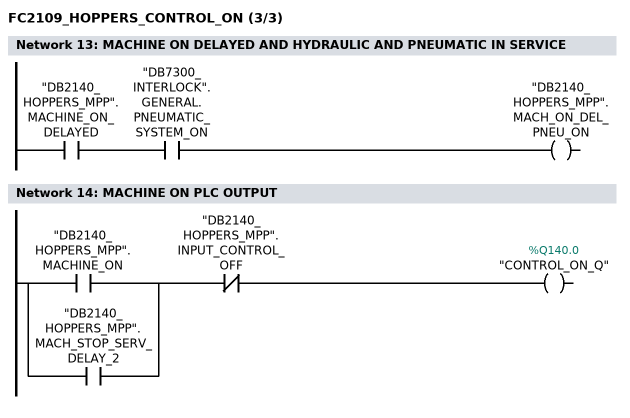
   RUNG wire#powerrail
      Contact( "DB2140_HOPPERS_MPP".MACHINE_ON_DELAYED )
      Contact( "DB7300_INTERLOCK".GENERAL.PNEUMATIC_SYSTEM_ON )
      Coil( "DB2140_HOPPERS_MPP".MACH_ON_DEL_PNEU_ON )
   END_RUNG
   // the same network as SCL:
   "DB2140_HOPPERS_MPP".MACH_ON_DEL_PNEU_ON := "DB2140_HOPPERS_MPP".MACHINE_ON_DELAYED AND "DB7300_INTERLOCK".GENERAL.PNEUMATIC_SYSTEM_ON;
END_REGION

REGION Network 14: MACHINE ON PLC OUTPUT
   RUNG wire#powerrail
      Contact( "DB2140_HOPPERS_MPP".MACHINE_ON )
      wire#w1
      I_Contact( "DB2140_HOPPERS_MPP".INPUT_CONTROL_OFF )
      Coil( "CONTROL_ON_Q" )
   END_RUNG
   RUNG wire#powerrail
      Contact( "DB2140_HOPPERS_MPP".MACH_STOP_SERV_DELAY_2 )
   END_RUNG wire#w1
   // the same network as SCL:
   "CONTROL_ON_Q" := ("DB2140_HOPPERS_MPP".MACHINE_ON OR "DB2140_HOPPERS_MPP".MACH_STOP_SERV_DELAY_2) AND NOT "DB2140_HOPPERS_MPP".INPUT_CONTROL_OFF;
END_REGION
END_FUNCTION

FUNCTION "FC2140_HOPPERS_BUTTONS" : Void   // FC2140, LAD
{ S7_Optimized_Access := 'FALSE' }
AUTHOR : ETXETAR
VERSION : 1.0
// stored: AutoNumber false, IsIECCheckEnabled false, SetENOAutomatically false, UDAEnableTagReadback false
   VAR_TEMP
      O_BYTE_0 : Struct   // OPTIONS BYTE 0
         IPC : Bool;   // IPC OPTION
      END_STRUCT;
      TCU_INDEX_SEL : Int;
   END_VAR
   VAR CONSTANT
      FC_NUMBER : DInt := 2140;   // FC NUMBER
   END_VAR
   VAR_TEMP   // added for the SCL form of the ladder/FBD networks
      _w1 : Bool;
   END_VAR
BEGIN

REGION Network 1: OPTIONS
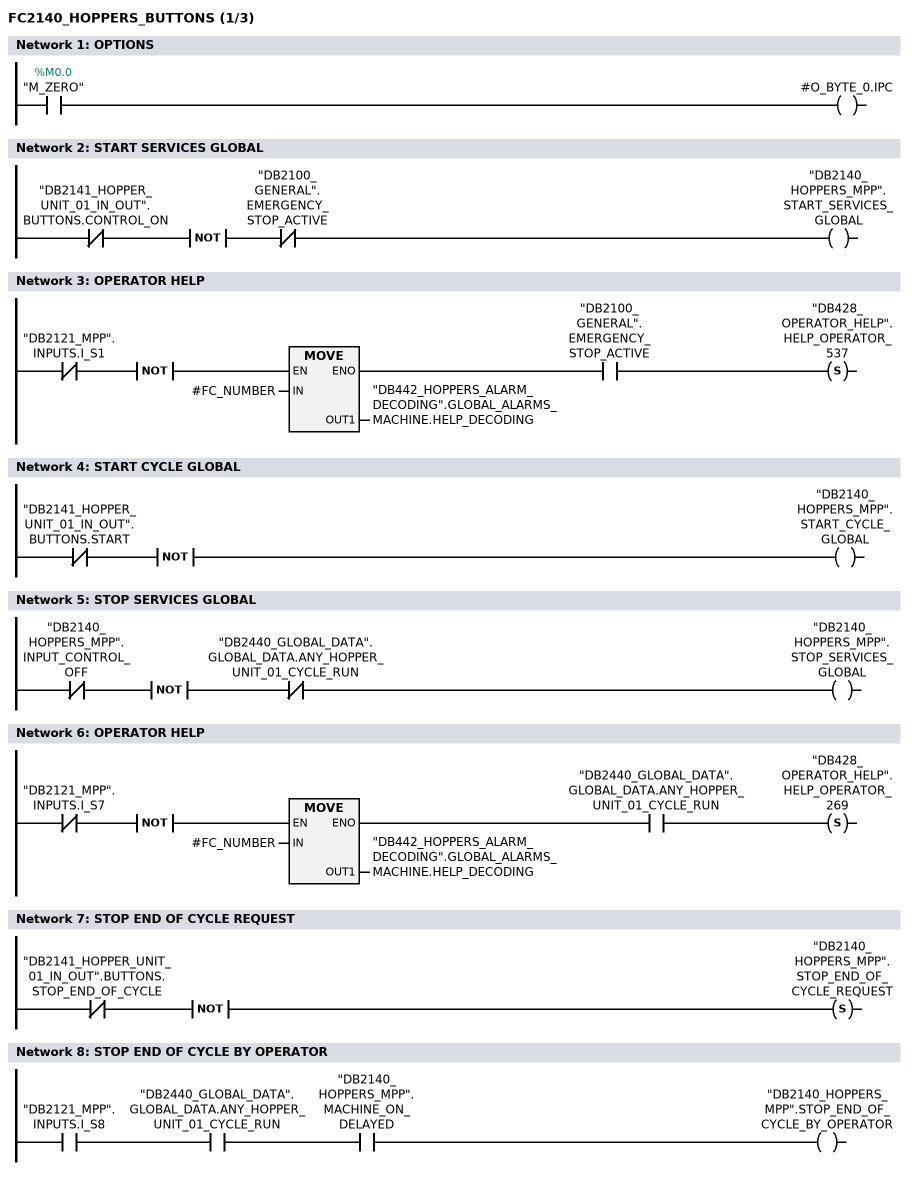
   RUNG wire#powerrail
      Contact( "M_ZERO" )
      Coil( #O_BYTE_0.IPC )
   END_RUNG
   // the same network as SCL:
   #O_BYTE_0.IPC := "M_ZERO";
END_REGION

REGION Network 2: START SERVICES GLOBAL
   RUNG wire#powerrail
      I_Contact( "DB2141_HOPPER_UNIT_01_IN_OUT".BUTTONS.CONTROL_ON )
      Not()
      I_Contact( "DB2100_GENERAL".EMERGENCY_STOP_ACTIVE )
      Coil( "DB2140_HOPPERS_MPP".START_SERVICES_GLOBAL )
   END_RUNG
   // the same network as SCL:
   "DB2140_HOPPERS_MPP".START_SERVICES_GLOBAL := NOT (NOT "DB2141_HOPPER_UNIT_01_IN_OUT".BUTTONS.CONTROL_ON) AND NOT "DB2100_GENERAL".EMERGENCY_STOP_ACTIVE;
END_REGION

REGION Network 3: OPERATOR HELP
   RUNG wire#powerrail
      I_Contact( "DB2121_MPP".INPUTS.I_S1 )
      Not()
      { S7_GenerateENO := "TRUE" } Move(in := #FC_NUMBER, out1 => "DB442_HOPPERS_ALARM_DECODING".GLOBAL_ALARMS_MACHINE.HELP_DECODING)
      Contact( "DB2100_GENERAL".EMERGENCY_STOP_ACTIVE )
      S_Coil( "DB428_OPERATOR_HELP".HELP_OPERATOR_537 )
   END_RUNG
   // the same network as SCL:
   // ENO of a box is taken as its EN; it also drops when the box reports an error
   #_w1 := NOT (NOT "DB2121_MPP".INPUTS.I_S1);
   IF #_w1 THEN "DB442_HOPPERS_ALARM_DECODING".GLOBAL_ALARMS_MACHINE.HELP_DECODING := #FC_NUMBER; END_IF;
   IF #_w1 AND "DB2100_GENERAL".EMERGENCY_STOP_ACTIVE THEN
       "DB428_OPERATOR_HELP".HELP_OPERATOR_537 := TRUE;
   END_IF;
END_REGION

REGION Network 4: START CYCLE GLOBAL
   RUNG wire#powerrail
      I_Contact( "DB2141_HOPPER_UNIT_01_IN_OUT".BUTTONS.START )
      Not()
      Coil( "DB2140_HOPPERS_MPP".START_CYCLE_GLOBAL )
   END_RUNG
   // the same network as SCL:
   "DB2140_HOPPERS_MPP".START_CYCLE_GLOBAL := NOT (NOT "DB2141_HOPPER_UNIT_01_IN_OUT".BUTTONS.START);
END_REGION

REGION Network 5: STOP SERVICES GLOBAL
   RUNG wire#powerrail
      I_Contact( "DB2140_HOPPERS_MPP".INPUT_CONTROL_OFF )
      Not()
      I_Contact( "DB2440_GLOBAL_DATA".GLOBAL_DATA.ANY_HOPPER_UNIT_01_CYCLE_RUN )
      Coil( "DB2140_HOPPERS_MPP".STOP_SERVICES_GLOBAL )
   END_RUNG
   // the same network as SCL:
   "DB2140_HOPPERS_MPP".STOP_SERVICES_GLOBAL := NOT (NOT "DB2140_HOPPERS_MPP".INPUT_CONTROL_OFF) AND NOT "DB2440_GLOBAL_DATA".GLOBAL_DATA.ANY_HOPPER_UNIT_01_CYCLE_RUN;
END_REGION

REGION Network 6: OPERATOR HELP
   RUNG wire#powerrail
      I_Contact( "DB2121_MPP".INPUTS.I_S7 )
      Not()
      { S7_GenerateENO := "TRUE" } Move(in := #FC_NUMBER, out1 => "DB442_HOPPERS_ALARM_DECODING".GLOBAL_ALARMS_MACHINE.HELP_DECODING)
      Contact( "DB2440_GLOBAL_DATA".GLOBAL_DATA.ANY_HOPPER_UNIT_01_CYCLE_RUN )
      S_Coil( "DB428_OPERATOR_HELP".HELP_OPERATOR_269 )
   END_RUNG
   // the same network as SCL:
   // ENO of a box is taken as its EN; it also drops when the box reports an error
   #_w1 := NOT (NOT "DB2121_MPP".INPUTS.I_S7);
   IF #_w1 THEN "DB442_HOPPERS_ALARM_DECODING".GLOBAL_ALARMS_MACHINE.HELP_DECODING := #FC_NUMBER; END_IF;
   IF #_w1 AND "DB2440_GLOBAL_DATA".GLOBAL_DATA.ANY_HOPPER_UNIT_01_CYCLE_RUN THEN
       "DB428_OPERATOR_HELP".HELP_OPERATOR_269 := TRUE;
   END_IF;
END_REGION

REGION Network 7: STOP END OF CYCLE REQUEST
   RUNG wire#powerrail
      I_Contact( "DB2141_HOPPER_UNIT_01_IN_OUT".BUTTONS.STOP_END_OF_CYCLE )
      Not()
      S_Coil( "DB2140_HOPPERS_MPP".STOP_END_OF_CYCLE_REQUEST )
   END_RUNG
   // the same network as SCL:
   IF NOT (NOT "DB2141_HOPPER_UNIT_01_IN_OUT".BUTTONS.STOP_END_OF_CYCLE) THEN
       "DB2140_HOPPERS_MPP".STOP_END_OF_CYCLE_REQUEST := TRUE;
   END_IF;
END_REGION

REGION Network 8: STOP END OF CYCLE BY OPERATOR
   RUNG wire#powerrail
      Contact( "DB2121_MPP".INPUTS.I_S8 )
      Contact( "DB2440_GLOBAL_DATA".GLOBAL_DATA.ANY_HOPPER_UNIT_01_CYCLE_RUN )
      Contact( "DB2140_HOPPERS_MPP".MACHINE_ON_DELAYED )
      Coil( "DB2140_HOPPERS_MPP".STOP_END_OF_CYCLE_BY_OPERATOR )
   END_RUNG
   // the same network as SCL:
   "DB2140_HOPPERS_MPP".STOP_END_OF_CYCLE_BY_OPERATOR := "DB2121_MPP".INPUTS.I_S8 AND "DB2440_GLOBAL_DATA".GLOBAL_DATA.ANY_HOPPER_UNIT_01_CYCLE_RUN AND "DB2140_HOPPERS_MPP".MACHINE_ON_DELAYED;
END_REGION

REGION Network 9: MAIN PANEL OPERATOR REQUEST STOP AT END OF CYCLE
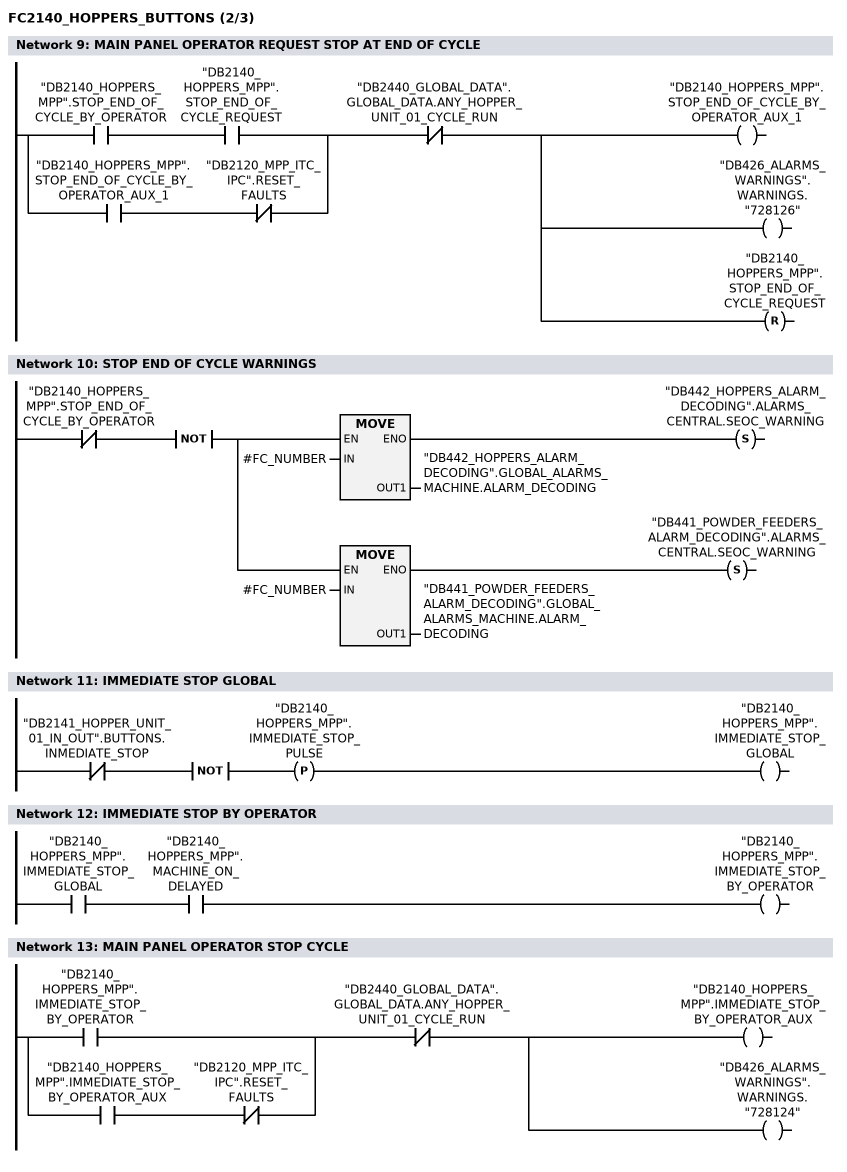
   RUNG wire#powerrail
      Contact( "DB2140_HOPPERS_MPP".STOP_END_OF_CYCLE_BY_OPERATOR )
      Contact( "DB2140_HOPPERS_MPP".STOP_END_OF_CYCLE_REQUEST )
      wire#w1
      I_Contact( "DB2440_GLOBAL_DATA".GLOBAL_DATA.ANY_HOPPER_UNIT_01_CYCLE_RUN )
      wire#w2
      Coil( "DB2140_HOPPERS_MPP".STOP_END_OF_CYCLE_BY_OPERATOR_AUX_1 )
   END_RUNG
   RUNG wire#powerrail
      Contact( "DB2140_HOPPERS_MPP".STOP_END_OF_CYCLE_BY_OPERATOR_AUX_1 )
      I_Contact( "DB2120_MPP_ITC_IPC".RESET_FAULTS )
   END_RUNG wire#w1
   RUNG wire#w2
      Coil( "DB426_ALARMS_WARNINGS".WARNINGS."728126" )
   END_RUNG
   RUNG wire#w2
      R_Coil( "DB2140_HOPPERS_MPP".STOP_END_OF_CYCLE_REQUEST )
   END_RUNG
   // the same network as SCL:
   "DB2140_HOPPERS_MPP".STOP_END_OF_CYCLE_BY_OPERATOR_AUX_1 := (("DB2140_HOPPERS_MPP".STOP_END_OF_CYCLE_BY_OPERATOR AND "DB2140_HOPPERS_MPP".STOP_END_OF_CYCLE_REQUEST) OR ("DB2140_HOPPERS_MPP".STOP_END_OF_CYCLE_BY_OPERATOR_AUX_1 AND NOT "DB2120_MPP_ITC_IPC".RESET_FAULTS)) AND NOT "DB2440_GLOBAL_DATA".GLOBAL_DATA.ANY_HOPPER_UNIT_01_CYCLE_RUN;
   "DB426_ALARMS_WARNINGS".WARNINGS."728126" := "DB2140_HOPPERS_MPP".STOP_END_OF_CYCLE_BY_OPERATOR_AUX_1;
   IF "DB2140_HOPPERS_MPP".STOP_END_OF_CYCLE_BY_OPERATOR_AUX_1 THEN
       "DB2140_HOPPERS_MPP".STOP_END_OF_CYCLE_REQUEST := FALSE;
   END_IF;
END_REGION

REGION Network 10: STOP END OF CYCLE WARNINGS
   RUNG wire#powerrail
      I_Contact( "DB2140_HOPPERS_MPP".STOP_END_OF_CYCLE_BY_OPERATOR )
      Not()
      wire#w1
      { S7_GenerateENO := "TRUE" } Move(in := #FC_NUMBER, out1 => "DB442_HOPPERS_ALARM_DECODING".GLOBAL_ALARMS_MACHINE.ALARM_DECODING)
      S_Coil( "DB442_HOPPERS_ALARM_DECODING".ALARMS_CENTRAL.SEOC_WARNING )
   END_RUNG
   RUNG wire#w1
      { S7_GenerateENO := "TRUE" } Move(in := #FC_NUMBER, out1 => "DB441_POWDER_FEEDERS_ALARM_DECODING".GLOBAL_ALARMS_MACHINE.ALARM_DECODING)
      S_Coil( "DB441_POWDER_FEEDERS_ALARM_DECODING".ALARMS_CENTRAL.SEOC_WARNING )
   END_RUNG
   // the same network as SCL:
   // ENO of a box is taken as its EN; it also drops when the box reports an error
   IF NOT (NOT "DB2140_HOPPERS_MPP".STOP_END_OF_CYCLE_BY_OPERATOR) THEN
       "DB442_HOPPERS_ALARM_DECODING".GLOBAL_ALARMS_MACHINE.ALARM_DECODING := #FC_NUMBER;
       "DB442_HOPPERS_ALARM_DECODING".ALARMS_CENTRAL.SEOC_WARNING := TRUE;
       "DB441_POWDER_FEEDERS_ALARM_DECODING".GLOBAL_ALARMS_MACHINE.ALARM_DECODING := #FC_NUMBER;
       "DB441_POWDER_FEEDERS_ALARM_DECODING".ALARMS_CENTRAL.SEOC_WARNING := TRUE;
   END_IF;
END_REGION

REGION Network 11: IMMEDIATE STOP GLOBAL
   RUNG wire#powerrail
      I_Contact( "DB2141_HOPPER_UNIT_01_IN_OUT".BUTTONS.INMEDIATE_STOP )
      Not()
      P_Trig( "DB2140_HOPPERS_MPP".IMMEDIATE_STOP_PULSE )
      Coil( "DB2140_HOPPERS_MPP".IMMEDIATE_STOP_GLOBAL )
   END_RUNG
   // the same network as SCL:
   #_w1 := NOT (NOT "DB2141_HOPPER_UNIT_01_IN_OUT".BUTTONS.INMEDIATE_STOP) AND NOT "DB2140_HOPPERS_MPP".IMMEDIATE_STOP_PULSE;   // rising edge
   "DB2140_HOPPERS_MPP".IMMEDIATE_STOP_PULSE := NOT (NOT "DB2141_HOPPER_UNIT_01_IN_OUT".BUTTONS.INMEDIATE_STOP);
   "DB2140_HOPPERS_MPP".IMMEDIATE_STOP_GLOBAL := #_w1;
END_REGION

REGION Network 12: IMMEDIATE STOP BY OPERATOR
   RUNG wire#powerrail
      Contact( "DB2140_HOPPERS_MPP".IMMEDIATE_STOP_GLOBAL )
      Contact( "DB2140_HOPPERS_MPP".MACHINE_ON_DELAYED )
      Coil( "DB2140_HOPPERS_MPP".IMMEDIATE_STOP_BY_OPERATOR )
   END_RUNG
   // the same network as SCL:
   "DB2140_HOPPERS_MPP".IMMEDIATE_STOP_BY_OPERATOR := "DB2140_HOPPERS_MPP".IMMEDIATE_STOP_GLOBAL AND "DB2140_HOPPERS_MPP".MACHINE_ON_DELAYED;
END_REGION

REGION Network 13: MAIN PANEL OPERATOR STOP CYCLE
   RUNG wire#powerrail
      Contact( "DB2140_HOPPERS_MPP".IMMEDIATE_STOP_BY_OPERATOR )
      wire#w1
      I_Contact( "DB2440_GLOBAL_DATA".GLOBAL_DATA.ANY_HOPPER_UNIT_01_CYCLE_RUN )
      wire#w2
      Coil( "DB2140_HOPPERS_MPP".IMMEDIATE_STOP_BY_OPERATOR_AUX )
   END_RUNG
   RUNG wire#powerrail
      Contact( "DB2140_HOPPERS_MPP".IMMEDIATE_STOP_BY_OPERATOR_AUX )
      I_Contact( "DB2120_MPP_ITC_IPC".RESET_FAULTS )
   END_RUNG wire#w1
   RUNG wire#w2
      Coil( "DB426_ALARMS_WARNINGS".WARNINGS."728124" )
   END_RUNG
   // the same network as SCL:
   "DB2140_HOPPERS_MPP".IMMEDIATE_STOP_BY_OPERATOR_AUX := ("DB2140_HOPPERS_MPP".IMMEDIATE_STOP_BY_OPERATOR OR ("DB2140_HOPPERS_MPP".IMMEDIATE_STOP_BY_OPERATOR_AUX AND NOT "DB2120_MPP_ITC_IPC".RESET_FAULTS)) AND NOT "DB2440_GLOBAL_DATA".GLOBAL_DATA.ANY_HOPPER_UNIT_01_CYCLE_RUN;
   "DB426_ALARMS_WARNINGS".WARNINGS."728124" := "DB2140_HOPPERS_MPP".IMMEDIATE_STOP_BY_OPERATOR_AUX;
END_REGION

REGION Network 14: IMMEDIATE STOP WARNING
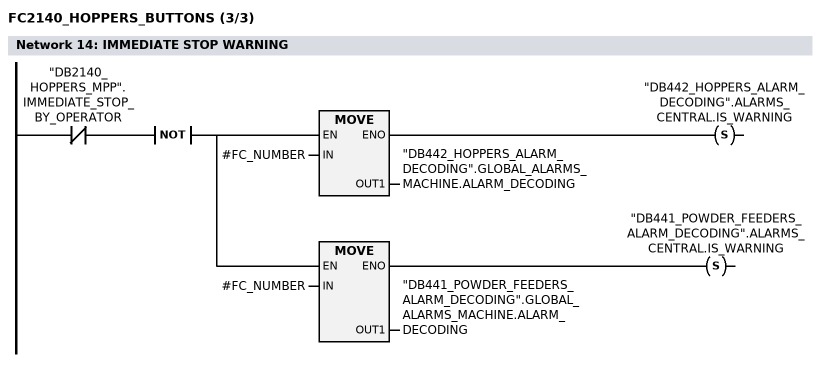
   RUNG wire#powerrail
      I_Contact( "DB2140_HOPPERS_MPP".IMMEDIATE_STOP_BY_OPERATOR )
      Not()
      wire#w1
      { S7_GenerateENO := "TRUE" } Move(in := #FC_NUMBER, out1 => "DB442_HOPPERS_ALARM_DECODING".GLOBAL_ALARMS_MACHINE.ALARM_DECODING)
      S_Coil( "DB442_HOPPERS_ALARM_DECODING".ALARMS_CENTRAL.IS_WARNING )
   END_RUNG
   RUNG wire#w1
      { S7_GenerateENO := "TRUE" } Move(in := #FC_NUMBER, out1 => "DB441_POWDER_FEEDERS_ALARM_DECODING".GLOBAL_ALARMS_MACHINE.ALARM_DECODING)
      S_Coil( "DB441_POWDER_FEEDERS_ALARM_DECODING".ALARMS_CENTRAL.IS_WARNING )
   END_RUNG
   // the same network as SCL:
   // ENO of a box is taken as its EN; it also drops when the box reports an error
   IF NOT (NOT "DB2140_HOPPERS_MPP".IMMEDIATE_STOP_BY_OPERATOR) THEN
       "DB442_HOPPERS_ALARM_DECODING".GLOBAL_ALARMS_MACHINE.ALARM_DECODING := #FC_NUMBER;
       "DB442_HOPPERS_ALARM_DECODING".ALARMS_CENTRAL.IS_WARNING := TRUE;
       "DB441_POWDER_FEEDERS_ALARM_DECODING".GLOBAL_ALARMS_MACHINE.ALARM_DECODING := #FC_NUMBER;
       "DB441_POWDER_FEEDERS_ALARM_DECODING".ALARMS_CENTRAL.IS_WARNING := TRUE;
   END_IF;
END_REGION
END_FUNCTION

FUNCTION "FC2141_HOPPERS_LAMPS" : Void   // FC2141, LAD
{ S7_Optimized_Access := 'FALSE' }
AUTHOR : ETXETAR
VERSION : 1.0
// stored: AutoNumber false, IsIECCheckEnabled false, SetENOAutomatically false, UDAEnableTagReadback false
   VAR_TEMP
      ONE : Int;
      RETVAL1 : Int;
      SIMU_PANEL_HMI_SEL : Bool;   // SIMULATED PANEL IN HMI SELECTED
   END_VAR
   VAR CONSTANT
      FC_NUMBER : DInt := 2141;   // FC NUMBER
   END_VAR
BEGIN

REGION Network 1: LAMP - CONTROL ON
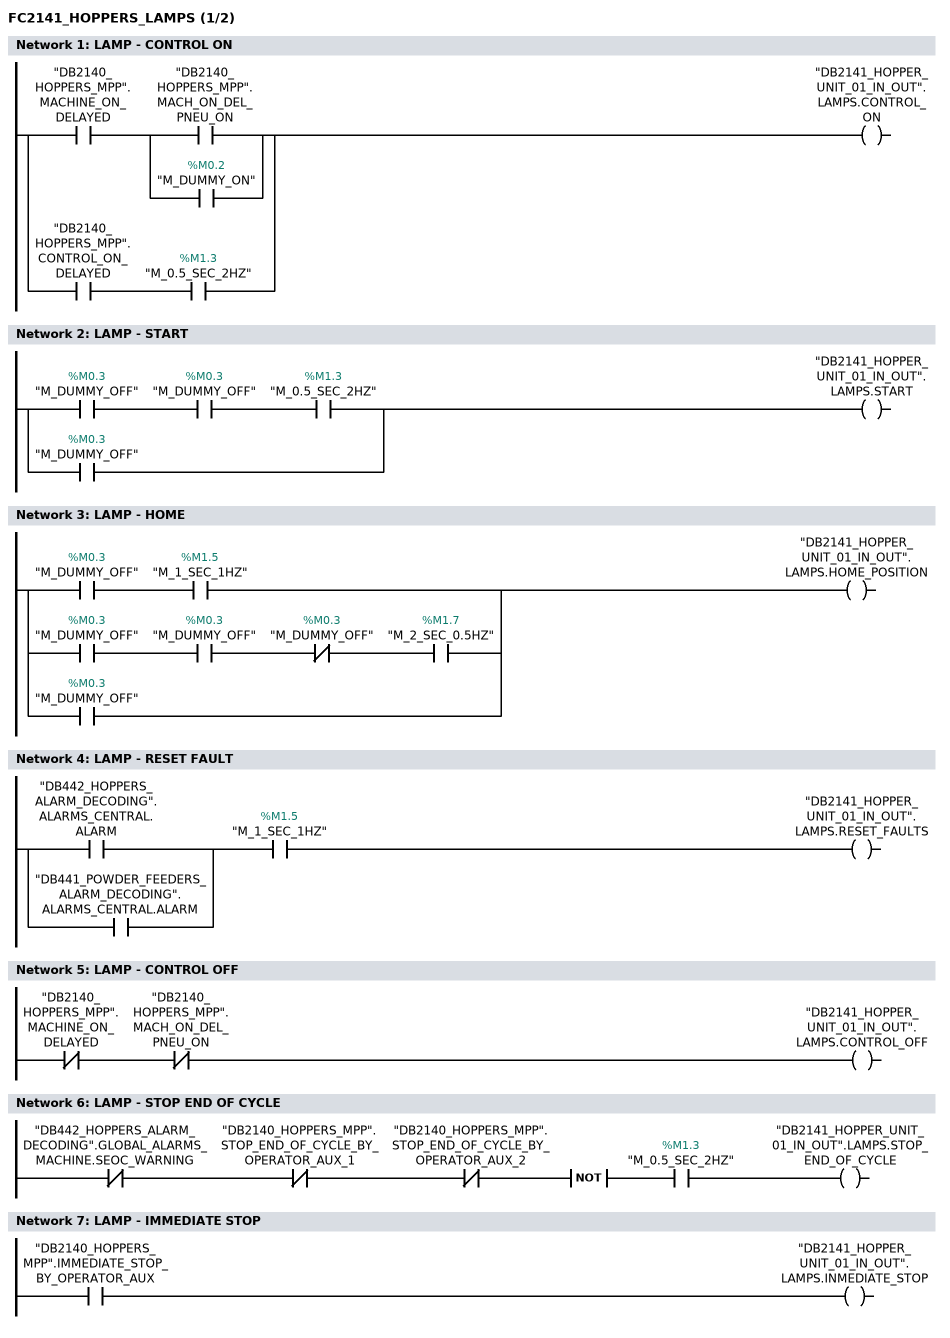
   RUNG wire#powerrail
      Contact( "DB2140_HOPPERS_MPP".MACHINE_ON_DELAYED )
      wire#w1
      Contact( "DB2140_HOPPERS_MPP".MACH_ON_DEL_PNEU_ON )
      wire#w2
      Coil( "DB2141_HOPPER_UNIT_01_IN_OUT".LAMPS.CONTROL_ON )
   END_RUNG
   RUNG wire#w1
      Contact( "M_DUMMY_ON" )
   END_RUNG wire#w2
   RUNG wire#powerrail
      Contact( "DB2140_HOPPERS_MPP".CONTROL_ON_DELAYED )
      Contact( "M_0.5_SEC_2HZ" )
   END_RUNG wire#w2
   // the same network as SCL:
   "DB2141_HOPPER_UNIT_01_IN_OUT".LAMPS.CONTROL_ON := ("DB2140_HOPPERS_MPP".MACHINE_ON_DELAYED AND ("DB2140_HOPPERS_MPP".MACH_ON_DEL_PNEU_ON OR "M_DUMMY_ON")) OR ("DB2140_HOPPERS_MPP".CONTROL_ON_DELAYED AND "M_0.5_SEC_2HZ");
END_REGION

REGION Network 2: LAMP - START
   RUNG wire#powerrail
      Contact( "M_DUMMY_OFF" )
      Contact( "M_DUMMY_OFF" )
      Contact( "M_0.5_SEC_2HZ" )
      wire#w1
      Coil( "DB2141_HOPPER_UNIT_01_IN_OUT".LAMPS.START )
   END_RUNG
   RUNG wire#powerrail
      Contact( "M_DUMMY_OFF" )
   END_RUNG wire#w1
   // the same network as SCL:
   "DB2141_HOPPER_UNIT_01_IN_OUT".LAMPS.START := ("M_DUMMY_OFF" AND "M_DUMMY_OFF" AND "M_0.5_SEC_2HZ") OR "M_DUMMY_OFF";
END_REGION

REGION Network 3: LAMP - HOME
   RUNG wire#powerrail
      Contact( "M_DUMMY_OFF" )
      Contact( "M_1_SEC_1HZ" )
      wire#w1
      Coil( "DB2141_HOPPER_UNIT_01_IN_OUT".LAMPS.HOME_POSITION )
   END_RUNG
   RUNG wire#powerrail
      Contact( "M_DUMMY_OFF" )
      Contact( "M_DUMMY_OFF" )
      I_Contact( "M_DUMMY_OFF" )
      Contact( "M_2_SEC_0.5HZ" )
   END_RUNG wire#w1
   RUNG wire#powerrail
      Contact( "M_DUMMY_OFF" )
   END_RUNG wire#w1
   // the same network as SCL:
   "DB2141_HOPPER_UNIT_01_IN_OUT".LAMPS.HOME_POSITION := ("M_DUMMY_OFF" AND "M_1_SEC_1HZ") OR ("M_DUMMY_OFF" AND "M_DUMMY_OFF" AND NOT "M_DUMMY_OFF" AND "M_2_SEC_0.5HZ") OR "M_DUMMY_OFF";
END_REGION

REGION Network 4: LAMP - RESET FAULT
   RUNG wire#powerrail
      Contact( "DB442_HOPPERS_ALARM_DECODING".ALARMS_CENTRAL.ALARM )
      wire#w1
      Contact( "M_1_SEC_1HZ" )
      Coil( "DB2141_HOPPER_UNIT_01_IN_OUT".LAMPS.RESET_FAULTS )
   END_RUNG
   RUNG wire#powerrail
      Contact( "DB441_POWDER_FEEDERS_ALARM_DECODING".ALARMS_CENTRAL.ALARM )
   END_RUNG wire#w1
   // the same network as SCL:
   "DB2141_HOPPER_UNIT_01_IN_OUT".LAMPS.RESET_FAULTS := ("DB442_HOPPERS_ALARM_DECODING".ALARMS_CENTRAL.ALARM OR "DB441_POWDER_FEEDERS_ALARM_DECODING".ALARMS_CENTRAL.ALARM) AND "M_1_SEC_1HZ";
END_REGION

REGION Network 5: LAMP - CONTROL OFF
   RUNG wire#powerrail
      I_Contact( "DB2140_HOPPERS_MPP".MACHINE_ON_DELAYED )
      I_Contact( "DB2140_HOPPERS_MPP".MACH_ON_DEL_PNEU_ON )
      Coil( "DB2141_HOPPER_UNIT_01_IN_OUT".LAMPS.CONTROL_OFF )
   END_RUNG
   // the same network as SCL:
   "DB2141_HOPPER_UNIT_01_IN_OUT".LAMPS.CONTROL_OFF := NOT "DB2140_HOPPERS_MPP".MACHINE_ON_DELAYED AND NOT "DB2140_HOPPERS_MPP".MACH_ON_DEL_PNEU_ON;
END_REGION

REGION Network 6: LAMP - STOP END OF CYCLE
   RUNG wire#powerrail
      I_Contact( "DB442_HOPPERS_ALARM_DECODING".GLOBAL_ALARMS_MACHINE.SEOC_WARNING )
      I_Contact( "DB2140_HOPPERS_MPP".STOP_END_OF_CYCLE_BY_OPERATOR_AUX_1 )
      I_Contact( "DB2140_HOPPERS_MPP".STOP_END_OF_CYCLE_BY_OPERATOR_AUX_2 )
      Not()
      Contact( "M_0.5_SEC_2HZ" )
      Coil( "DB2141_HOPPER_UNIT_01_IN_OUT".LAMPS.STOP_END_OF_CYCLE )
   END_RUNG
   // the same network as SCL:
   "DB2141_HOPPER_UNIT_01_IN_OUT".LAMPS.STOP_END_OF_CYCLE := NOT (NOT "DB442_HOPPERS_ALARM_DECODING".GLOBAL_ALARMS_MACHINE.SEOC_WARNING AND NOT "DB2140_HOPPERS_MPP".STOP_END_OF_CYCLE_BY_OPERATOR_AUX_1 AND NOT "DB2140_HOPPERS_MPP".STOP_END_OF_CYCLE_BY_OPERATOR_AUX_2) AND "M_0.5_SEC_2HZ";
END_REGION

REGION Network 7: LAMP - IMMEDIATE STOP
   RUNG wire#powerrail
      Contact( "DB2140_HOPPERS_MPP".IMMEDIATE_STOP_BY_OPERATOR_AUX )
      Coil( "DB2141_HOPPER_UNIT_01_IN_OUT".LAMPS.INMEDIATE_STOP )
   END_RUNG
   // the same network as SCL:
   "DB2141_HOPPER_UNIT_01_IN_OUT".LAMPS.INMEDIATE_STOP := "DB2140_HOPPERS_MPP".IMMEDIATE_STOP_BY_OPERATOR_AUX;
END_REGION

REGION Network 8: LAMPS - MODES
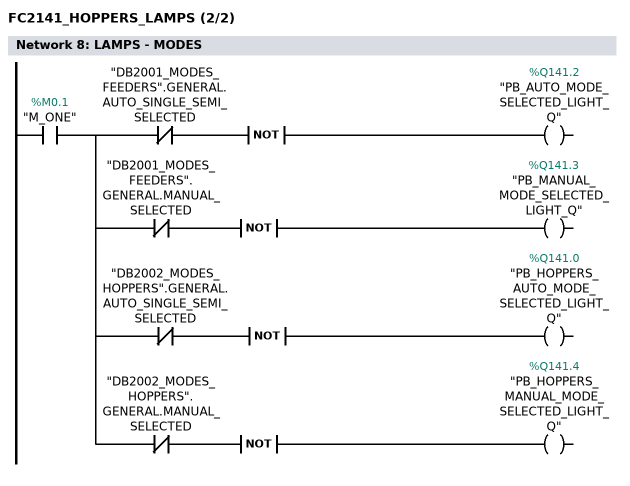
   RUNG wire#powerrail
      Contact( "M_ONE" )
      wire#w1
      I_Contact( "DB2001_MODES_FEEDERS".GENERAL.AUTO_SINGLE_SEMI_SELECTED )
      Not()
      Coil( "PB_AUTO_MODE_SELECTED_LIGHT_Q" )
   END_RUNG
   RUNG wire#w1
      I_Contact( "DB2001_MODES_FEEDERS".GENERAL.MANUAL_SELECTED )
      Not()
      Coil( "PB_MANUAL_MODE_SELECTED_LIGHT_Q" )
   END_RUNG
   RUNG wire#w1
      I_Contact( "DB2002_MODES_HOPPERS".GENERAL.AUTO_SINGLE_SEMI_SELECTED )
      Not()
      Coil( "PB_HOPPERS_AUTO_MODE_SELECTED_LIGHT_Q" )
   END_RUNG
   RUNG wire#w1
      I_Contact( "DB2002_MODES_HOPPERS".GENERAL.MANUAL_SELECTED )
      Not()
      Coil( "PB_HOPPERS_MANUAL_MODE_SELECTED_LIGHT_Q" )
   END_RUNG
   // the same network as SCL:
   "PB_AUTO_MODE_SELECTED_LIGHT_Q" := NOT ("M_ONE" AND NOT "DB2001_MODES_FEEDERS".GENERAL.AUTO_SINGLE_SEMI_SELECTED);
   "PB_MANUAL_MODE_SELECTED_LIGHT_Q" := NOT ("M_ONE" AND NOT "DB2001_MODES_FEEDERS".GENERAL.MANUAL_SELECTED);
   "PB_HOPPERS_AUTO_MODE_SELECTED_LIGHT_Q" := NOT ("M_ONE" AND NOT "DB2002_MODES_HOPPERS".GENERAL.AUTO_SINGLE_SEMI_SELECTED);
   "PB_HOPPERS_MANUAL_MODE_SELECTED_LIGHT_Q" := NOT ("M_ONE" AND NOT "DB2002_MODES_HOPPERS".GENERAL.MANUAL_SELECTED);
END_REGION
END_FUNCTION

FUNCTION "FC21000_POWDER_FEEDER_MAIN" : Void   // FC21000, LAD
TITLE = FC21000 POWDER FEEDER MAIN
{ S7_Optimized_Access := 'TRUE' }
VERSION : 0.1
// stored: AutoNumber false, IsIECCheckEnabled false, SetENOAutomatically false, UDAEnableTagReadback false
   VAR_TEMP
      ret_val_1 : Int;
      OPTIONS_OFF : Bool;
      OPTIONS_ON : Bool;
      POWDER_SWITCH_OPTION : Bool;
      MEDICOAT_OPTION : Bool;
   END_VAR
BEGIN

REGION Network 1: OPTIONS OFF
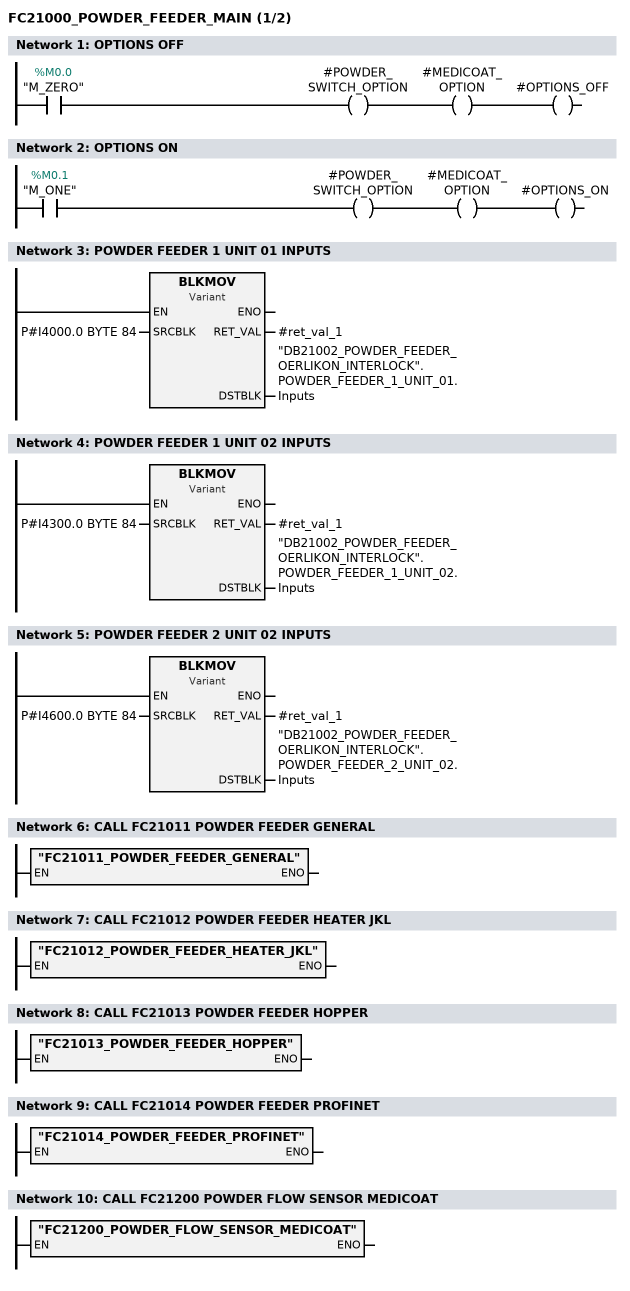
   RUNG wire#powerrail
      Contact( "M_ZERO" )
      Coil( #POWDER_SWITCH_OPTION )
      Coil( #MEDICOAT_OPTION )
      Coil( #OPTIONS_OFF )
   END_RUNG
   // the same network as SCL:
   #POWDER_SWITCH_OPTION := "M_ZERO";
   #MEDICOAT_OPTION := "M_ZERO";
   #OPTIONS_OFF := "M_ZERO";
END_REGION

REGION Network 2: OPTIONS ON
   RUNG wire#powerrail
      Contact( "M_ONE" )
      Coil( #POWDER_SWITCH_OPTION )
      Coil( #MEDICOAT_OPTION )
      Coil( #OPTIONS_ON )
   END_RUNG
   // the same network as SCL:
   #POWDER_SWITCH_OPTION := "M_ONE";
   #MEDICOAT_OPTION := "M_ONE";
   #OPTIONS_ON := "M_ONE";
END_REGION

REGION Network 3: POWDER FEEDER 1 UNIT 01 INPUTS
   RUNG wire#powerrail
      { S7_Templates := "blk_type := Variant" } BLKMOV(SRCBLK := P#I4000.0 BYTE 84, RET_VAL => #ret_val_1, DSTBLK => "DB21002_POWDER_FEEDER_OERLIKON_INTERLOCK".POWDER_FEEDER_1_UNIT_01.Inputs)
   END_RUNG
   // the same network as SCL:
   #ret_val_1 := BLKMOV(SRCBLK := P#I4000.0 BYTE 84,
                        DSTBLK => "DB21002_POWDER_FEEDER_OERLIKON_INTERLOCK".POWDER_FEEDER_1_UNIT_01.Inputs);
END_REGION

REGION Network 4: POWDER FEEDER 1 UNIT 02 INPUTS
   RUNG wire#powerrail
      { S7_Templates := "blk_type := Variant" } BLKMOV(SRCBLK := P#I4300.0 BYTE 84, RET_VAL => #ret_val_1, DSTBLK => "DB21002_POWDER_FEEDER_OERLIKON_INTERLOCK".POWDER_FEEDER_1_UNIT_02.Inputs)
   END_RUNG
   // the same network as SCL:
   #ret_val_1 := BLKMOV(SRCBLK := P#I4300.0 BYTE 84,
                        DSTBLK => "DB21002_POWDER_FEEDER_OERLIKON_INTERLOCK".POWDER_FEEDER_1_UNIT_02.Inputs);
END_REGION

REGION Network 5: POWDER FEEDER 2 UNIT 02 INPUTS
   RUNG wire#powerrail
      { S7_Templates := "blk_type := Variant" } BLKMOV(SRCBLK := P#I4600.0 BYTE 84, RET_VAL => #ret_val_1, DSTBLK => "DB21002_POWDER_FEEDER_OERLIKON_INTERLOCK".POWDER_FEEDER_2_UNIT_02.Inputs)
   END_RUNG
   // the same network as SCL:
   #ret_val_1 := BLKMOV(SRCBLK := P#I4600.0 BYTE 84,
                        DSTBLK => "DB21002_POWDER_FEEDER_OERLIKON_INTERLOCK".POWDER_FEEDER_2_UNIT_02.Inputs);
END_REGION

REGION Network 6: CALL FC21011 POWDER FEEDER GENERAL
   RUNG wire#powerrail
      "FC21011_POWDER_FEEDER_GENERAL"()
   END_RUNG
   // the same network as SCL:
   "FC21011_POWDER_FEEDER_GENERAL"();
END_REGION

REGION Network 7: CALL FC21012 POWDER FEEDER HEATER JKL
   RUNG wire#powerrail
      "FC21012_POWDER_FEEDER_HEATER_JKL"()
   END_RUNG
   // the same network as SCL:
   "FC21012_POWDER_FEEDER_HEATER_JKL"();
END_REGION

REGION Network 8: CALL FC21013 POWDER FEEDER HOPPER
   RUNG wire#powerrail
      "FC21013_POWDER_FEEDER_HOPPER"()
   END_RUNG
   // the same network as SCL:
   "FC21013_POWDER_FEEDER_HOPPER"();
END_REGION

REGION Network 9: CALL FC21014 POWDER FEEDER PROFINET
   RUNG wire#powerrail
      "FC21014_POWDER_FEEDER_PROFINET"()
   END_RUNG
   // the same network as SCL:
   "FC21014_POWDER_FEEDER_PROFINET"();
END_REGION

REGION Network 10: CALL FC21200 POWDER FLOW SENSOR MEDICOAT
   RUNG wire#powerrail
      "FC21200_POWDER_FLOW_SENSOR_MEDICOAT"()
   END_RUNG
   // the same network as SCL:
   "FC21200_POWDER_FLOW_SENSOR_MEDICOAT"();
END_REGION

REGION Network 11: POWDER FEEDER 1 UNIT 01 OUTPUTS
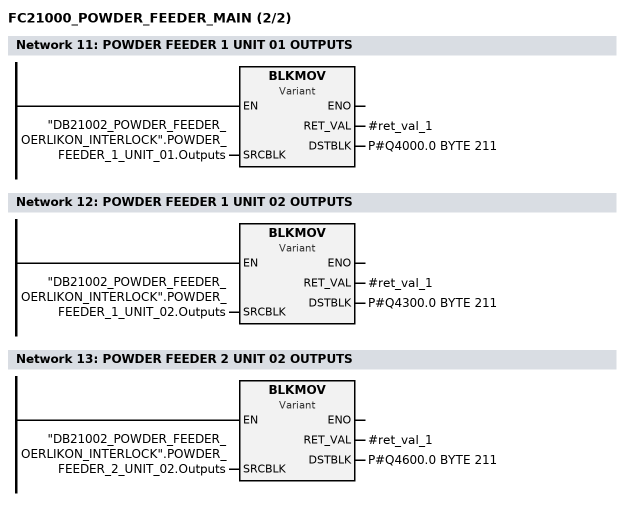
   RUNG wire#powerrail
      { S7_Templates := "blk_type := Variant" } BLKMOV(SRCBLK := "DB21002_POWDER_FEEDER_OERLIKON_INTERLOCK".POWDER_FEEDER_1_UNIT_01.Outputs, RET_VAL => #ret_val_1, DSTBLK => P#Q4000.0 BYTE 211)
   END_RUNG
   // the same network as SCL:
   #ret_val_1 := BLKMOV(SRCBLK := "DB21002_POWDER_FEEDER_OERLIKON_INTERLOCK".POWDER_FEEDER_1_UNIT_01.Outputs,
                        DSTBLK => P#Q4000.0 BYTE 211);
END_REGION

REGION Network 12: POWDER FEEDER 1 UNIT 02 OUTPUTS
   RUNG wire#powerrail
      { S7_Templates := "blk_type := Variant" } BLKMOV(SRCBLK := "DB21002_POWDER_FEEDER_OERLIKON_INTERLOCK".POWDER_FEEDER_1_UNIT_02.Outputs, RET_VAL => #ret_val_1, DSTBLK => P#Q4300.0 BYTE 211)
   END_RUNG
   // the same network as SCL:
   #ret_val_1 := BLKMOV(SRCBLK := "DB21002_POWDER_FEEDER_OERLIKON_INTERLOCK".POWDER_FEEDER_1_UNIT_02.Outputs,
                        DSTBLK => P#Q4300.0 BYTE 211);
END_REGION

REGION Network 13: POWDER FEEDER 2 UNIT 02 OUTPUTS
   RUNG wire#powerrail
      { S7_Templates := "blk_type := Variant" } BLKMOV(SRCBLK := "DB21002_POWDER_FEEDER_OERLIKON_INTERLOCK".POWDER_FEEDER_2_UNIT_02.Outputs, RET_VAL => #ret_val_1, DSTBLK => P#Q4600.0 BYTE 211)
   END_RUNG
   // the same network as SCL:
   #ret_val_1 := BLKMOV(SRCBLK := "DB21002_POWDER_FEEDER_OERLIKON_INTERLOCK".POWDER_FEEDER_2_UNIT_02.Outputs,
                        DSTBLK => P#Q4600.0 BYTE 211);
END_REGION
END_FUNCTION

FUNCTION "FC21011_POWDER_FEEDER_GENERAL" : Void   // FC21011, LAD
TITLE = FC21011 POWDER FEEDER GENERAL
{ S7_Optimized_Access := 'TRUE' }
VERSION : 0.1
// stored: AutoNumber false, IsIECCheckEnabled false, SetENOAutomatically false, UDAEnableTagReadback false
BEGIN

REGION Network 1: /////_UNIT_01_/////
END_REGION

REGION Network 2: CALL FB21011 POWDER FEEDER 1 GENERAL UNIT 01
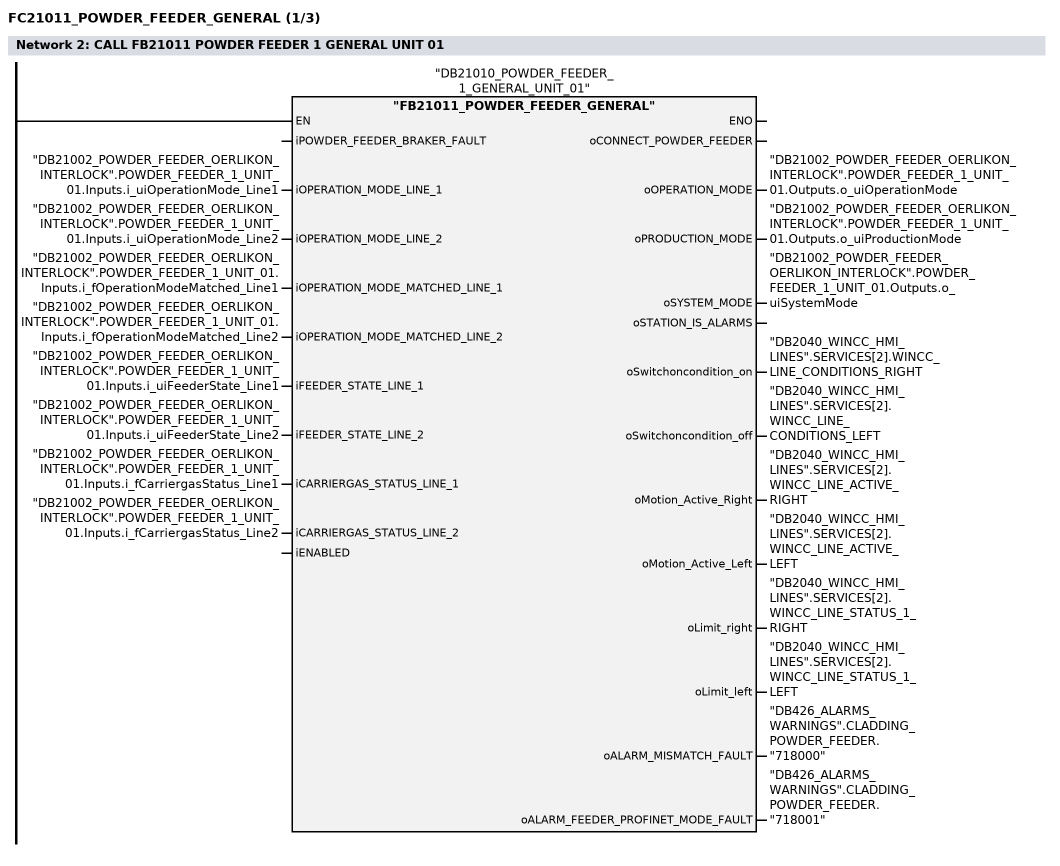
   RUNG wire#powerrail
      "DB21010_POWDER_FEEDER_1_GENERAL_UNIT_01"(iPOWDER_FEEDER_BRAKER_FAULT :=, iOPERATION_MODE_LINE_1 := "DB21002_POWDER_FEEDER_OERLIKON_INTERLOCK".POWDER_FEEDER_1_UNIT_01.Inputs.i_uiOperationMode_Line1, iOPERATION_MODE_LINE_2 := "DB21002_POWDER_FEEDER_OERLIKON_INTERLOCK".POWDER_FEEDER_1_UNIT_01.Inputs.i_uiOperationMode_Line2, iOPERATION_MODE_MATCHED_LINE_1 := "DB21002_POWDER_FEEDER_OERLIKON_INTERLOCK".POWDER_FEEDER_1_UNIT_01.Inputs.i_fOperationModeMatched_Line1, iOPERATION_MODE_MATCHED_LINE_2 := "DB21002_POWDER_FEEDER_OERLIKON_INTERLOCK".POWDER_FEEDER_1_UNIT_01.Inputs.i_fOperationModeMatched_Line2, iFEEDER_STATE_LINE_1 := "DB21002_POWDER_FEEDER_OERLIKON_INTERLOCK".POWDER_FEEDER_1_UNIT_01.Inputs.i_uiFeederState_Line1, iFEEDER_STATE_LINE_2 := "DB21002_POWDER_FEEDER_OERLIKON_INTERLOCK".POWDER_FEEDER_1_UNIT_01.Inputs.i_uiFeederState_Line2, iCARRIERGAS_STATUS_LINE_1 := "DB21002_POWDER_FEEDER_OERLIKON_INTERLOCK".POWDER_FEEDER_1_UNIT_01.Inputs.i_fCarriergasStatus_Line1, iCARRIERGAS_STATUS_LINE_2 := "DB21002_POWDER_FEEDER_OERLIKON_INTERLOCK".POWDER_FEEDER_1_UNIT_01.Inputs.i_fCarriergasStatus_Line2, iENABLED :=, oCONNECT_POWDER_FEEDER =>, oOPERATION_MODE => "DB21002_POWDER_FEEDER_OERLIKON_INTERLOCK".POWDER_FEEDER_1_UNIT_01.Outputs.o_uiOperationMode, oPRODUCTION_MODE => "DB21002_POWDER_FEEDER_OERLIKON_INTERLOCK".POWDER_FEEDER_1_UNIT_01.Outputs.o_uiProductionMode, oSYSTEM_MODE => "DB21002_POWDER_FEEDER_OERLIKON_INTERLOCK".POWDER_FEEDER_1_UNIT_01.Outputs.o_uiSystemMode, oSTATION_IS_ALARMS =>, oSwitchoncondition_on => "DB2040_WINCC_HMI_LINES".SERVICES[2].WINCC_LINE_CONDITIONS_RIGHT, oSwitchoncondition_off => "DB2040_WINCC_HMI_LINES".SERVICES[2].WINCC_LINE_CONDITIONS_LEFT, oMotion_Active_Right => "DB2040_WINCC_HMI_LINES".SERVICES[2].WINCC_LINE_ACTIVE_RIGHT, oMotion_Active_Left => "DB2040_WINCC_HMI_LINES".SERVICES[2].WINCC_LINE_ACTIVE_LEFT, oLimit_right => "DB2040_WINCC_HMI_LINES".SERVICES[2].WINCC_LINE_STATUS_1_RIGHT, oLimit_left => "DB2040_WINCC_HMI_LINES".SERVICES[2].WINCC_LINE_STATUS_1_LEFT, oALARM_MISMATCH_FAULT => "DB426_ALARMS_WARNINGS".CLADDING_POWDER_FEEDER."718000", oALARM_FEEDER_PROFINET_MODE_FAULT => "DB426_ALARMS_WARNINGS".CLADDING_POWDER_FEEDER."718001")
   END_RUNG
   // the same network as SCL:
   "DB21010_POWDER_FEEDER_1_GENERAL_UNIT_01"(iOPERATION_MODE_LINE_1 := "DB21002_POWDER_FEEDER_OERLIKON_INTERLOCK".POWDER_FEEDER_1_UNIT_01.Inputs.i_uiOperationMode_Line1,   // "FB21011_POWDER_FEEDER_GENERAL"
                           iOPERATION_MODE_LINE_2 := "DB21002_POWDER_FEEDER_OERLIKON_INTERLOCK".POWDER_FEEDER_1_UNIT_01.Inputs.i_uiOperationMode_Line2,
                           iOPERATION_MODE_MATCHED_LINE_1 := "DB21002_POWDER_FEEDER_OERLIKON_INTERLOCK".POWDER_FEEDER_1_UNIT_01.Inputs.i_fOperationModeMatched_Line1,
                           iOPERATION_MODE_MATCHED_LINE_2 := "DB21002_POWDER_FEEDER_OERLIKON_INTERLOCK".POWDER_FEEDER_1_UNIT_01.Inputs.i_fOperationModeMatched_Line2,
                           iFEEDER_STATE_LINE_1 := "DB21002_POWDER_FEEDER_OERLIKON_INTERLOCK".POWDER_FEEDER_1_UNIT_01.Inputs.i_uiFeederState_Line1,
                           iFEEDER_STATE_LINE_2 := "DB21002_POWDER_FEEDER_OERLIKON_INTERLOCK".POWDER_FEEDER_1_UNIT_01.Inputs.i_uiFeederState_Line2,
                           iCARRIERGAS_STATUS_LINE_1 := "DB21002_POWDER_FEEDER_OERLIKON_INTERLOCK".POWDER_FEEDER_1_UNIT_01.Inputs.i_fCarriergasStatus_Line1,
                           iCARRIERGAS_STATUS_LINE_2 := "DB21002_POWDER_FEEDER_OERLIKON_INTERLOCK".POWDER_FEEDER_1_UNIT_01.Inputs.i_fCarriergasStatus_Line2,
                           oOPERATION_MODE => "DB21002_POWDER_FEEDER_OERLIKON_INTERLOCK".POWDER_FEEDER_1_UNIT_01.Outputs.o_uiOperationMode,
                           oPRODUCTION_MODE => "DB21002_POWDER_FEEDER_OERLIKON_INTERLOCK".POWDER_FEEDER_1_UNIT_01.Outputs.o_uiProductionMode,
                           oSYSTEM_MODE => "DB21002_POWDER_FEEDER_OERLIKON_INTERLOCK".POWDER_FEEDER_1_UNIT_01.Outputs.o_uiSystemMode,
                           oSwitchoncondition_on => "DB2040_WINCC_HMI_LINES".SERVICES[2].WINCC_LINE_CONDITIONS_RIGHT,
                           oSwitchoncondition_off => "DB2040_WINCC_HMI_LINES".SERVICES[2].WINCC_LINE_CONDITIONS_LEFT,
                           oMotion_Active_Right => "DB2040_WINCC_HMI_LINES".SERVICES[2].WINCC_LINE_ACTIVE_RIGHT,
                           oMotion_Active_Left => "DB2040_WINCC_HMI_LINES".SERVICES[2].WINCC_LINE_ACTIVE_LEFT,
                           oLimit_right => "DB2040_WINCC_HMI_LINES".SERVICES[2].WINCC_LINE_STATUS_1_RIGHT,
                           oLimit_left => "DB2040_WINCC_HMI_LINES".SERVICES[2].WINCC_LINE_STATUS_1_LEFT,
                           oALARM_MISMATCH_FAULT => "DB426_ALARMS_WARNINGS".CLADDING_POWDER_FEEDER."718000",
                           oALARM_FEEDER_PROFINET_MODE_FAULT => "DB426_ALARMS_WARNINGS".CLADDING_POWDER_FEEDER."718001");
END_REGION

REGION Network 3: /////_UNIT_02_/////
END_REGION

REGION Network 4: CALL FB21011 POWDER FEEDER 1 GENERAL UNIT 02
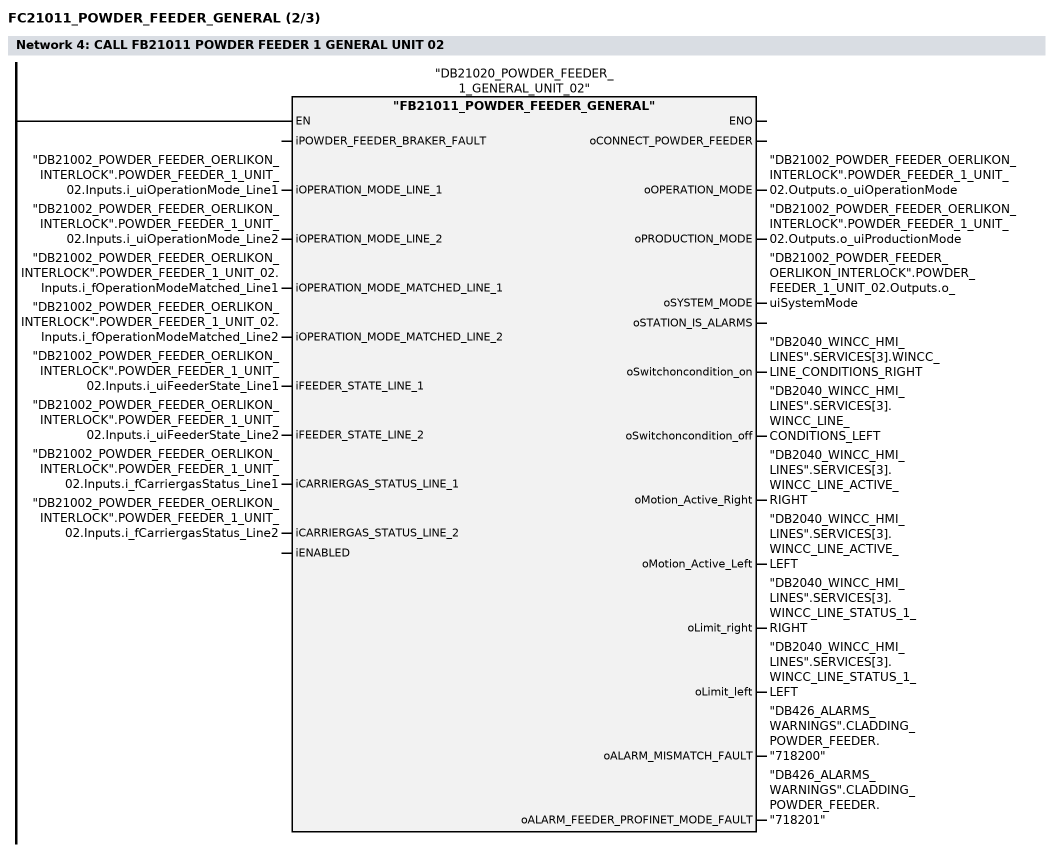
   RUNG wire#powerrail
      "DB21020_POWDER_FEEDER_1_GENERAL_UNIT_02"(iPOWDER_FEEDER_BRAKER_FAULT :=, iOPERATION_MODE_LINE_1 := "DB21002_POWDER_FEEDER_OERLIKON_INTERLOCK".POWDER_FEEDER_1_UNIT_02.Inputs.i_uiOperationMode_Line1, iOPERATION_MODE_LINE_2 := "DB21002_POWDER_FEEDER_OERLIKON_INTERLOCK".POWDER_FEEDER_1_UNIT_02.Inputs.i_uiOperationMode_Line2, iOPERATION_MODE_MATCHED_LINE_1 := "DB21002_POWDER_FEEDER_OERLIKON_INTERLOCK".POWDER_FEEDER_1_UNIT_02.Inputs.i_fOperationModeMatched_Line1, iOPERATION_MODE_MATCHED_LINE_2 := "DB21002_POWDER_FEEDER_OERLIKON_INTERLOCK".POWDER_FEEDER_1_UNIT_02.Inputs.i_fOperationModeMatched_Line2, iFEEDER_STATE_LINE_1 := "DB21002_POWDER_FEEDER_OERLIKON_INTERLOCK".POWDER_FEEDER_1_UNIT_02.Inputs.i_uiFeederState_Line1, iFEEDER_STATE_LINE_2 := "DB21002_POWDER_FEEDER_OERLIKON_INTERLOCK".POWDER_FEEDER_1_UNIT_02.Inputs.i_uiFeederState_Line2, iCARRIERGAS_STATUS_LINE_1 := "DB21002_POWDER_FEEDER_OERLIKON_INTERLOCK".POWDER_FEEDER_1_UNIT_02.Inputs.i_fCarriergasStatus_Line1, iCARRIERGAS_STATUS_LINE_2 := "DB21002_POWDER_FEEDER_OERLIKON_INTERLOCK".POWDER_FEEDER_1_UNIT_02.Inputs.i_fCarriergasStatus_Line2, iENABLED :=, oCONNECT_POWDER_FEEDER =>, oOPERATION_MODE => "DB21002_POWDER_FEEDER_OERLIKON_INTERLOCK".POWDER_FEEDER_1_UNIT_02.Outputs.o_uiOperationMode, oPRODUCTION_MODE => "DB21002_POWDER_FEEDER_OERLIKON_INTERLOCK".POWDER_FEEDER_1_UNIT_02.Outputs.o_uiProductionMode, oSYSTEM_MODE => "DB21002_POWDER_FEEDER_OERLIKON_INTERLOCK".POWDER_FEEDER_1_UNIT_02.Outputs.o_uiSystemMode, oSTATION_IS_ALARMS =>, oSwitchoncondition_on => "DB2040_WINCC_HMI_LINES".SERVICES[3].WINCC_LINE_CONDITIONS_RIGHT, oSwitchoncondition_off => "DB2040_WINCC_HMI_LINES".SERVICES[3].WINCC_LINE_CONDITIONS_LEFT, oMotion_Active_Right => "DB2040_WINCC_HMI_LINES".SERVICES[3].WINCC_LINE_ACTIVE_RIGHT, oMotion_Active_Left => "DB2040_WINCC_HMI_LINES".SERVICES[3].WINCC_LINE_ACTIVE_LEFT, oLimit_right => "DB2040_WINCC_HMI_LINES".SERVICES[3].WINCC_LINE_STATUS_1_RIGHT, oLimit_left => "DB2040_WINCC_HMI_LINES".SERVICES[3].WINCC_LINE_STATUS_1_LEFT, oALARM_MISMATCH_FAULT => "DB426_ALARMS_WARNINGS".CLADDING_POWDER_FEEDER."718200", oALARM_FEEDER_PROFINET_MODE_FAULT => "DB426_ALARMS_WARNINGS".CLADDING_POWDER_FEEDER."718201")
   END_RUNG
   // the same network as SCL:
   "DB21020_POWDER_FEEDER_1_GENERAL_UNIT_02"(iOPERATION_MODE_LINE_1 := "DB21002_POWDER_FEEDER_OERLIKON_INTERLOCK".POWDER_FEEDER_1_UNIT_02.Inputs.i_uiOperationMode_Line1,   // "FB21011_POWDER_FEEDER_GENERAL"
                           iOPERATION_MODE_LINE_2 := "DB21002_POWDER_FEEDER_OERLIKON_INTERLOCK".POWDER_FEEDER_1_UNIT_02.Inputs.i_uiOperationMode_Line2,
                           iOPERATION_MODE_MATCHED_LINE_1 := "DB21002_POWDER_FEEDER_OERLIKON_INTERLOCK".POWDER_FEEDER_1_UNIT_02.Inputs.i_fOperationModeMatched_Line1,
                           iOPERATION_MODE_MATCHED_LINE_2 := "DB21002_POWDER_FEEDER_OERLIKON_INTERLOCK".POWDER_FEEDER_1_UNIT_02.Inputs.i_fOperationModeMatched_Line2,
                           iFEEDER_STATE_LINE_1 := "DB21002_POWDER_FEEDER_OERLIKON_INTERLOCK".POWDER_FEEDER_1_UNIT_02.Inputs.i_uiFeederState_Line1,
                           iFEEDER_STATE_LINE_2 := "DB21002_POWDER_FEEDER_OERLIKON_INTERLOCK".POWDER_FEEDER_1_UNIT_02.Inputs.i_uiFeederState_Line2,
                           iCARRIERGAS_STATUS_LINE_1 := "DB21002_POWDER_FEEDER_OERLIKON_INTERLOCK".POWDER_FEEDER_1_UNIT_02.Inputs.i_fCarriergasStatus_Line1,
                           iCARRIERGAS_STATUS_LINE_2 := "DB21002_POWDER_FEEDER_OERLIKON_INTERLOCK".POWDER_FEEDER_1_UNIT_02.Inputs.i_fCarriergasStatus_Line2,
                           oOPERATION_MODE => "DB21002_POWDER_FEEDER_OERLIKON_INTERLOCK".POWDER_FEEDER_1_UNIT_02.Outputs.o_uiOperationMode,
                           oPRODUCTION_MODE => "DB21002_POWDER_FEEDER_OERLIKON_INTERLOCK".POWDER_FEEDER_1_UNIT_02.Outputs.o_uiProductionMode,
                           oSYSTEM_MODE => "DB21002_POWDER_FEEDER_OERLIKON_INTERLOCK".POWDER_FEEDER_1_UNIT_02.Outputs.o_uiSystemMode,
                           oSwitchoncondition_on => "DB2040_WINCC_HMI_LINES".SERVICES[3].WINCC_LINE_CONDITIONS_RIGHT,
                           oSwitchoncondition_off => "DB2040_WINCC_HMI_LINES".SERVICES[3].WINCC_LINE_CONDITIONS_LEFT,
                           oMotion_Active_Right => "DB2040_WINCC_HMI_LINES".SERVICES[3].WINCC_LINE_ACTIVE_RIGHT,
                           oMotion_Active_Left => "DB2040_WINCC_HMI_LINES".SERVICES[3].WINCC_LINE_ACTIVE_LEFT,
                           oLimit_right => "DB2040_WINCC_HMI_LINES".SERVICES[3].WINCC_LINE_STATUS_1_RIGHT,
                           oLimit_left => "DB2040_WINCC_HMI_LINES".SERVICES[3].WINCC_LINE_STATUS_1_LEFT,
                           oALARM_MISMATCH_FAULT => "DB426_ALARMS_WARNINGS".CLADDING_POWDER_FEEDER."718200",
                           oALARM_FEEDER_PROFINET_MODE_FAULT => "DB426_ALARMS_WARNINGS".CLADDING_POWDER_FEEDER."718201");
END_REGION

REGION Network 5: CALL FB21011 POWDER FEEDER 2 GENERAL UNIT 02
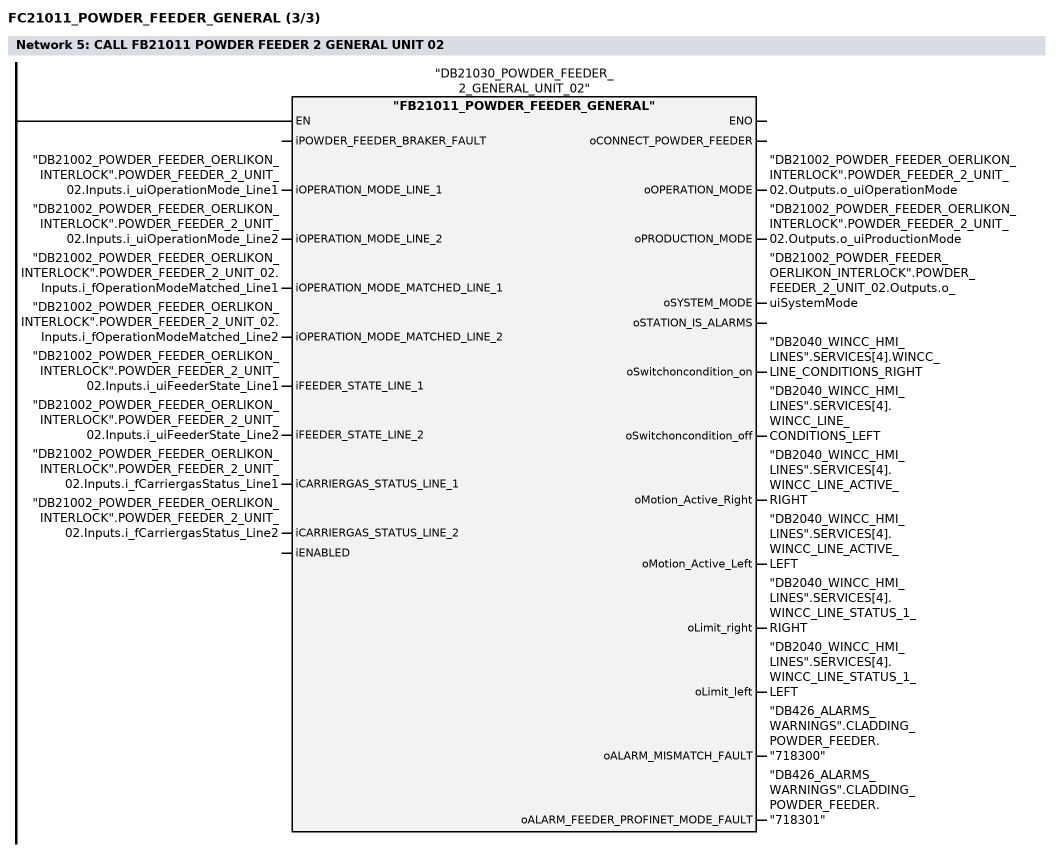
   RUNG wire#powerrail
      "DB21030_POWDER_FEEDER_2_GENERAL_UNIT_02"(iPOWDER_FEEDER_BRAKER_FAULT :=, iOPERATION_MODE_LINE_1 := "DB21002_POWDER_FEEDER_OERLIKON_INTERLOCK".POWDER_FEEDER_2_UNIT_02.Inputs.i_uiOperationMode_Line1, iOPERATION_MODE_LINE_2 := "DB21002_POWDER_FEEDER_OERLIKON_INTERLOCK".POWDER_FEEDER_2_UNIT_02.Inputs.i_uiOperationMode_Line2, iOPERATION_MODE_MATCHED_LINE_1 := "DB21002_POWDER_FEEDER_OERLIKON_INTERLOCK".POWDER_FEEDER_2_UNIT_02.Inputs.i_fOperationModeMatched_Line1, iOPERATION_MODE_MATCHED_LINE_2 := "DB21002_POWDER_FEEDER_OERLIKON_INTERLOCK".POWDER_FEEDER_2_UNIT_02.Inputs.i_fOperationModeMatched_Line2, iFEEDER_STATE_LINE_1 := "DB21002_POWDER_FEEDER_OERLIKON_INTERLOCK".POWDER_FEEDER_2_UNIT_02.Inputs.i_uiFeederState_Line1, iFEEDER_STATE_LINE_2 := "DB21002_POWDER_FEEDER_OERLIKON_INTERLOCK".POWDER_FEEDER_2_UNIT_02.Inputs.i_uiFeederState_Line2, iCARRIERGAS_STATUS_LINE_1 := "DB21002_POWDER_FEEDER_OERLIKON_INTERLOCK".POWDER_FEEDER_2_UNIT_02.Inputs.i_fCarriergasStatus_Line1, iCARRIERGAS_STATUS_LINE_2 := "DB21002_POWDER_FEEDER_OERLIKON_INTERLOCK".POWDER_FEEDER_2_UNIT_02.Inputs.i_fCarriergasStatus_Line2, iENABLED :=, oCONNECT_POWDER_FEEDER =>, oOPERATION_MODE => "DB21002_POWDER_FEEDER_OERLIKON_INTERLOCK".POWDER_FEEDER_2_UNIT_02.Outputs.o_uiOperationMode, oPRODUCTION_MODE => "DB21002_POWDER_FEEDER_OERLIKON_INTERLOCK".POWDER_FEEDER_2_UNIT_02.Outputs.o_uiProductionMode, oSYSTEM_MODE => "DB21002_POWDER_FEEDER_OERLIKON_INTERLOCK".POWDER_FEEDER_2_UNIT_02.Outputs.o_uiSystemMode, oSTATION_IS_ALARMS =>, oSwitchoncondition_on => "DB2040_WINCC_HMI_LINES".SERVICES[4].WINCC_LINE_CONDITIONS_RIGHT, oSwitchoncondition_off => "DB2040_WINCC_HMI_LINES".SERVICES[4].WINCC_LINE_CONDITIONS_LEFT, oMotion_Active_Right => "DB2040_WINCC_HMI_LINES".SERVICES[4].WINCC_LINE_ACTIVE_RIGHT, oMotion_Active_Left => "DB2040_WINCC_HMI_LINES".SERVICES[4].WINCC_LINE_ACTIVE_LEFT, oLimit_right => "DB2040_WINCC_HMI_LINES".SERVICES[4].WINCC_LINE_STATUS_1_RIGHT, oLimit_left => "DB2040_WINCC_HMI_LINES".SERVICES[4].WINCC_LINE_STATUS_1_LEFT, oALARM_MISMATCH_FAULT => "DB426_ALARMS_WARNINGS".CLADDING_POWDER_FEEDER."718300", oALARM_FEEDER_PROFINET_MODE_FAULT => "DB426_ALARMS_WARNINGS".CLADDING_POWDER_FEEDER."718301")
   END_RUNG
   // the same network as SCL:
   "DB21030_POWDER_FEEDER_2_GENERAL_UNIT_02"(iOPERATION_MODE_LINE_1 := "DB21002_POWDER_FEEDER_OERLIKON_INTERLOCK".POWDER_FEEDER_2_UNIT_02.Inputs.i_uiOperationMode_Line1,   // "FB21011_POWDER_FEEDER_GENERAL"
                           iOPERATION_MODE_LINE_2 := "DB21002_POWDER_FEEDER_OERLIKON_INTERLOCK".POWDER_FEEDER_2_UNIT_02.Inputs.i_uiOperationMode_Line2,
                           iOPERATION_MODE_MATCHED_LINE_1 := "DB21002_POWDER_FEEDER_OERLIKON_INTERLOCK".POWDER_FEEDER_2_UNIT_02.Inputs.i_fOperationModeMatched_Line1,
                           iOPERATION_MODE_MATCHED_LINE_2 := "DB21002_POWDER_FEEDER_OERLIKON_INTERLOCK".POWDER_FEEDER_2_UNIT_02.Inputs.i_fOperationModeMatched_Line2,
                           iFEEDER_STATE_LINE_1 := "DB21002_POWDER_FEEDER_OERLIKON_INTERLOCK".POWDER_FEEDER_2_UNIT_02.Inputs.i_uiFeederState_Line1,
                           iFEEDER_STATE_LINE_2 := "DB21002_POWDER_FEEDER_OERLIKON_INTERLOCK".POWDER_FEEDER_2_UNIT_02.Inputs.i_uiFeederState_Line2,
                           iCARRIERGAS_STATUS_LINE_1 := "DB21002_POWDER_FEEDER_OERLIKON_INTERLOCK".POWDER_FEEDER_2_UNIT_02.Inputs.i_fCarriergasStatus_Line1,
                           iCARRIERGAS_STATUS_LINE_2 := "DB21002_POWDER_FEEDER_OERLIKON_INTERLOCK".POWDER_FEEDER_2_UNIT_02.Inputs.i_fCarriergasStatus_Line2,
                           oOPERATION_MODE => "DB21002_POWDER_FEEDER_OERLIKON_INTERLOCK".POWDER_FEEDER_2_UNIT_02.Outputs.o_uiOperationMode,
                           oPRODUCTION_MODE => "DB21002_POWDER_FEEDER_OERLIKON_INTERLOCK".POWDER_FEEDER_2_UNIT_02.Outputs.o_uiProductionMode,
                           oSYSTEM_MODE => "DB21002_POWDER_FEEDER_OERLIKON_INTERLOCK".POWDER_FEEDER_2_UNIT_02.Outputs.o_uiSystemMode,
                           oSwitchoncondition_on => "DB2040_WINCC_HMI_LINES".SERVICES[4].WINCC_LINE_CONDITIONS_RIGHT,
                           oSwitchoncondition_off => "DB2040_WINCC_HMI_LINES".SERVICES[4].WINCC_LINE_CONDITIONS_LEFT,
                           oMotion_Active_Right => "DB2040_WINCC_HMI_LINES".SERVICES[4].WINCC_LINE_ACTIVE_RIGHT,
                           oMotion_Active_Left => "DB2040_WINCC_HMI_LINES".SERVICES[4].WINCC_LINE_ACTIVE_LEFT,
                           oLimit_right => "DB2040_WINCC_HMI_LINES".SERVICES[4].WINCC_LINE_STATUS_1_RIGHT,
                           oLimit_left => "DB2040_WINCC_HMI_LINES".SERVICES[4].WINCC_LINE_STATUS_1_LEFT,
                           oALARM_MISMATCH_FAULT => "DB426_ALARMS_WARNINGS".CLADDING_POWDER_FEEDER."718300",
                           oALARM_FEEDER_PROFINET_MODE_FAULT => "DB426_ALARMS_WARNINGS".CLADDING_POWDER_FEEDER."718301");
END_REGION
END_FUNCTION

FUNCTION_BLOCK "FB21011_POWDER_FEEDER_GENERAL"   // FB21011, LAD
TITLE = FB21011 POWDER FEEDER GENERAL
{ S7_Optimized_Access := 'TRUE' }
VERSION : 0.1
// stored: AutoNumber false, IsIECCheckEnabled false, IsRetainMemResEnabled false, MemoryReserve 100, SetENOAutomatically false, UDAEnableTagReadback false
   VAR_INPUT
      iPOWDER_FEEDER_BRAKER_FAULT : Bool;
      iOPERATION_MODE_LINE_1 : Word;
      iOPERATION_MODE_LINE_2 : Word;
      iOPERATION_MODE_MATCHED_LINE_1 : Bool;
      iOPERATION_MODE_MATCHED_LINE_2 : Bool;
      iFEEDER_STATE_LINE_1 : Word;
      iFEEDER_STATE_LINE_2 : Word;
      iCARRIERGAS_STATUS_LINE_1 : Bool;
      iCARRIERGAS_STATUS_LINE_2 : Bool;
      iENABLED : Bool;
   END_VAR
   VAR_OUTPUT
      oCONNECT_POWDER_FEEDER : Bool;
      oOPERATION_MODE : Word;
      oPRODUCTION_MODE : Word;
      oSYSTEM_MODE : Word;
      oSTATION_IS_ALARMS : Bool;
      oSwitchoncondition_on : Bool;
      oSwitchoncondition_off : Bool;
      oMotion_Active_Right : Bool;
      oMotion_Active_Left : Bool;
      oLimit_right : Bool;
      oLimit_left : Bool;
      oALARM_MISMATCH_FAULT : Bool;
      oALARM_FEEDER_PROFINET_MODE_FAULT : Bool;
   END_VAR
   VAR
      DATA : "POWDER FEEDER GENERAL";
      INPUT_SETTINGS : Struct
         UNIT_NUMBER : Int;
         FEEDER_NUMBER : Int;
      END_STRUCT;
   END_VAR
   VAR_TEMP
      OPTIONS_OFF : Bool;
      OPTIONS_ON : Bool;
      HOPPER_1 : Bool;
      HOPPER_2 : Bool;
      DB_NUMBER : DInt;
   END_VAR
   VAR_TEMP   // added for the SCL form of the ladder/FBD networks
      _w1 : Bool;
   END_VAR
BEGIN

NETWORK
TITLE = READ INSTANCE DB NUMBER
      L     DINO;
      +     10#800000;
      T     #DB_NUMBER;

REGION Network 2: OPTIONS OFF / Options Off
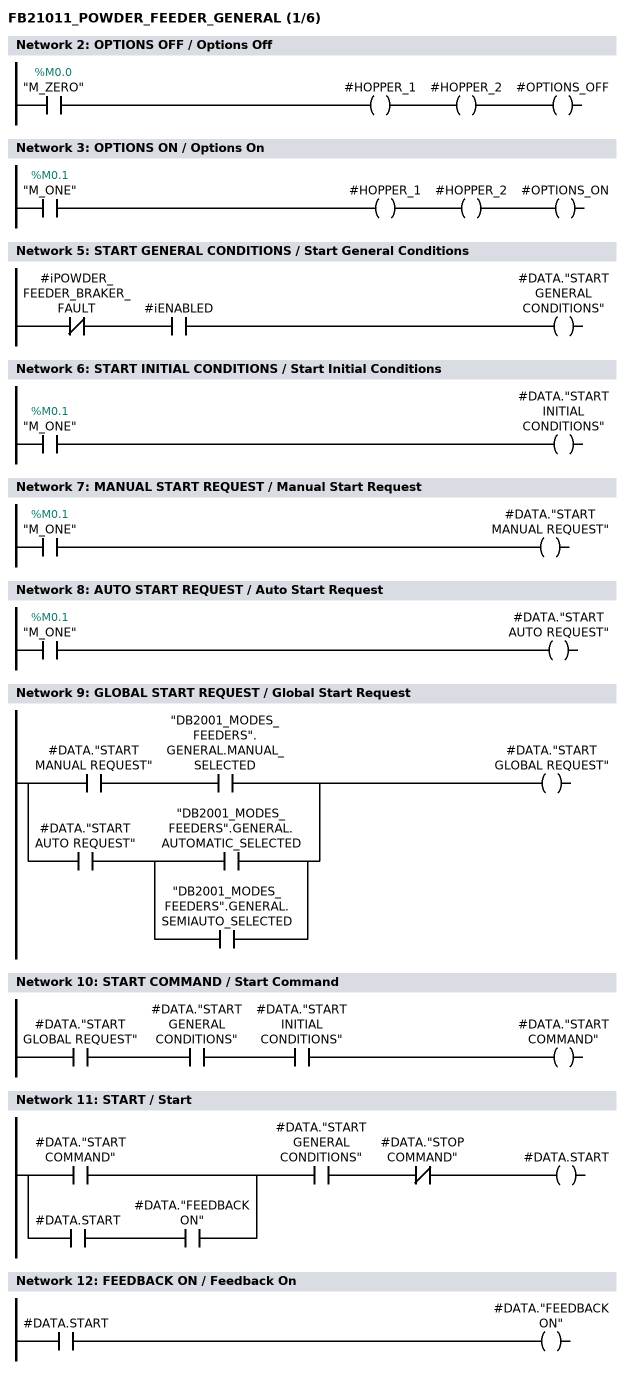
   RUNG wire#powerrail
      Contact( "M_ZERO" )
      Coil( #HOPPER_1 )
      Coil( #HOPPER_2 )
      Coil( #OPTIONS_OFF )
   END_RUNG
   // the same network as SCL:
   #HOPPER_1 := "M_ZERO";
   #HOPPER_2 := "M_ZERO";
   #OPTIONS_OFF := "M_ZERO";
END_REGION

REGION Network 3: OPTIONS ON / Options On
   RUNG wire#powerrail
      Contact( "M_ONE" )
      Coil( #HOPPER_1 )
      Coil( #HOPPER_2 )
      Coil( #OPTIONS_ON )
   END_RUNG
   // the same network as SCL:
   #HOPPER_1 := "M_ONE";
   #HOPPER_2 := "M_ONE";
   #OPTIONS_ON := "M_ONE";
END_REGION

REGION Network 4: INPUT / Input
END_REGION

REGION Network 5: START GENERAL CONDITIONS / Start General Conditions
   RUNG wire#powerrail
      I_Contact( #iPOWDER_FEEDER_BRAKER_FAULT )
      Contact( #iENABLED )
      Coil( #DATA."START GENERAL CONDITIONS" )
   END_RUNG
   // the same network as SCL:
   #DATA."START GENERAL CONDITIONS" := NOT #iPOWDER_FEEDER_BRAKER_FAULT AND #iENABLED;
END_REGION

REGION Network 6: START INITIAL CONDITIONS / Start Initial Conditions
   RUNG wire#powerrail
      Contact( "M_ONE" )
      Coil( #DATA."START INITIAL CONDITIONS" )
   END_RUNG
   // the same network as SCL:
   #DATA."START INITIAL CONDITIONS" := "M_ONE";
END_REGION

REGION Network 7: MANUAL START REQUEST / Manual Start Request
   RUNG wire#powerrail
      Contact( "M_ONE" )
      Coil( #DATA."START MANUAL REQUEST" )
   END_RUNG
   // the same network as SCL:
   #DATA."START MANUAL REQUEST" := "M_ONE";
END_REGION

REGION Network 8: AUTO START REQUEST / Auto Start Request
   RUNG wire#powerrail
      Contact( "M_ONE" )
      Coil( #DATA."START AUTO REQUEST" )
   END_RUNG
   // the same network as SCL:
   #DATA."START AUTO REQUEST" := "M_ONE";
END_REGION

REGION Network 9: GLOBAL START REQUEST / Global Start Request
   RUNG wire#powerrail
      Contact( #DATA."START MANUAL REQUEST" )
      Contact( "DB2001_MODES_FEEDERS".GENERAL.MANUAL_SELECTED )
      wire#w1
      Coil( #DATA."START GLOBAL REQUEST" )
   END_RUNG
   RUNG wire#powerrail
      Contact( #DATA."START AUTO REQUEST" )
      wire#w2
      Contact( "DB2001_MODES_FEEDERS".GENERAL.AUTOMATIC_SELECTED )
   END_RUNG wire#w1
   RUNG wire#w2
      Contact( "DB2001_MODES_FEEDERS".GENERAL.SEMIAUTO_SELECTED )
   END_RUNG wire#w1
   // the same network as SCL:
   #DATA."START GLOBAL REQUEST" := (#DATA."START MANUAL REQUEST" AND "DB2001_MODES_FEEDERS".GENERAL.MANUAL_SELECTED) OR (#DATA."START AUTO REQUEST" AND ("DB2001_MODES_FEEDERS".GENERAL.AUTOMATIC_SELECTED OR "DB2001_MODES_FEEDERS".GENERAL.SEMIAUTO_SELECTED));
END_REGION

REGION Network 10: START COMMAND / Start Command
   RUNG wire#powerrail
      Contact( #DATA."START GLOBAL REQUEST" )
      Contact( #DATA."START GENERAL CONDITIONS" )
      Contact( #DATA."START INITIAL CONDITIONS" )
      Coil( #DATA."START COMMAND" )
   END_RUNG
   // the same network as SCL:
   #DATA."START COMMAND" := #DATA."START GLOBAL REQUEST" AND #DATA."START GENERAL CONDITIONS" AND #DATA."START INITIAL CONDITIONS";
END_REGION

REGION Network 11: START / Start
   RUNG wire#powerrail
      Contact( #DATA."START COMMAND" )
      wire#w1
      Contact( #DATA."START GENERAL CONDITIONS" )
      I_Contact( #DATA."STOP COMMAND" )
      Coil( #DATA.START )
   END_RUNG
   RUNG wire#powerrail
      Contact( #DATA.START )
      Contact( #DATA."FEEDBACK ON" )
   END_RUNG wire#w1
   // the same network as SCL:
   #DATA.START := (#DATA."START COMMAND" OR (#DATA.START AND #DATA."FEEDBACK ON")) AND #DATA."START GENERAL CONDITIONS" AND NOT #DATA."STOP COMMAND";
END_REGION

REGION Network 12: FEEDBACK ON / Feedback On
   RUNG wire#powerrail
      Contact( #DATA.START )
      Coil( #DATA."FEEDBACK ON" )
   END_RUNG
   // the same network as SCL:
   #DATA."FEEDBACK ON" := #DATA.START;
END_REGION

REGION Network 13: STOP GENERAL CONDITIONS / Stop General Conditions
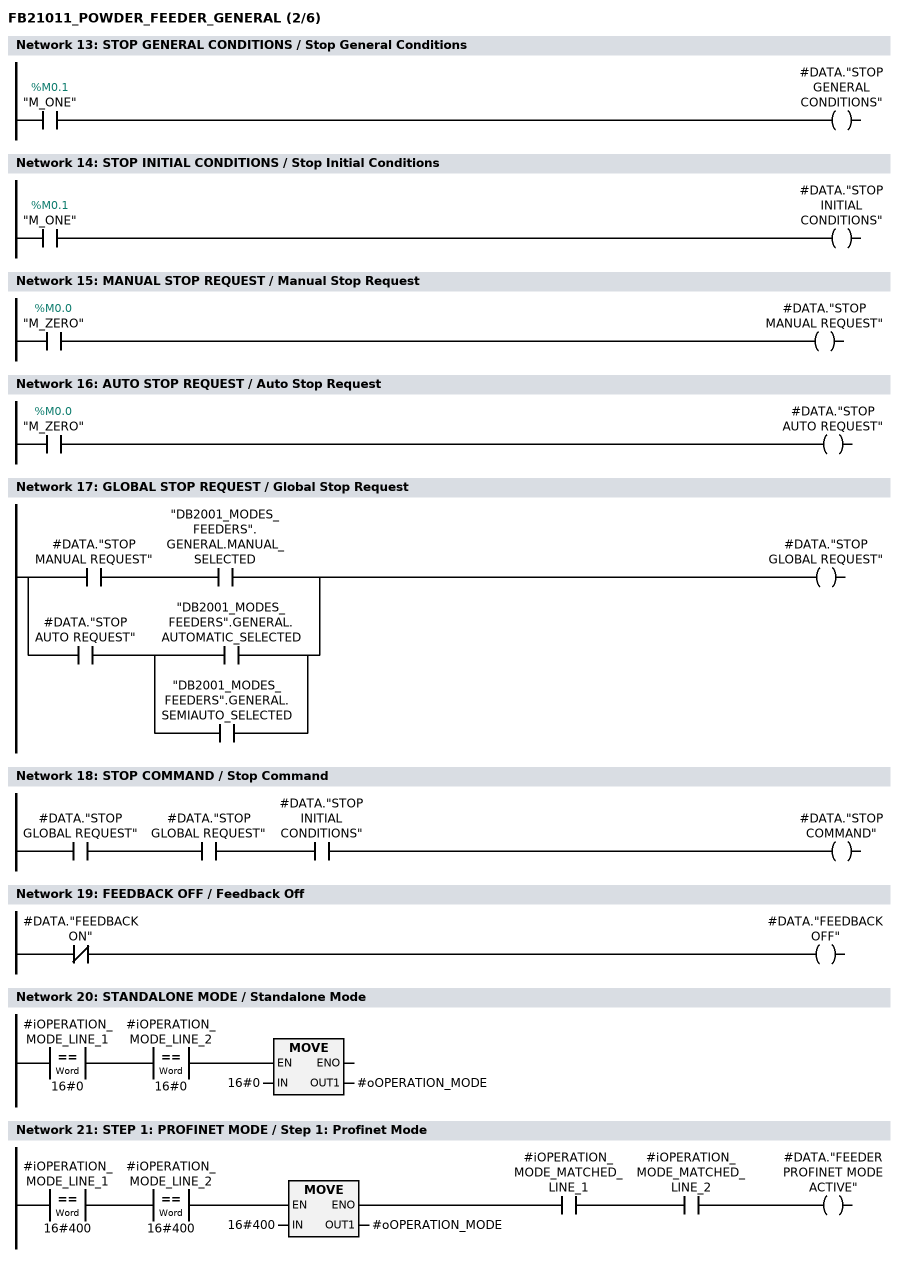
   RUNG wire#powerrail
      Contact( "M_ONE" )
      Coil( #DATA."STOP GENERAL CONDITIONS" )
   END_RUNG
   // the same network as SCL:
   #DATA."STOP GENERAL CONDITIONS" := "M_ONE";
END_REGION

REGION Network 14: STOP INITIAL CONDITIONS / Stop Initial Conditions
   RUNG wire#powerrail
      Contact( "M_ONE" )
      Coil( #DATA."STOP INITIAL CONDITIONS" )
   END_RUNG
   // the same network as SCL:
   #DATA."STOP INITIAL CONDITIONS" := "M_ONE";
END_REGION

REGION Network 15: MANUAL STOP REQUEST / Manual Stop Request
   RUNG wire#powerrail
      Contact( "M_ZERO" )
      Coil( #DATA."STOP MANUAL REQUEST" )
   END_RUNG
   // the same network as SCL:
   #DATA."STOP MANUAL REQUEST" := "M_ZERO";
END_REGION

REGION Network 16: AUTO STOP REQUEST / Auto Stop Request
   RUNG wire#powerrail
      Contact( "M_ZERO" )
      Coil( #DATA."STOP AUTO REQUEST" )
   END_RUNG
   // the same network as SCL:
   #DATA."STOP AUTO REQUEST" := "M_ZERO";
END_REGION

REGION Network 17: GLOBAL STOP REQUEST / Global Stop Request
   RUNG wire#powerrail
      Contact( #DATA."STOP MANUAL REQUEST" )
      Contact( "DB2001_MODES_FEEDERS".GENERAL.MANUAL_SELECTED )
      wire#w1
      Coil( #DATA."STOP GLOBAL REQUEST" )
   END_RUNG
   RUNG wire#powerrail
      Contact( #DATA."STOP AUTO REQUEST" )
      wire#w2
      Contact( "DB2001_MODES_FEEDERS".GENERAL.AUTOMATIC_SELECTED )
   END_RUNG wire#w1
   RUNG wire#w2
      Contact( "DB2001_MODES_FEEDERS".GENERAL.SEMIAUTO_SELECTED )
   END_RUNG wire#w1
   // the same network as SCL:
   #DATA."STOP GLOBAL REQUEST" := (#DATA."STOP MANUAL REQUEST" AND "DB2001_MODES_FEEDERS".GENERAL.MANUAL_SELECTED) OR (#DATA."STOP AUTO REQUEST" AND ("DB2001_MODES_FEEDERS".GENERAL.AUTOMATIC_SELECTED OR "DB2001_MODES_FEEDERS".GENERAL.SEMIAUTO_SELECTED));
END_REGION

REGION Network 18: STOP COMMAND / Stop Command
   RUNG wire#powerrail
      Contact( #DATA."STOP GLOBAL REQUEST" )
      Contact( #DATA."STOP GLOBAL REQUEST" )
      Contact( #DATA."STOP INITIAL CONDITIONS" )
      Coil( #DATA."STOP COMMAND" )
   END_RUNG
   // the same network as SCL:
   #DATA."STOP COMMAND" := #DATA."STOP GLOBAL REQUEST" AND #DATA."STOP GLOBAL REQUEST" AND #DATA."STOP INITIAL CONDITIONS";
END_REGION

REGION Network 19: FEEDBACK OFF / Feedback Off
   RUNG wire#powerrail
      I_Contact( #DATA."FEEDBACK ON" )
      Coil( #DATA."FEEDBACK OFF" )
   END_RUNG
   // the same network as SCL:
   #DATA."FEEDBACK OFF" := NOT #DATA."FEEDBACK ON";
END_REGION

REGION Network 20: STANDALONE MODE / Standalone Mode
   RUNG wire#powerrail
      { S7_Templates := "SrcType := Word" } EQ_Contact(in1 := #iOPERATION_MODE_LINE_1, in2 := 16#0)
      { S7_Templates := "SrcType := Word" } EQ_Contact(in1 := #iOPERATION_MODE_LINE_2, in2 := 16#0)
      Move(in := 16#0, out1 => #oOPERATION_MODE)
   END_RUNG
   // the same network as SCL:
   IF (#iOPERATION_MODE_LINE_1 = 16#0) AND (#iOPERATION_MODE_LINE_2 = 16#0) THEN
       #oOPERATION_MODE := 16#0;
   END_IF;
END_REGION

REGION Network 21: STEP 1: PROFINET MODE / Step 1: Profinet Mode
   RUNG wire#powerrail
      { S7_Templates := "SrcType := Word" } EQ_Contact(in1 := #iOPERATION_MODE_LINE_1, in2 := 16#400)
      { S7_Templates := "SrcType := Word" } EQ_Contact(in1 := #iOPERATION_MODE_LINE_2, in2 := 16#400)
      Move(in := 16#400, out1 => #oOPERATION_MODE)
      Contact( #iOPERATION_MODE_MATCHED_LINE_1 )
      Contact( #iOPERATION_MODE_MATCHED_LINE_2 )
      Coil( #DATA."FEEDER PROFINET MODE ACTIVE" )
   END_RUNG
   // the same network as SCL:
   #_w1 := (#iOPERATION_MODE_LINE_1 = 16#400) AND (#iOPERATION_MODE_LINE_2 = 16#400);
   IF #_w1 THEN #oOPERATION_MODE := 16#400; END_IF;
   #DATA."FEEDER PROFINET MODE ACTIVE" := #_w1 AND #iOPERATION_MODE_MATCHED_LINE_1 AND #iOPERATION_MODE_MATCHED_LINE_2;
END_REGION

REGION Network 22: STEP 2: PRODUCTION MODE / Step 2: Production Mode
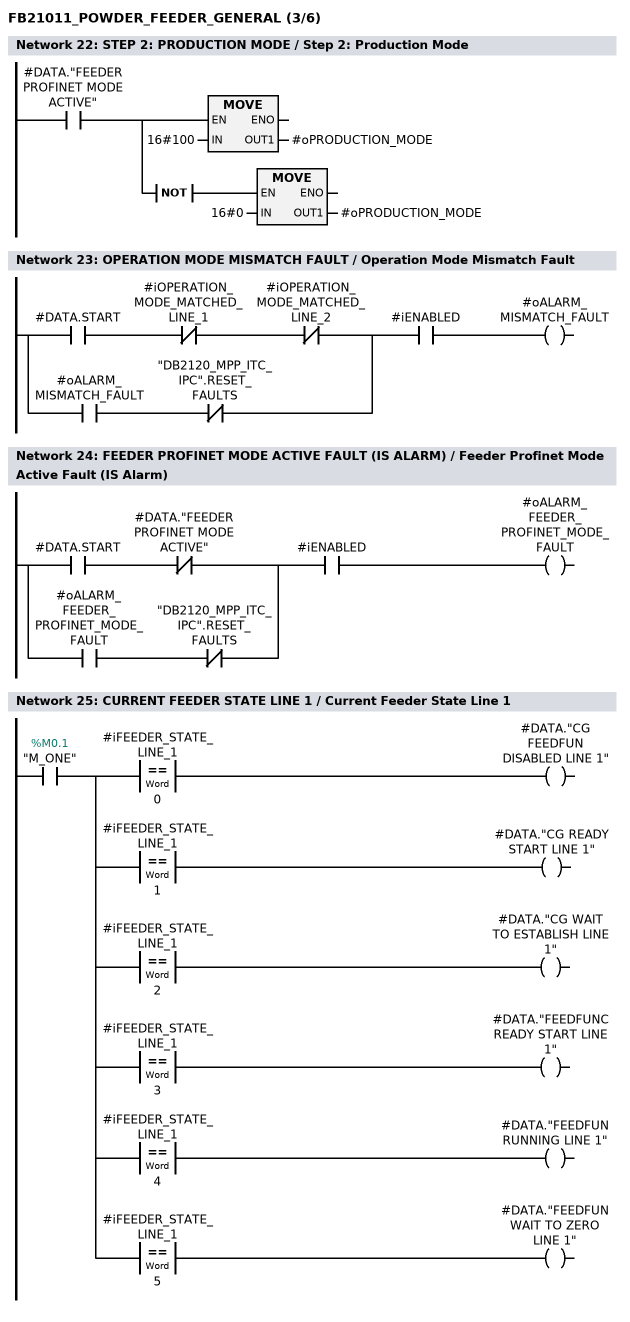
   RUNG wire#powerrail
      Contact( #DATA."FEEDER PROFINET MODE ACTIVE" )
      wire#w1
      Move(in := 16#100, out1 => #oPRODUCTION_MODE)
   END_RUNG
   RUNG wire#w1
      Not()
      Move(in := 16#0, out1 => #oPRODUCTION_MODE)
   END_RUNG
   // the same network as SCL:
   IF #DATA."FEEDER PROFINET MODE ACTIVE" THEN #oPRODUCTION_MODE := 16#100; END_IF;
   IF NOT #DATA."FEEDER PROFINET MODE ACTIVE" THEN #oPRODUCTION_MODE := 16#0; END_IF;
END_REGION

REGION Network 23: OPERATION MODE MISMATCH FAULT / Operation Mode Mismatch Fault
   RUNG wire#powerrail
      Contact( #DATA.START )
      I_Contact( #iOPERATION_MODE_MATCHED_LINE_1 )
      I_Contact( #iOPERATION_MODE_MATCHED_LINE_2 )
      wire#w1
      Contact( #iENABLED )
      Coil( #oALARM_MISMATCH_FAULT )
   END_RUNG
   RUNG wire#powerrail
      Contact( #oALARM_MISMATCH_FAULT )
      I_Contact( "DB2120_MPP_ITC_IPC".RESET_FAULTS )
   END_RUNG wire#w1
   // the same network as SCL:
   #oALARM_MISMATCH_FAULT := ((#DATA.START AND NOT #iOPERATION_MODE_MATCHED_LINE_1 AND NOT #iOPERATION_MODE_MATCHED_LINE_2) OR (#oALARM_MISMATCH_FAULT AND NOT "DB2120_MPP_ITC_IPC".RESET_FAULTS)) AND #iENABLED;
END_REGION

REGION Network 24: FEEDER PROFINET MODE ACTIVE FAULT (IS ALARM) / Feeder Profinet Mode Active Fault (IS Alarm)
   RUNG wire#powerrail
      Contact( #DATA.START )
      I_Contact( #DATA."FEEDER PROFINET MODE ACTIVE" )
      wire#w1
      Contact( #iENABLED )
      Coil( #oALARM_FEEDER_PROFINET_MODE_FAULT )
   END_RUNG
   RUNG wire#powerrail
      Contact( #oALARM_FEEDER_PROFINET_MODE_FAULT )
      I_Contact( "DB2120_MPP_ITC_IPC".RESET_FAULTS )
   END_RUNG wire#w1
   // the same network as SCL:
   #oALARM_FEEDER_PROFINET_MODE_FAULT := ((#DATA.START AND NOT #DATA."FEEDER PROFINET MODE ACTIVE") OR (#oALARM_FEEDER_PROFINET_MODE_FAULT AND NOT "DB2120_MPP_ITC_IPC".RESET_FAULTS)) AND #iENABLED;
END_REGION

REGION Network 25: CURRENT FEEDER STATE LINE 1 / Current Feeder State Line 1
   RUNG wire#powerrail
      Contact( "M_ONE" )
      wire#w1
      { S7_Templates := "SrcType := Word" } EQ_Contact(in1 := #iFEEDER_STATE_LINE_1, in2 := 0)
      Coil( #DATA."CG FEEDFUN DISABLED LINE 1" )
   END_RUNG
   RUNG wire#w1
      { S7_Templates := "SrcType := Word" } EQ_Contact(in1 := #iFEEDER_STATE_LINE_1, in2 := 1)
      Coil( #DATA."CG READY START LINE 1" )
   END_RUNG
   RUNG wire#w1
      { S7_Templates := "SrcType := Word" } EQ_Contact(in1 := #iFEEDER_STATE_LINE_1, in2 := 2)
      Coil( #DATA."CG WAIT TO ESTABLISH LINE 1" )
   END_RUNG
   RUNG wire#w1
      { S7_Templates := "SrcType := Word" } EQ_Contact(in1 := #iFEEDER_STATE_LINE_1, in2 := 3)
      Coil( #DATA."FEEDFUNC READY START LINE 1" )
   END_RUNG
   RUNG wire#w1
      { S7_Templates := "SrcType := Word" } EQ_Contact(in1 := #iFEEDER_STATE_LINE_1, in2 := 4)
      Coil( #DATA."FEEDFUN RUNNING LINE 1" )
   END_RUNG
   RUNG wire#w1
      { S7_Templates := "SrcType := Word" } EQ_Contact(in1 := #iFEEDER_STATE_LINE_1, in2 := 5)
      Coil( #DATA."FEEDFUN WAIT TO ZERO LINE 1" )
   END_RUNG
   // the same network as SCL:
   #DATA."CG FEEDFUN DISABLED LINE 1" := "M_ONE" AND (#iFEEDER_STATE_LINE_1 = 0);
   #DATA."CG READY START LINE 1" := "M_ONE" AND (#iFEEDER_STATE_LINE_1 = 1);
   #DATA."CG WAIT TO ESTABLISH LINE 1" := "M_ONE" AND (#iFEEDER_STATE_LINE_1 = 2);
   #DATA."FEEDFUNC READY START LINE 1" := "M_ONE" AND (#iFEEDER_STATE_LINE_1 = 3);
   #DATA."FEEDFUN RUNNING LINE 1" := "M_ONE" AND (#iFEEDER_STATE_LINE_1 = 4);
   #DATA."FEEDFUN WAIT TO ZERO LINE 1" := "M_ONE" AND (#iFEEDER_STATE_LINE_1 = 5);
END_REGION

REGION Network 26: CURRENT FEEDER STATE LINE 2 / Current Feeder State Line 2
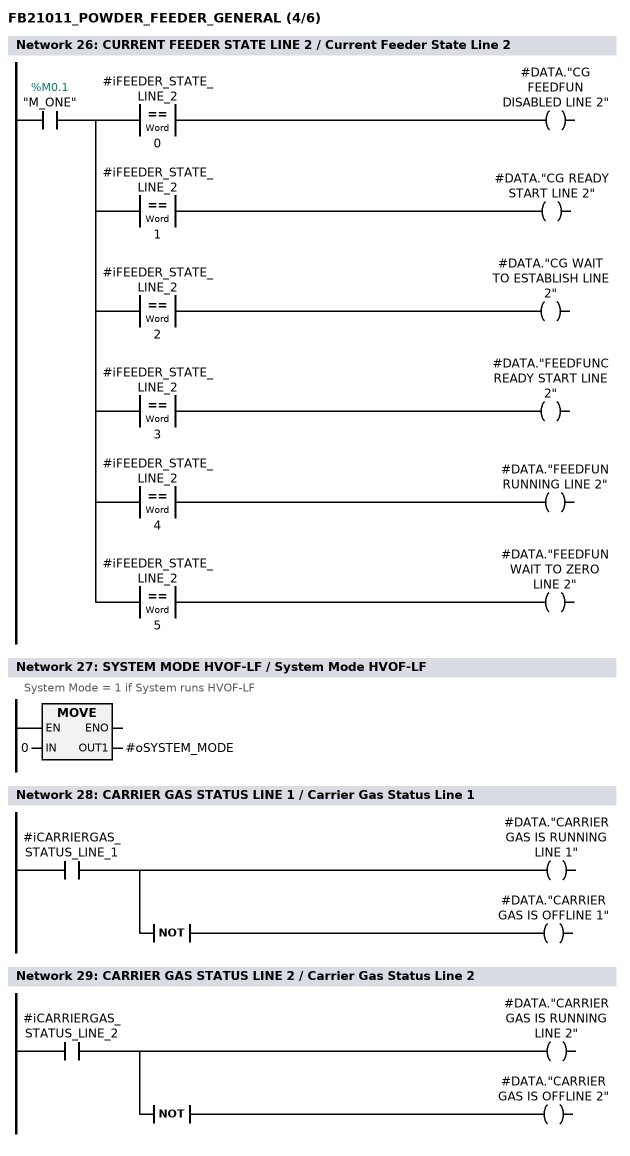
   RUNG wire#powerrail
      Contact( "M_ONE" )
      wire#w1
      { S7_Templates := "SrcType := Word" } EQ_Contact(in1 := #iFEEDER_STATE_LINE_2, in2 := 0)
      Coil( #DATA."CG FEEDFUN DISABLED LINE 2" )
   END_RUNG
   RUNG wire#w1
      { S7_Templates := "SrcType := Word" } EQ_Contact(in1 := #iFEEDER_STATE_LINE_2, in2 := 1)
      Coil( #DATA."CG READY START LINE 2" )
   END_RUNG
   RUNG wire#w1
      { S7_Templates := "SrcType := Word" } EQ_Contact(in1 := #iFEEDER_STATE_LINE_2, in2 := 2)
      Coil( #DATA."CG WAIT TO ESTABLISH LINE 2" )
   END_RUNG
   RUNG wire#w1
      { S7_Templates := "SrcType := Word" } EQ_Contact(in1 := #iFEEDER_STATE_LINE_2, in2 := 3)
      Coil( #DATA."FEEDFUNC READY START LINE 2" )
   END_RUNG
   RUNG wire#w1
      { S7_Templates := "SrcType := Word" } EQ_Contact(in1 := #iFEEDER_STATE_LINE_2, in2 := 4)
      Coil( #DATA."FEEDFUN RUNNING LINE 2" )
   END_RUNG
   RUNG wire#w1
      { S7_Templates := "SrcType := Word" } EQ_Contact(in1 := #iFEEDER_STATE_LINE_2, in2 := 5)
      Coil( #DATA."FEEDFUN WAIT TO ZERO LINE 2" )
   END_RUNG
   // the same network as SCL:
   #DATA."CG FEEDFUN DISABLED LINE 2" := "M_ONE" AND (#iFEEDER_STATE_LINE_2 = 0);
   #DATA."CG READY START LINE 2" := "M_ONE" AND (#iFEEDER_STATE_LINE_2 = 1);
   #DATA."CG WAIT TO ESTABLISH LINE 2" := "M_ONE" AND (#iFEEDER_STATE_LINE_2 = 2);
   #DATA."FEEDFUNC READY START LINE 2" := "M_ONE" AND (#iFEEDER_STATE_LINE_2 = 3);
   #DATA."FEEDFUN RUNNING LINE 2" := "M_ONE" AND (#iFEEDER_STATE_LINE_2 = 4);
   #DATA."FEEDFUN WAIT TO ZERO LINE 2" := "M_ONE" AND (#iFEEDER_STATE_LINE_2 = 5);
END_REGION

REGION Network 27: SYSTEM MODE HVOF-LF / System Mode HVOF-LF
   // System Mode = 1 if System runs HVOF-LF
   RUNG wire#powerrail
      Move(in := 0, out1 => #oSYSTEM_MODE)
   END_RUNG
   // the same network as SCL:
   #oSYSTEM_MODE := 0;
END_REGION

REGION Network 28: CARRIER GAS STATUS LINE 1 / Carrier Gas Status Line 1
   RUNG wire#powerrail
      Contact( #iCARRIERGAS_STATUS_LINE_1 )
      wire#w1
      Coil( #DATA."CARRIER GAS IS RUNNING LINE 1" )
   END_RUNG
   RUNG wire#w1
      Not()
      Coil( #DATA."CARRIER GAS IS OFFLINE 1" )
   END_RUNG
   // the same network as SCL:
   #DATA."CARRIER GAS IS RUNNING LINE 1" := #iCARRIERGAS_STATUS_LINE_1;
   #DATA."CARRIER GAS IS OFFLINE 1" := NOT #iCARRIERGAS_STATUS_LINE_1;
END_REGION

REGION Network 29: CARRIER GAS STATUS LINE 2 / Carrier Gas Status Line 2
   RUNG wire#powerrail
      Contact( #iCARRIERGAS_STATUS_LINE_2 )
      wire#w1
      Coil( #DATA."CARRIER GAS IS RUNNING LINE 2" )
   END_RUNG
   RUNG wire#w1
      Not()
      Coil( #DATA."CARRIER GAS IS OFFLINE 2" )
   END_RUNG
   // the same network as SCL:
   #DATA."CARRIER GAS IS RUNNING LINE 2" := #iCARRIERGAS_STATUS_LINE_2;
   #DATA."CARRIER GAS IS OFFLINE 2" := NOT #iCARRIERGAS_STATUS_LINE_2;
END_REGION

REGION Network 30: INMEDIATE STOP ALARMS / Inmediate Stop Alarms
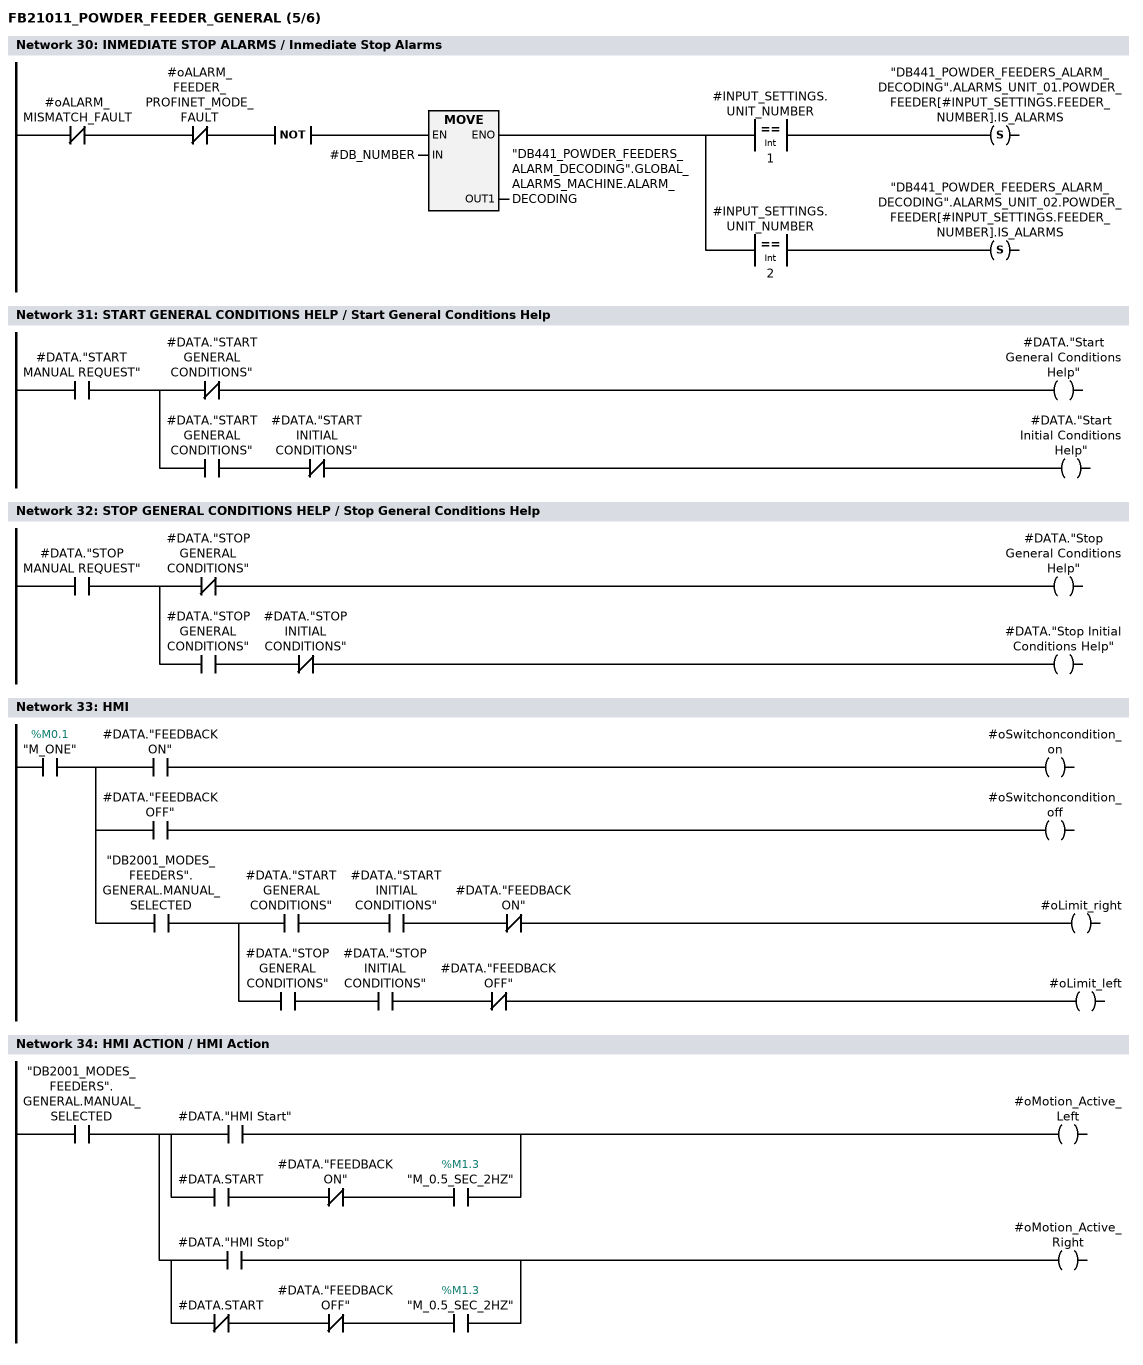
   RUNG wire#powerrail
      I_Contact( #oALARM_MISMATCH_FAULT )
      I_Contact( #oALARM_FEEDER_PROFINET_MODE_FAULT )
      Not()
      Move(in := #DB_NUMBER, out1 => "DB441_POWDER_FEEDERS_ALARM_DECODING".GLOBAL_ALARMS_MACHINE.ALARM_DECODING)
      wire#w1
      { S7_Templates := "SrcType := Int" } EQ_Contact(in1 := #INPUT_SETTINGS.UNIT_NUMBER, in2 := 1)
      S_Coil( "DB441_POWDER_FEEDERS_ALARM_DECODING".ALARMS_UNIT_01.POWDER_FEEDER[#INPUT_SETTINGS.FEEDER_NUMBER].IS_ALARMS )
   END_RUNG
   RUNG wire#w1
      { S7_Templates := "SrcType := Int" } EQ_Contact(in1 := #INPUT_SETTINGS.UNIT_NUMBER, in2 := 2)
      S_Coil( "DB441_POWDER_FEEDERS_ALARM_DECODING".ALARMS_UNIT_02.POWDER_FEEDER[#INPUT_SETTINGS.FEEDER_NUMBER].IS_ALARMS )
   END_RUNG
   // the same network as SCL:
   #_w1 := NOT (NOT #oALARM_MISMATCH_FAULT AND NOT #oALARM_FEEDER_PROFINET_MODE_FAULT);
   IF #_w1 THEN
       "DB441_POWDER_FEEDERS_ALARM_DECODING".GLOBAL_ALARMS_MACHINE.ALARM_DECODING := #DB_NUMBER;
   END_IF;
   IF #_w1 AND (#INPUT_SETTINGS.UNIT_NUMBER = 1) THEN
       "DB441_POWDER_FEEDERS_ALARM_DECODING".ALARMS_UNIT_01.POWDER_FEEDER[#INPUT_SETTINGS.FEEDER_NUMBER].IS_ALARMS := TRUE;
   END_IF;
   IF #_w1 AND (#INPUT_SETTINGS.UNIT_NUMBER = 2) THEN
       "DB441_POWDER_FEEDERS_ALARM_DECODING".ALARMS_UNIT_02.POWDER_FEEDER[#INPUT_SETTINGS.FEEDER_NUMBER].IS_ALARMS := TRUE;
   END_IF;
END_REGION

REGION Network 31: START GENERAL CONDITIONS HELP / Start General Conditions Help
   RUNG wire#powerrail
      Contact( #DATA."START MANUAL REQUEST" )
      wire#w1
      I_Contact( #DATA."START GENERAL CONDITIONS" )
      Coil( #DATA."Start General Conditions Help" )
   END_RUNG
   RUNG wire#w1
      Contact( #DATA."START GENERAL CONDITIONS" )
      I_Contact( #DATA."START INITIAL CONDITIONS" )
      Coil( #DATA."Start Initial Conditions Help" )
   END_RUNG
   // the same network as SCL:
   #DATA."Start General Conditions Help" := #DATA."START MANUAL REQUEST" AND NOT #DATA."START GENERAL CONDITIONS";
   #DATA."Start Initial Conditions Help" := #DATA."START MANUAL REQUEST" AND #DATA."START GENERAL CONDITIONS" AND NOT #DATA."START INITIAL CONDITIONS";
END_REGION

REGION Network 32: STOP GENERAL CONDITIONS HELP / Stop General Conditions Help
   RUNG wire#powerrail
      Contact( #DATA."STOP MANUAL REQUEST" )
      wire#w1
      I_Contact( #DATA."STOP GENERAL CONDITIONS" )
      Coil( #DATA."Stop General Conditions Help" )
   END_RUNG
   RUNG wire#w1
      Contact( #DATA."STOP GENERAL CONDITIONS" )
      I_Contact( #DATA."STOP INITIAL CONDITIONS" )
      Coil( #DATA."Stop Initial Conditions Help" )
   END_RUNG
   // the same network as SCL:
   #DATA."Stop General Conditions Help" := #DATA."STOP MANUAL REQUEST" AND NOT #DATA."STOP GENERAL CONDITIONS";
   #DATA."Stop Initial Conditions Help" := #DATA."STOP MANUAL REQUEST" AND #DATA."STOP GENERAL CONDITIONS" AND NOT #DATA."STOP INITIAL CONDITIONS";
END_REGION

REGION Network 33: HMI
   RUNG wire#powerrail
      Contact( "M_ONE" )
      wire#w1
      Contact( #DATA."FEEDBACK ON" )
      Coil( #oSwitchoncondition_on )
   END_RUNG
   RUNG wire#w1
      Contact( #DATA."FEEDBACK OFF" )
      Coil( #oSwitchoncondition_off )
   END_RUNG
   RUNG wire#w1
      Contact( "DB2001_MODES_FEEDERS".GENERAL.MANUAL_SELECTED )
      wire#w2
      Contact( #DATA."START GENERAL CONDITIONS" )
      Contact( #DATA."START INITIAL CONDITIONS" )
      I_Contact( #DATA."FEEDBACK ON" )
      Coil( #oLimit_right )
   END_RUNG
   RUNG wire#w2
      Contact( #DATA."STOP GENERAL CONDITIONS" )
      Contact( #DATA."STOP INITIAL CONDITIONS" )
      I_Contact( #DATA."FEEDBACK OFF" )
      Coil( #oLimit_left )
   END_RUNG
   // the same network as SCL:
   #oSwitchoncondition_on := "M_ONE" AND #DATA."FEEDBACK ON";
   #oSwitchoncondition_off := "M_ONE" AND #DATA."FEEDBACK OFF";
   #_w1 := "M_ONE" AND "DB2001_MODES_FEEDERS".GENERAL.MANUAL_SELECTED;
   #oLimit_right := #_w1 AND #DATA."START GENERAL CONDITIONS" AND #DATA."START INITIAL CONDITIONS" AND NOT #DATA."FEEDBACK ON";
   #oLimit_left := #_w1 AND #DATA."STOP GENERAL CONDITIONS" AND #DATA."STOP INITIAL CONDITIONS" AND NOT #DATA."FEEDBACK OFF";
END_REGION

REGION Network 34: HMI ACTION / HMI Action
   RUNG wire#powerrail
      Contact( "DB2001_MODES_FEEDERS".GENERAL.MANUAL_SELECTED )
      wire#w1
      Contact( #DATA."HMI Start" )
      wire#w2
      Coil( #oMotion_Active_Left )
   END_RUNG
   RUNG wire#w1
      Contact( #DATA.START )
      I_Contact( #DATA."FEEDBACK ON" )
      Contact( "M_0.5_SEC_2HZ" )
   END_RUNG wire#w2
   RUNG wire#w1
      Contact( #DATA."HMI Stop" )
      wire#w3
      Coil( #oMotion_Active_Right )
   END_RUNG
   RUNG wire#w1
      I_Contact( #DATA.START )
      I_Contact( #DATA."FEEDBACK OFF" )
      Contact( "M_0.5_SEC_2HZ" )
   END_RUNG wire#w3
   // the same network as SCL:
   #oMotion_Active_Left := "DB2001_MODES_FEEDERS".GENERAL.MANUAL_SELECTED AND (#DATA."HMI Start" OR (#DATA.START AND NOT #DATA."FEEDBACK ON" AND "M_0.5_SEC_2HZ"));
   #oMotion_Active_Right := "DB2001_MODES_FEEDERS".GENERAL.MANUAL_SELECTED AND (#DATA."HMI Stop" OR (NOT #DATA.START AND NOT #DATA."FEEDBACK OFF" AND "M_0.5_SEC_2HZ"));
END_REGION

REGION Network 35: FEEDBACK ON AUX FOR HMI / Feedback On Aux for HMI
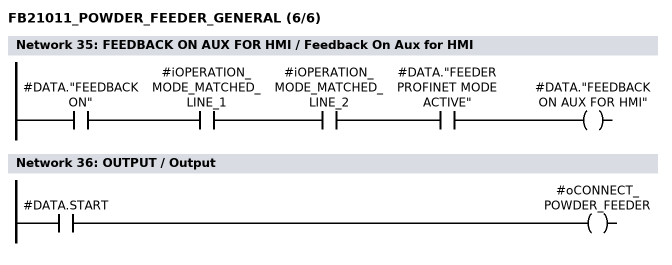
   RUNG wire#powerrail
      Contact( #DATA."FEEDBACK ON" )
      Contact( #iOPERATION_MODE_MATCHED_LINE_1 )
      Contact( #iOPERATION_MODE_MATCHED_LINE_2 )
      Contact( #DATA."FEEDER PROFINET MODE ACTIVE" )
      Coil( #DATA."FEEDBACK ON AUX FOR HMI" )
   END_RUNG
   // the same network as SCL:
   #DATA."FEEDBACK ON AUX FOR HMI" := #DATA."FEEDBACK ON" AND #iOPERATION_MODE_MATCHED_LINE_1 AND #iOPERATION_MODE_MATCHED_LINE_2 AND #DATA."FEEDER PROFINET MODE ACTIVE";
END_REGION

REGION Network 36: OUTPUT / Output
   RUNG wire#powerrail
      Contact( #DATA.START )
      Coil( #oCONNECT_POWDER_FEEDER )
   END_RUNG
   // the same network as SCL:
   #oCONNECT_POWDER_FEEDER := #DATA.START;
END_REGION
END_FUNCTION_BLOCK

FUNCTION "FC21012_POWDER_FEEDER_HEATER_JKL" : Void   // FC21012, LAD
TITLE = FC21012 POWDER FEEDER HEATER JKL
{ S7_Optimized_Access := 'TRUE' }
VERSION : 0.1
// stored: AutoNumber false, IsIECCheckEnabled false, SetENOAutomatically false, UDAEnableTagReadback false
BEGIN

REGION Network 1: /////_UNIT_01_/////
END_REGION

REGION Network 2: CALL FB21012 POWDER FEEDER 1 HEATER JKL UNIT 01
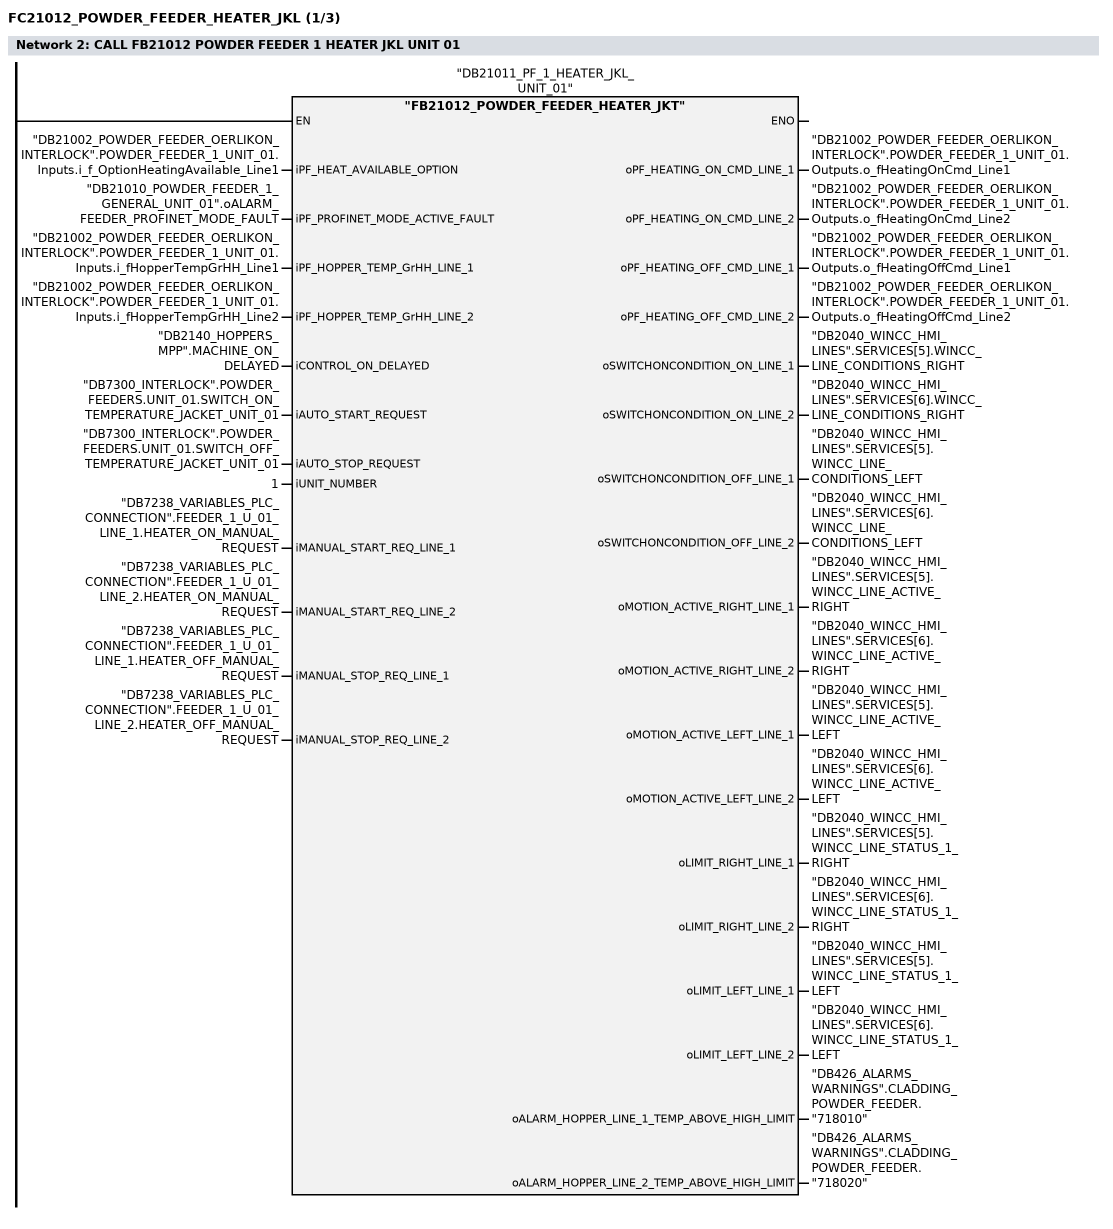
   RUNG wire#powerrail
      "DB21011_PF_1_HEATER_JKL_UNIT_01"(iPF_HEAT_AVAILABLE_OPTION := "DB21002_POWDER_FEEDER_OERLIKON_INTERLOCK".POWDER_FEEDER_1_UNIT_01.Inputs.i_f_OptionHeatingAvailable_Line1, iPF_PROFINET_MODE_ACTIVE_FAULT := "DB21010_POWDER_FEEDER_1_GENERAL_UNIT_01".oALARM_FEEDER_PROFINET_MODE_FAULT, iPF_HOPPER_TEMP_GrHH_LINE_1 := "DB21002_POWDER_FEEDER_OERLIKON_INTERLOCK".POWDER_FEEDER_1_UNIT_01.Inputs.i_fHopperTempGrHH_Line1, iPF_HOPPER_TEMP_GrHH_LINE_2 := "DB21002_POWDER_FEEDER_OERLIKON_INTERLOCK".POWDER_FEEDER_1_UNIT_01.Inputs.i_fHopperTempGrHH_Line2, iCONTROL_ON_DELAYED := "DB2140_HOPPERS_MPP".MACHINE_ON_DELAYED, iAUTO_START_REQUEST := "DB7300_INTERLOCK".POWDER_FEEDERS.UNIT_01.SWITCH_ON_TEMPERATURE_JACKET_UNIT_01, iAUTO_STOP_REQUEST := "DB7300_INTERLOCK".POWDER_FEEDERS.UNIT_01.SWITCH_OFF_TEMPERATURE_JACKET_UNIT_01, iUNIT_NUMBER := 1, iMANUAL_START_REQ_LINE_1 := "DB7238_VARIABLES_PLC_CONNECTION".FEEDER_1_U_01_LINE_1.HEATER_ON_MANUAL_REQUEST, iMANUAL_START_REQ_LINE_2 := "DB7238_VARIABLES_PLC_CONNECTION".FEEDER_1_U_01_LINE_2.HEATER_ON_MANUAL_REQUEST, iMANUAL_STOP_REQ_LINE_1 := "DB7238_VARIABLES_PLC_CONNECTION".FEEDER_1_U_01_LINE_1.HEATER_OFF_MANUAL_REQUEST, iMANUAL_STOP_REQ_LINE_2 := "DB7238_VARIABLES_PLC_CONNECTION".FEEDER_1_U_01_LINE_2.HEATER_OFF_MANUAL_REQUEST, oPF_HEATING_ON_CMD_LINE_1 => "DB21002_POWDER_FEEDER_OERLIKON_INTERLOCK".POWDER_FEEDER_1_UNIT_01.Outputs.o_fHeatingOnCmd_Line1, oPF_HEATING_ON_CMD_LINE_2 => "DB21002_POWDER_FEEDER_OERLIKON_INTERLOCK".POWDER_FEEDER_1_UNIT_01.Outputs.o_fHeatingOnCmd_Line2, oPF_HEATING_OFF_CMD_LINE_1 => "DB21002_POWDER_FEEDER_OERLIKON_INTERLOCK".POWDER_FEEDER_1_UNIT_01.Outputs.o_fHeatingOffCmd_Line1, oPF_HEATING_OFF_CMD_LINE_2 => "DB21002_POWDER_FEEDER_OERLIKON_INTERLOCK".POWDER_FEEDER_1_UNIT_01.Outputs.o_fHeatingOffCmd_Line2, oSWITCHONCONDITION_ON_LINE_1 => "DB2040_WINCC_HMI_LINES".SERVICES[5].WINCC_LINE_CONDITIONS_RIGHT, oSWITCHONCONDITION_ON_LINE_2 => "DB2040_WINCC_HMI_LINES".SERVICES[6].WINCC_LINE_CONDITIONS_RIGHT, oSWITCHONCONDITION_OFF_LINE_1 => "DB2040_WINCC_HMI_LINES".SERVICES[5].WINCC_LINE_CONDITIONS_LEFT, oSWITCHONCONDITION_OFF_LINE_2 => "DB2040_WINCC_HMI_LINES".SERVICES[6].WINCC_LINE_CONDITIONS_LEFT, oMOTION_ACTIVE_RIGHT_LINE_1 => "DB2040_WINCC_HMI_LINES".SERVICES[5].WINCC_LINE_ACTIVE_RIGHT, oMOTION_ACTIVE_RIGHT_LINE_2 => "DB2040_WINCC_HMI_LINES".SERVICES[6].WINCC_LINE_ACTIVE_RIGHT, oMOTION_ACTIVE_LEFT_LINE_1 => "DB2040_WINCC_HMI_LINES".SERVICES[5].WINCC_LINE_ACTIVE_LEFT, oMOTION_ACTIVE_LEFT_LINE_2 => "DB2040_WINCC_HMI_LINES".SERVICES[6].WINCC_LINE_ACTIVE_LEFT, oLIMIT_RIGHT_LINE_1 => "DB2040_WINCC_HMI_LINES".SERVICES[5].WINCC_LINE_STATUS_1_RIGHT, oLIMIT_RIGHT_LINE_2 => "DB2040_WINCC_HMI_LINES".SERVICES[6].WINCC_LINE_STATUS_1_RIGHT, oLIMIT_LEFT_LINE_1 => "DB2040_WINCC_HMI_LINES".SERVICES[5].WINCC_LINE_STATUS_1_LEFT, oLIMIT_LEFT_LINE_2 => "DB2040_WINCC_HMI_LINES".SERVICES[6].WINCC_LINE_STATUS_1_LEFT, oALARM_HOPPER_LINE_1_TEMP_ABOVE_HIGH_LIMIT => "DB426_ALARMS_WARNINGS".CLADDING_POWDER_FEEDER."718010", oALARM_HOPPER_LINE_2_TEMP_ABOVE_HIGH_LIMIT => "DB426_ALARMS_WARNINGS".CLADDING_POWDER_FEEDER."718020")
   END_RUNG
   // the same network as SCL:
   "DB21011_PF_1_HEATER_JKL_UNIT_01"(iPF_HEAT_AVAILABLE_OPTION := "DB21002_POWDER_FEEDER_OERLIKON_INTERLOCK".POWDER_FEEDER_1_UNIT_01.Inputs.i_f_OptionHeatingAvailable_Line1,   // "FB21012_POWDER_FEEDER_HEATER_JKT"
                           iPF_PROFINET_MODE_ACTIVE_FAULT := "DB21010_POWDER_FEEDER_1_GENERAL_UNIT_01".oALARM_FEEDER_PROFINET_MODE_FAULT,
                           iPF_HOPPER_TEMP_GrHH_LINE_1 := "DB21002_POWDER_FEEDER_OERLIKON_INTERLOCK".POWDER_FEEDER_1_UNIT_01.Inputs.i_fHopperTempGrHH_Line1,
                           iPF_HOPPER_TEMP_GrHH_LINE_2 := "DB21002_POWDER_FEEDER_OERLIKON_INTERLOCK".POWDER_FEEDER_1_UNIT_01.Inputs.i_fHopperTempGrHH_Line2,
                           iCONTROL_ON_DELAYED := "DB2140_HOPPERS_MPP".MACHINE_ON_DELAYED,
                           iAUTO_START_REQUEST := "DB7300_INTERLOCK".POWDER_FEEDERS.UNIT_01.SWITCH_ON_TEMPERATURE_JACKET_UNIT_01,
                           iAUTO_STOP_REQUEST := "DB7300_INTERLOCK".POWDER_FEEDERS.UNIT_01.SWITCH_OFF_TEMPERATURE_JACKET_UNIT_01,
                           iUNIT_NUMBER := 1,
                           iMANUAL_START_REQ_LINE_1 := "DB7238_VARIABLES_PLC_CONNECTION".FEEDER_1_U_01_LINE_1.HEATER_ON_MANUAL_REQUEST,
                           iMANUAL_START_REQ_LINE_2 := "DB7238_VARIABLES_PLC_CONNECTION".FEEDER_1_U_01_LINE_2.HEATER_ON_MANUAL_REQUEST,
                           iMANUAL_STOP_REQ_LINE_1 := "DB7238_VARIABLES_PLC_CONNECTION".FEEDER_1_U_01_LINE_1.HEATER_OFF_MANUAL_REQUEST,
                           iMANUAL_STOP_REQ_LINE_2 := "DB7238_VARIABLES_PLC_CONNECTION".FEEDER_1_U_01_LINE_2.HEATER_OFF_MANUAL_REQUEST,
                           oPF_HEATING_ON_CMD_LINE_1 => "DB21002_POWDER_FEEDER_OERLIKON_INTERLOCK".POWDER_FEEDER_1_UNIT_01.Outputs.o_fHeatingOnCmd_Line1,
                           oPF_HEATING_ON_CMD_LINE_2 => "DB21002_POWDER_FEEDER_OERLIKON_INTERLOCK".POWDER_FEEDER_1_UNIT_01.Outputs.o_fHeatingOnCmd_Line2,
                           oPF_HEATING_OFF_CMD_LINE_1 => "DB21002_POWDER_FEEDER_OERLIKON_INTERLOCK".POWDER_FEEDER_1_UNIT_01.Outputs.o_fHeatingOffCmd_Line1,
                           oPF_HEATING_OFF_CMD_LINE_2 => "DB21002_POWDER_FEEDER_OERLIKON_INTERLOCK".POWDER_FEEDER_1_UNIT_01.Outputs.o_fHeatingOffCmd_Line2,
                           oSWITCHONCONDITION_ON_LINE_1 => "DB2040_WINCC_HMI_LINES".SERVICES[5].WINCC_LINE_CONDITIONS_RIGHT,
                           oSWITCHONCONDITION_ON_LINE_2 => "DB2040_WINCC_HMI_LINES".SERVICES[6].WINCC_LINE_CONDITIONS_RIGHT,
                           oSWITCHONCONDITION_OFF_LINE_1 => "DB2040_WINCC_HMI_LINES".SERVICES[5].WINCC_LINE_CONDITIONS_LEFT,
                           oSWITCHONCONDITION_OFF_LINE_2 => "DB2040_WINCC_HMI_LINES".SERVICES[6].WINCC_LINE_CONDITIONS_LEFT,
                           oMOTION_ACTIVE_RIGHT_LINE_1 => "DB2040_WINCC_HMI_LINES".SERVICES[5].WINCC_LINE_ACTIVE_RIGHT,
                           oMOTION_ACTIVE_RIGHT_LINE_2 => "DB2040_WINCC_HMI_LINES".SERVICES[6].WINCC_LINE_ACTIVE_RIGHT,
                           oMOTION_ACTIVE_LEFT_LINE_1 => "DB2040_WINCC_HMI_LINES".SERVICES[5].WINCC_LINE_ACTIVE_LEFT,
                           oMOTION_ACTIVE_LEFT_LINE_2 => "DB2040_WINCC_HMI_LINES".SERVICES[6].WINCC_LINE_ACTIVE_LEFT,
                           oLIMIT_RIGHT_LINE_1 => "DB2040_WINCC_HMI_LINES".SERVICES[5].WINCC_LINE_STATUS_1_RIGHT,
                           oLIMIT_RIGHT_LINE_2 => "DB2040_WINCC_HMI_LINES".SERVICES[6].WINCC_LINE_STATUS_1_RIGHT,
                           oLIMIT_LEFT_LINE_1 => "DB2040_WINCC_HMI_LINES".SERVICES[5].WINCC_LINE_STATUS_1_LEFT,
                           oLIMIT_LEFT_LINE_2 => "DB2040_WINCC_HMI_LINES".SERVICES[6].WINCC_LINE_STATUS_1_LEFT,
                           oALARM_HOPPER_LINE_1_TEMP_ABOVE_HIGH_LIMIT => "DB426_ALARMS_WARNINGS".CLADDING_POWDER_FEEDER."718010",
                           oALARM_HOPPER_LINE_2_TEMP_ABOVE_HIGH_LIMIT => "DB426_ALARMS_WARNINGS".CLADDING_POWDER_FEEDER."718020");
END_REGION

REGION Network 3: /////_UNIT_02_/////
END_REGION

REGION Network 4: CALL FB21012 POWDER FEEDER 1 HEATER JKL UNIT 02
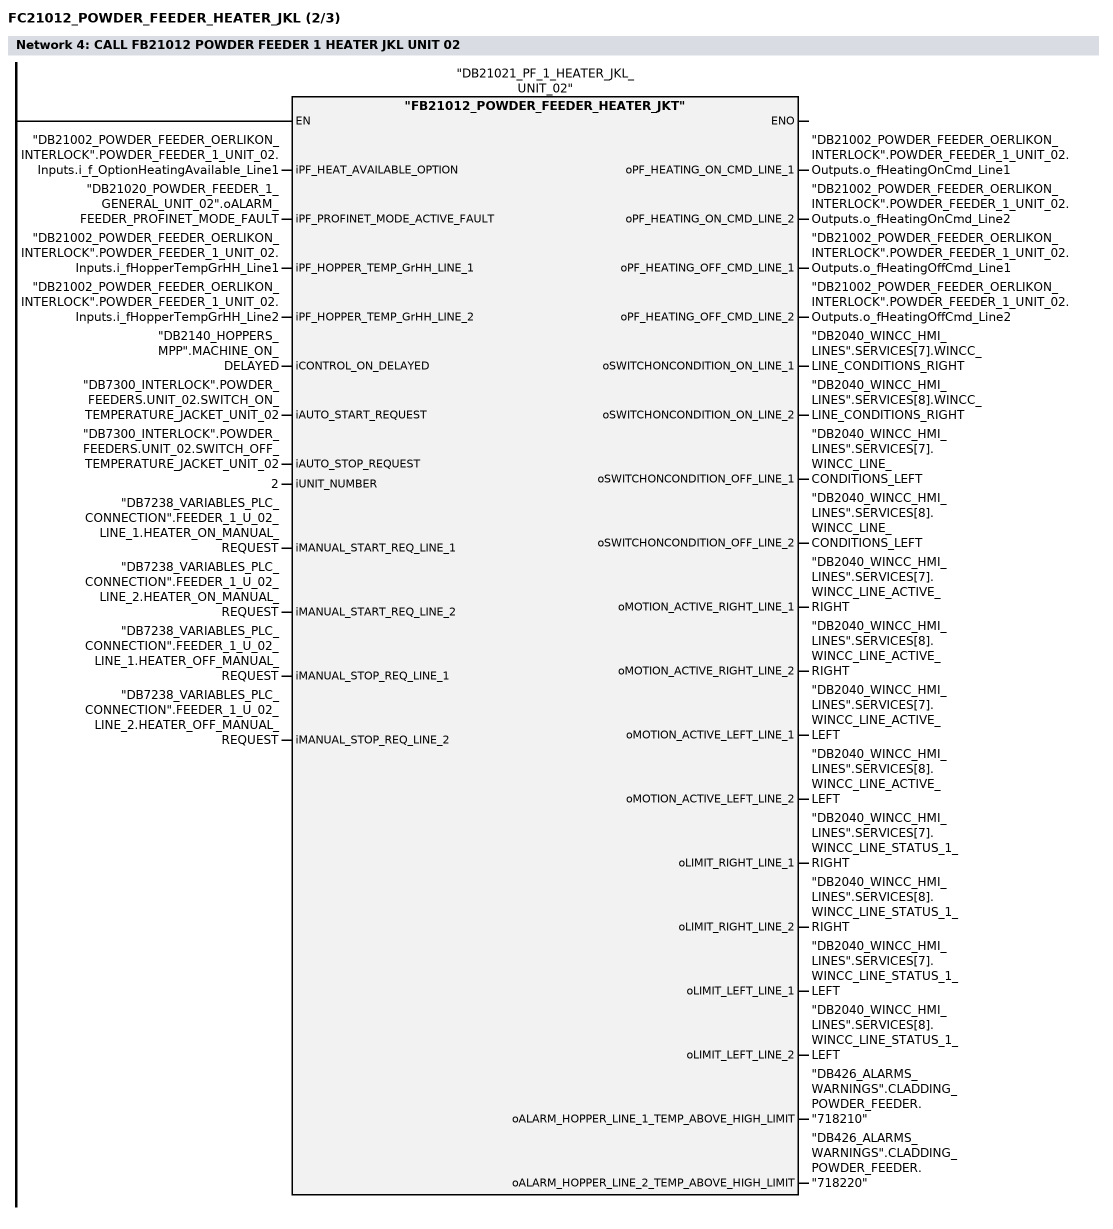
   RUNG wire#powerrail
      "DB21021_PF_1_HEATER_JKL_UNIT_02"(iPF_HEAT_AVAILABLE_OPTION := "DB21002_POWDER_FEEDER_OERLIKON_INTERLOCK".POWDER_FEEDER_1_UNIT_02.Inputs.i_f_OptionHeatingAvailable_Line1, iPF_PROFINET_MODE_ACTIVE_FAULT := "DB21020_POWDER_FEEDER_1_GENERAL_UNIT_02".oALARM_FEEDER_PROFINET_MODE_FAULT, iPF_HOPPER_TEMP_GrHH_LINE_1 := "DB21002_POWDER_FEEDER_OERLIKON_INTERLOCK".POWDER_FEEDER_1_UNIT_02.Inputs.i_fHopperTempGrHH_Line1, iPF_HOPPER_TEMP_GrHH_LINE_2 := "DB21002_POWDER_FEEDER_OERLIKON_INTERLOCK".POWDER_FEEDER_1_UNIT_02.Inputs.i_fHopperTempGrHH_Line2, iCONTROL_ON_DELAYED := "DB2140_HOPPERS_MPP".MACHINE_ON_DELAYED, iAUTO_START_REQUEST := "DB7300_INTERLOCK".POWDER_FEEDERS.UNIT_02.SWITCH_ON_TEMPERATURE_JACKET_UNIT_02, iAUTO_STOP_REQUEST := "DB7300_INTERLOCK".POWDER_FEEDERS.UNIT_02.SWITCH_OFF_TEMPERATURE_JACKET_UNIT_02, iUNIT_NUMBER := 2, iMANUAL_START_REQ_LINE_1 := "DB7238_VARIABLES_PLC_CONNECTION".FEEDER_1_U_02_LINE_1.HEATER_ON_MANUAL_REQUEST, iMANUAL_START_REQ_LINE_2 := "DB7238_VARIABLES_PLC_CONNECTION".FEEDER_1_U_02_LINE_2.HEATER_ON_MANUAL_REQUEST, iMANUAL_STOP_REQ_LINE_1 := "DB7238_VARIABLES_PLC_CONNECTION".FEEDER_1_U_02_LINE_1.HEATER_OFF_MANUAL_REQUEST, iMANUAL_STOP_REQ_LINE_2 := "DB7238_VARIABLES_PLC_CONNECTION".FEEDER_1_U_02_LINE_2.HEATER_OFF_MANUAL_REQUEST, oPF_HEATING_ON_CMD_LINE_1 => "DB21002_POWDER_FEEDER_OERLIKON_INTERLOCK".POWDER_FEEDER_1_UNIT_02.Outputs.o_fHeatingOnCmd_Line1, oPF_HEATING_ON_CMD_LINE_2 => "DB21002_POWDER_FEEDER_OERLIKON_INTERLOCK".POWDER_FEEDER_1_UNIT_02.Outputs.o_fHeatingOnCmd_Line2, oPF_HEATING_OFF_CMD_LINE_1 => "DB21002_POWDER_FEEDER_OERLIKON_INTERLOCK".POWDER_FEEDER_1_UNIT_02.Outputs.o_fHeatingOffCmd_Line1, oPF_HEATING_OFF_CMD_LINE_2 => "DB21002_POWDER_FEEDER_OERLIKON_INTERLOCK".POWDER_FEEDER_1_UNIT_02.Outputs.o_fHeatingOffCmd_Line2, oSWITCHONCONDITION_ON_LINE_1 => "DB2040_WINCC_HMI_LINES".SERVICES[7].WINCC_LINE_CONDITIONS_RIGHT, oSWITCHONCONDITION_ON_LINE_2 => "DB2040_WINCC_HMI_LINES".SERVICES[8].WINCC_LINE_CONDITIONS_RIGHT, oSWITCHONCONDITION_OFF_LINE_1 => "DB2040_WINCC_HMI_LINES".SERVICES[7].WINCC_LINE_CONDITIONS_LEFT, oSWITCHONCONDITION_OFF_LINE_2 => "DB2040_WINCC_HMI_LINES".SERVICES[8].WINCC_LINE_CONDITIONS_LEFT, oMOTION_ACTIVE_RIGHT_LINE_1 => "DB2040_WINCC_HMI_LINES".SERVICES[7].WINCC_LINE_ACTIVE_RIGHT, oMOTION_ACTIVE_RIGHT_LINE_2 => "DB2040_WINCC_HMI_LINES".SERVICES[8].WINCC_LINE_ACTIVE_RIGHT, oMOTION_ACTIVE_LEFT_LINE_1 => "DB2040_WINCC_HMI_LINES".SERVICES[7].WINCC_LINE_ACTIVE_LEFT, oMOTION_ACTIVE_LEFT_LINE_2 => "DB2040_WINCC_HMI_LINES".SERVICES[8].WINCC_LINE_ACTIVE_LEFT, oLIMIT_RIGHT_LINE_1 => "DB2040_WINCC_HMI_LINES".SERVICES[7].WINCC_LINE_STATUS_1_RIGHT, oLIMIT_RIGHT_LINE_2 => "DB2040_WINCC_HMI_LINES".SERVICES[8].WINCC_LINE_STATUS_1_RIGHT, oLIMIT_LEFT_LINE_1 => "DB2040_WINCC_HMI_LINES".SERVICES[7].WINCC_LINE_STATUS_1_LEFT, oLIMIT_LEFT_LINE_2 => "DB2040_WINCC_HMI_LINES".SERVICES[8].WINCC_LINE_STATUS_1_LEFT, oALARM_HOPPER_LINE_1_TEMP_ABOVE_HIGH_LIMIT => "DB426_ALARMS_WARNINGS".CLADDING_POWDER_FEEDER."718210", oALARM_HOPPER_LINE_2_TEMP_ABOVE_HIGH_LIMIT => "DB426_ALARMS_WARNINGS".CLADDING_POWDER_FEEDER."718220")
   END_RUNG
   // the same network as SCL:
   "DB21021_PF_1_HEATER_JKL_UNIT_02"(iPF_HEAT_AVAILABLE_OPTION := "DB21002_POWDER_FEEDER_OERLIKON_INTERLOCK".POWDER_FEEDER_1_UNIT_02.Inputs.i_f_OptionHeatingAvailable_Line1,   // "FB21012_POWDER_FEEDER_HEATER_JKT"
                           iPF_PROFINET_MODE_ACTIVE_FAULT := "DB21020_POWDER_FEEDER_1_GENERAL_UNIT_02".oALARM_FEEDER_PROFINET_MODE_FAULT,
                           iPF_HOPPER_TEMP_GrHH_LINE_1 := "DB21002_POWDER_FEEDER_OERLIKON_INTERLOCK".POWDER_FEEDER_1_UNIT_02.Inputs.i_fHopperTempGrHH_Line1,
                           iPF_HOPPER_TEMP_GrHH_LINE_2 := "DB21002_POWDER_FEEDER_OERLIKON_INTERLOCK".POWDER_FEEDER_1_UNIT_02.Inputs.i_fHopperTempGrHH_Line2,
                           iCONTROL_ON_DELAYED := "DB2140_HOPPERS_MPP".MACHINE_ON_DELAYED,
                           iAUTO_START_REQUEST := "DB7300_INTERLOCK".POWDER_FEEDERS.UNIT_02.SWITCH_ON_TEMPERATURE_JACKET_UNIT_02,
                           iAUTO_STOP_REQUEST := "DB7300_INTERLOCK".POWDER_FEEDERS.UNIT_02.SWITCH_OFF_TEMPERATURE_JACKET_UNIT_02,
                           iUNIT_NUMBER := 2,
                           iMANUAL_START_REQ_LINE_1 := "DB7238_VARIABLES_PLC_CONNECTION".FEEDER_1_U_02_LINE_1.HEATER_ON_MANUAL_REQUEST,
                           iMANUAL_START_REQ_LINE_2 := "DB7238_VARIABLES_PLC_CONNECTION".FEEDER_1_U_02_LINE_2.HEATER_ON_MANUAL_REQUEST,
                           iMANUAL_STOP_REQ_LINE_1 := "DB7238_VARIABLES_PLC_CONNECTION".FEEDER_1_U_02_LINE_1.HEATER_OFF_MANUAL_REQUEST,
                           iMANUAL_STOP_REQ_LINE_2 := "DB7238_VARIABLES_PLC_CONNECTION".FEEDER_1_U_02_LINE_2.HEATER_OFF_MANUAL_REQUEST,
                           oPF_HEATING_ON_CMD_LINE_1 => "DB21002_POWDER_FEEDER_OERLIKON_INTERLOCK".POWDER_FEEDER_1_UNIT_02.Outputs.o_fHeatingOnCmd_Line1,
                           oPF_HEATING_ON_CMD_LINE_2 => "DB21002_POWDER_FEEDER_OERLIKON_INTERLOCK".POWDER_FEEDER_1_UNIT_02.Outputs.o_fHeatingOnCmd_Line2,
                           oPF_HEATING_OFF_CMD_LINE_1 => "DB21002_POWDER_FEEDER_OERLIKON_INTERLOCK".POWDER_FEEDER_1_UNIT_02.Outputs.o_fHeatingOffCmd_Line1,
                           oPF_HEATING_OFF_CMD_LINE_2 => "DB21002_POWDER_FEEDER_OERLIKON_INTERLOCK".POWDER_FEEDER_1_UNIT_02.Outputs.o_fHeatingOffCmd_Line2,
                           oSWITCHONCONDITION_ON_LINE_1 => "DB2040_WINCC_HMI_LINES".SERVICES[7].WINCC_LINE_CONDITIONS_RIGHT,
                           oSWITCHONCONDITION_ON_LINE_2 => "DB2040_WINCC_HMI_LINES".SERVICES[8].WINCC_LINE_CONDITIONS_RIGHT,
                           oSWITCHONCONDITION_OFF_LINE_1 => "DB2040_WINCC_HMI_LINES".SERVICES[7].WINCC_LINE_CONDITIONS_LEFT,
                           oSWITCHONCONDITION_OFF_LINE_2 => "DB2040_WINCC_HMI_LINES".SERVICES[8].WINCC_LINE_CONDITIONS_LEFT,
                           oMOTION_ACTIVE_RIGHT_LINE_1 => "DB2040_WINCC_HMI_LINES".SERVICES[7].WINCC_LINE_ACTIVE_RIGHT,
                           oMOTION_ACTIVE_RIGHT_LINE_2 => "DB2040_WINCC_HMI_LINES".SERVICES[8].WINCC_LINE_ACTIVE_RIGHT,
                           oMOTION_ACTIVE_LEFT_LINE_1 => "DB2040_WINCC_HMI_LINES".SERVICES[7].WINCC_LINE_ACTIVE_LEFT,
                           oMOTION_ACTIVE_LEFT_LINE_2 => "DB2040_WINCC_HMI_LINES".SERVICES[8].WINCC_LINE_ACTIVE_LEFT,
                           oLIMIT_RIGHT_LINE_1 => "DB2040_WINCC_HMI_LINES".SERVICES[7].WINCC_LINE_STATUS_1_RIGHT,
                           oLIMIT_RIGHT_LINE_2 => "DB2040_WINCC_HMI_LINES".SERVICES[8].WINCC_LINE_STATUS_1_RIGHT,
                           oLIMIT_LEFT_LINE_1 => "DB2040_WINCC_HMI_LINES".SERVICES[7].WINCC_LINE_STATUS_1_LEFT,
                           oLIMIT_LEFT_LINE_2 => "DB2040_WINCC_HMI_LINES".SERVICES[8].WINCC_LINE_STATUS_1_LEFT,
                           oALARM_HOPPER_LINE_1_TEMP_ABOVE_HIGH_LIMIT => "DB426_ALARMS_WARNINGS".CLADDING_POWDER_FEEDER."718210",
                           oALARM_HOPPER_LINE_2_TEMP_ABOVE_HIGH_LIMIT => "DB426_ALARMS_WARNINGS".CLADDING_POWDER_FEEDER."718220");
END_REGION

REGION Network 5: CALL FB21012 POWDER FEEDER 2 HEATER JKL UNIT 02
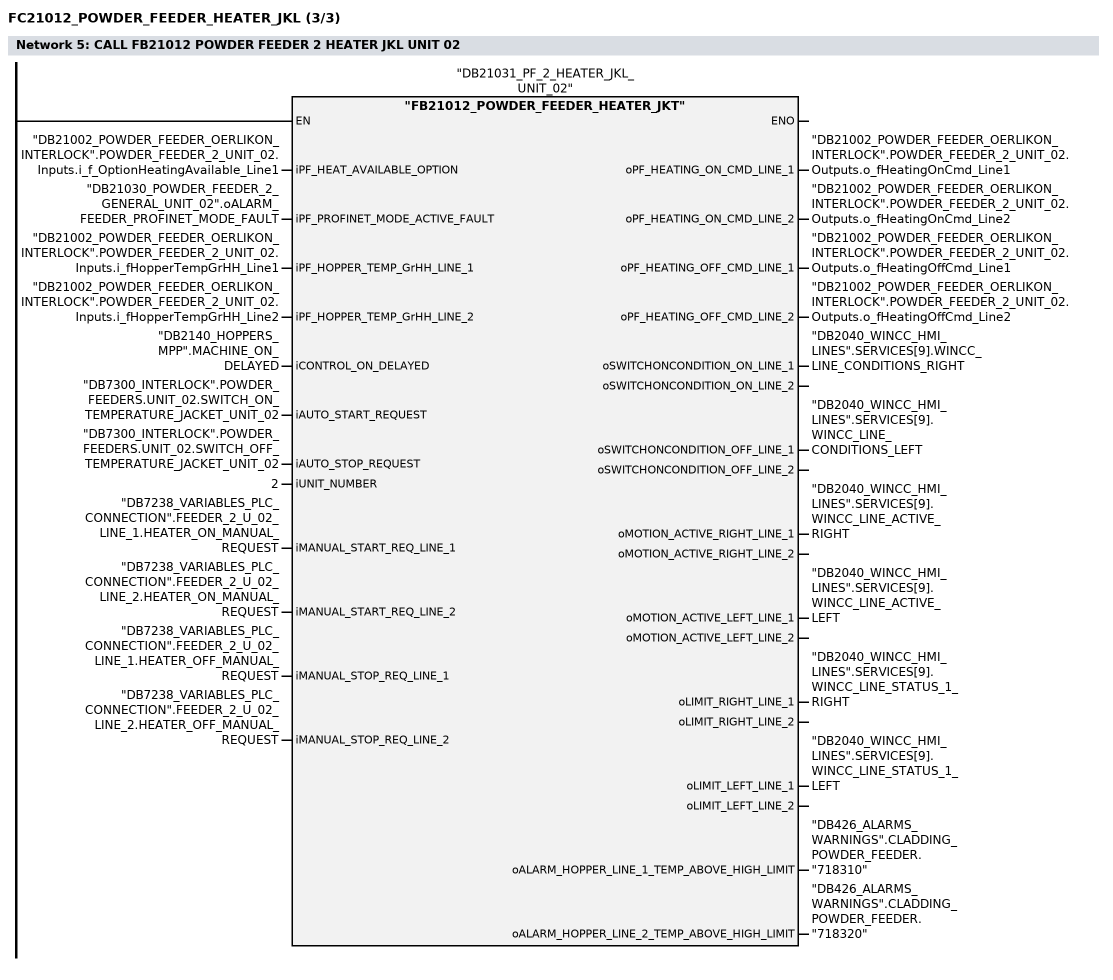
   RUNG wire#powerrail
      "DB21031_PF_2_HEATER_JKL_UNIT_02"(iPF_HEAT_AVAILABLE_OPTION := "DB21002_POWDER_FEEDER_OERLIKON_INTERLOCK".POWDER_FEEDER_2_UNIT_02.Inputs.i_f_OptionHeatingAvailable_Line1, iPF_PROFINET_MODE_ACTIVE_FAULT := "DB21030_POWDER_FEEDER_2_GENERAL_UNIT_02".oALARM_FEEDER_PROFINET_MODE_FAULT, iPF_HOPPER_TEMP_GrHH_LINE_1 := "DB21002_POWDER_FEEDER_OERLIKON_INTERLOCK".POWDER_FEEDER_2_UNIT_02.Inputs.i_fHopperTempGrHH_Line1, iPF_HOPPER_TEMP_GrHH_LINE_2 := "DB21002_POWDER_FEEDER_OERLIKON_INTERLOCK".POWDER_FEEDER_2_UNIT_02.Inputs.i_fHopperTempGrHH_Line2, iCONTROL_ON_DELAYED := "DB2140_HOPPERS_MPP".MACHINE_ON_DELAYED, iAUTO_START_REQUEST := "DB7300_INTERLOCK".POWDER_FEEDERS.UNIT_02.SWITCH_ON_TEMPERATURE_JACKET_UNIT_02, iAUTO_STOP_REQUEST := "DB7300_INTERLOCK".POWDER_FEEDERS.UNIT_02.SWITCH_OFF_TEMPERATURE_JACKET_UNIT_02, iUNIT_NUMBER := 2, iMANUAL_START_REQ_LINE_1 := "DB7238_VARIABLES_PLC_CONNECTION".FEEDER_2_U_02_LINE_1.HEATER_ON_MANUAL_REQUEST, iMANUAL_START_REQ_LINE_2 := "DB7238_VARIABLES_PLC_CONNECTION".FEEDER_2_U_02_LINE_2.HEATER_ON_MANUAL_REQUEST, iMANUAL_STOP_REQ_LINE_1 := "DB7238_VARIABLES_PLC_CONNECTION".FEEDER_2_U_02_LINE_1.HEATER_OFF_MANUAL_REQUEST, iMANUAL_STOP_REQ_LINE_2 := "DB7238_VARIABLES_PLC_CONNECTION".FEEDER_2_U_02_LINE_2.HEATER_OFF_MANUAL_REQUEST, oPF_HEATING_ON_CMD_LINE_1 => "DB21002_POWDER_FEEDER_OERLIKON_INTERLOCK".POWDER_FEEDER_2_UNIT_02.Outputs.o_fHeatingOnCmd_Line1, oPF_HEATING_ON_CMD_LINE_2 => "DB21002_POWDER_FEEDER_OERLIKON_INTERLOCK".POWDER_FEEDER_2_UNIT_02.Outputs.o_fHeatingOnCmd_Line2, oPF_HEATING_OFF_CMD_LINE_1 => "DB21002_POWDER_FEEDER_OERLIKON_INTERLOCK".POWDER_FEEDER_2_UNIT_02.Outputs.o_fHeatingOffCmd_Line1, oPF_HEATING_OFF_CMD_LINE_2 => "DB21002_POWDER_FEEDER_OERLIKON_INTERLOCK".POWDER_FEEDER_2_UNIT_02.Outputs.o_fHeatingOffCmd_Line2, oSWITCHONCONDITION_ON_LINE_1 => "DB2040_WINCC_HMI_LINES".SERVICES[9].WINCC_LINE_CONDITIONS_RIGHT, oSWITCHONCONDITION_ON_LINE_2 =>, oSWITCHONCONDITION_OFF_LINE_1 => "DB2040_WINCC_HMI_LINES".SERVICES[9].WINCC_LINE_CONDITIONS_LEFT, oSWITCHONCONDITION_OFF_LINE_2 =>, oMOTION_ACTIVE_RIGHT_LINE_1 => "DB2040_WINCC_HMI_LINES".SERVICES[9].WINCC_LINE_ACTIVE_RIGHT, oMOTION_ACTIVE_RIGHT_LINE_2 =>, oMOTION_ACTIVE_LEFT_LINE_1 => "DB2040_WINCC_HMI_LINES".SERVICES[9].WINCC_LINE_ACTIVE_LEFT, oMOTION_ACTIVE_LEFT_LINE_2 =>, oLIMIT_RIGHT_LINE_1 => "DB2040_WINCC_HMI_LINES".SERVICES[9].WINCC_LINE_STATUS_1_RIGHT, oLIMIT_RIGHT_LINE_2 =>, oLIMIT_LEFT_LINE_1 => "DB2040_WINCC_HMI_LINES".SERVICES[9].WINCC_LINE_STATUS_1_LEFT, oLIMIT_LEFT_LINE_2 =>, oALARM_HOPPER_LINE_1_TEMP_ABOVE_HIGH_LIMIT => "DB426_ALARMS_WARNINGS".CLADDING_POWDER_FEEDER."718310", oALARM_HOPPER_LINE_2_TEMP_ABOVE_HIGH_LIMIT => "DB426_ALARMS_WARNINGS".CLADDING_POWDER_FEEDER."718320")
   END_RUNG
   // the same network as SCL:
   "DB21031_PF_2_HEATER_JKL_UNIT_02"(iPF_HEAT_AVAILABLE_OPTION := "DB21002_POWDER_FEEDER_OERLIKON_INTERLOCK".POWDER_FEEDER_2_UNIT_02.Inputs.i_f_OptionHeatingAvailable_Line1,   // "FB21012_POWDER_FEEDER_HEATER_JKT"
                           iPF_PROFINET_MODE_ACTIVE_FAULT := "DB21030_POWDER_FEEDER_2_GENERAL_UNIT_02".oALARM_FEEDER_PROFINET_MODE_FAULT,
                           iPF_HOPPER_TEMP_GrHH_LINE_1 := "DB21002_POWDER_FEEDER_OERLIKON_INTERLOCK".POWDER_FEEDER_2_UNIT_02.Inputs.i_fHopperTempGrHH_Line1,
                           iPF_HOPPER_TEMP_GrHH_LINE_2 := "DB21002_POWDER_FEEDER_OERLIKON_INTERLOCK".POWDER_FEEDER_2_UNIT_02.Inputs.i_fHopperTempGrHH_Line2,
                           iCONTROL_ON_DELAYED := "DB2140_HOPPERS_MPP".MACHINE_ON_DELAYED,
                           iAUTO_START_REQUEST := "DB7300_INTERLOCK".POWDER_FEEDERS.UNIT_02.SWITCH_ON_TEMPERATURE_JACKET_UNIT_02,
                           iAUTO_STOP_REQUEST := "DB7300_INTERLOCK".POWDER_FEEDERS.UNIT_02.SWITCH_OFF_TEMPERATURE_JACKET_UNIT_02,
                           iUNIT_NUMBER := 2,
                           iMANUAL_START_REQ_LINE_1 := "DB7238_VARIABLES_PLC_CONNECTION".FEEDER_2_U_02_LINE_1.HEATER_ON_MANUAL_REQUEST,
                           iMANUAL_START_REQ_LINE_2 := "DB7238_VARIABLES_PLC_CONNECTION".FEEDER_2_U_02_LINE_2.HEATER_ON_MANUAL_REQUEST,
                           iMANUAL_STOP_REQ_LINE_1 := "DB7238_VARIABLES_PLC_CONNECTION".FEEDER_2_U_02_LINE_1.HEATER_OFF_MANUAL_REQUEST,
                           iMANUAL_STOP_REQ_LINE_2 := "DB7238_VARIABLES_PLC_CONNECTION".FEEDER_2_U_02_LINE_2.HEATER_OFF_MANUAL_REQUEST,
                           oPF_HEATING_ON_CMD_LINE_1 => "DB21002_POWDER_FEEDER_OERLIKON_INTERLOCK".POWDER_FEEDER_2_UNIT_02.Outputs.o_fHeatingOnCmd_Line1,
                           oPF_HEATING_ON_CMD_LINE_2 => "DB21002_POWDER_FEEDER_OERLIKON_INTERLOCK".POWDER_FEEDER_2_UNIT_02.Outputs.o_fHeatingOnCmd_Line2,
                           oPF_HEATING_OFF_CMD_LINE_1 => "DB21002_POWDER_FEEDER_OERLIKON_INTERLOCK".POWDER_FEEDER_2_UNIT_02.Outputs.o_fHeatingOffCmd_Line1,
                           oPF_HEATING_OFF_CMD_LINE_2 => "DB21002_POWDER_FEEDER_OERLIKON_INTERLOCK".POWDER_FEEDER_2_UNIT_02.Outputs.o_fHeatingOffCmd_Line2,
                           oSWITCHONCONDITION_ON_LINE_1 => "DB2040_WINCC_HMI_LINES".SERVICES[9].WINCC_LINE_CONDITIONS_RIGHT,
                           oSWITCHONCONDITION_OFF_LINE_1 => "DB2040_WINCC_HMI_LINES".SERVICES[9].WINCC_LINE_CONDITIONS_LEFT,
                           oMOTION_ACTIVE_RIGHT_LINE_1 => "DB2040_WINCC_HMI_LINES".SERVICES[9].WINCC_LINE_ACTIVE_RIGHT,
                           oMOTION_ACTIVE_LEFT_LINE_1 => "DB2040_WINCC_HMI_LINES".SERVICES[9].WINCC_LINE_ACTIVE_LEFT,
                           oLIMIT_RIGHT_LINE_1 => "DB2040_WINCC_HMI_LINES".SERVICES[9].WINCC_LINE_STATUS_1_RIGHT,
                           oLIMIT_LEFT_LINE_1 => "DB2040_WINCC_HMI_LINES".SERVICES[9].WINCC_LINE_STATUS_1_LEFT,
                           oALARM_HOPPER_LINE_1_TEMP_ABOVE_HIGH_LIMIT => "DB426_ALARMS_WARNINGS".CLADDING_POWDER_FEEDER."718310",
                           oALARM_HOPPER_LINE_2_TEMP_ABOVE_HIGH_LIMIT => "DB426_ALARMS_WARNINGS".CLADDING_POWDER_FEEDER."718320");
END_REGION
END_FUNCTION

FUNCTION_BLOCK "FB21012_POWDER_FEEDER_HEATER_JKT"   // FB21012, LAD
TITLE = FB21012 POWDER FEEDER HEATER JKT
{ S7_Optimized_Access := 'FALSE' }
VERSION : 0.1
// stored: AutoNumber false, IsIECCheckEnabled false, SetENOAutomatically false, UDAEnableTagReadback false
   VAR_INPUT
      iPF_HEAT_AVAILABLE_OPTION : Bool;
      iPF_PROFINET_MODE_ACTIVE_FAULT : Bool;
      iPF_HOPPER_TEMP_GrHH_LINE_1 : Bool;   // POWDER FEEDER HOPPER TEMPERATURE LINE 1 ALARM
      iPF_HOPPER_TEMP_GrHH_LINE_2 : Bool;   // POWDER FEEDER HOPPER TEMPERATURE LINE 2 ALARM
      iCONTROL_ON_DELAYED : Bool;   // LOCAL MACHINE ON
      iAUTO_START_REQUEST : Bool;   // AUTO START REQUEST
      iAUTO_STOP_REQUEST : Bool;   // AUTO STOP SEQUEST
      iUNIT_NUMBER : Byte;
      iMANUAL_START_REQ_LINE_1 : Bool;
      iMANUAL_START_REQ_LINE_2 : Bool;
      iMANUAL_STOP_REQ_LINE_1 : Bool;
      iMANUAL_STOP_REQ_LINE_2 : Bool;
   END_VAR
   VAR_OUTPUT
      oPF_HEATING_ON_CMD_LINE_1 : Bool;   // POWDER FEEDER HEATING ON COMMAND LINE 1
      oPF_HEATING_ON_CMD_LINE_2 : Bool;   // POWDER FEEDER HEATING ON COMMAND LINE 2
      oPF_HEATING_OFF_CMD_LINE_1 : Bool;   // POWDER FEEDER HEATING OF COMMAND LINE 1
      oPF_HEATING_OFF_CMD_LINE_2 : Bool;   // POWDER FEEDER HEATING OF COMMAND LINE 2
      oSWITCHONCONDITION_ON_LINE_1 : Bool;
      oSWITCHONCONDITION_ON_LINE_2 : Bool;
      oSWITCHONCONDITION_OFF_LINE_1 : Bool;
      oSWITCHONCONDITION_OFF_LINE_2 : Bool;
      oMOTION_ACTIVE_RIGHT_LINE_1 : Bool;
      oMOTION_ACTIVE_RIGHT_LINE_2 : Bool;
      oMOTION_ACTIVE_LEFT_LINE_1 : Bool;
      oMOTION_ACTIVE_LEFT_LINE_2 : Bool;
      oLIMIT_RIGHT_LINE_1 : Bool;
      oLIMIT_RIGHT_LINE_2 : Bool;
      oLIMIT_LEFT_LINE_1 : Bool;
      oLIMIT_LEFT_LINE_2 : Bool;
      oALARM_HOPPER_LINE_1_TEMP_ABOVE_HIGH_LIMIT : Bool;
      oALARM_HOPPER_LINE_2_TEMP_ABOVE_HIGH_LIMIT : Bool;
   END_VAR
   VAR DB_SPECIFIC
      DATA : "POWDER FEEDER HEATER JKT";
      INPUT_SETTINGS : Struct
         UNIT_NUMBER : Int;
         FEEDER_NUMBER : Int;
      END_STRUCT;
      HEATER_STATUS_LINE_1 { S7_SetPoint := 'True'} : Byte;
      HEATER_STATUS_LINE_2 : Byte;
   END_VAR
   VAR_TEMP
      DB_NUMBER : DInt;
   END_VAR
   VAR_TEMP   // added for the SCL form of the ladder/FBD networks
      _w1 : Bool;
      _w2 : Bool;
   END_VAR
BEGIN

NETWORK
TITLE = READ INSTANCE DB NUMBER
      L     DINO;
      +     10#800000;
      T     #DB_NUMBER;

REGION Network 2: START GENERAL CONDITIONS / Start General Conditions
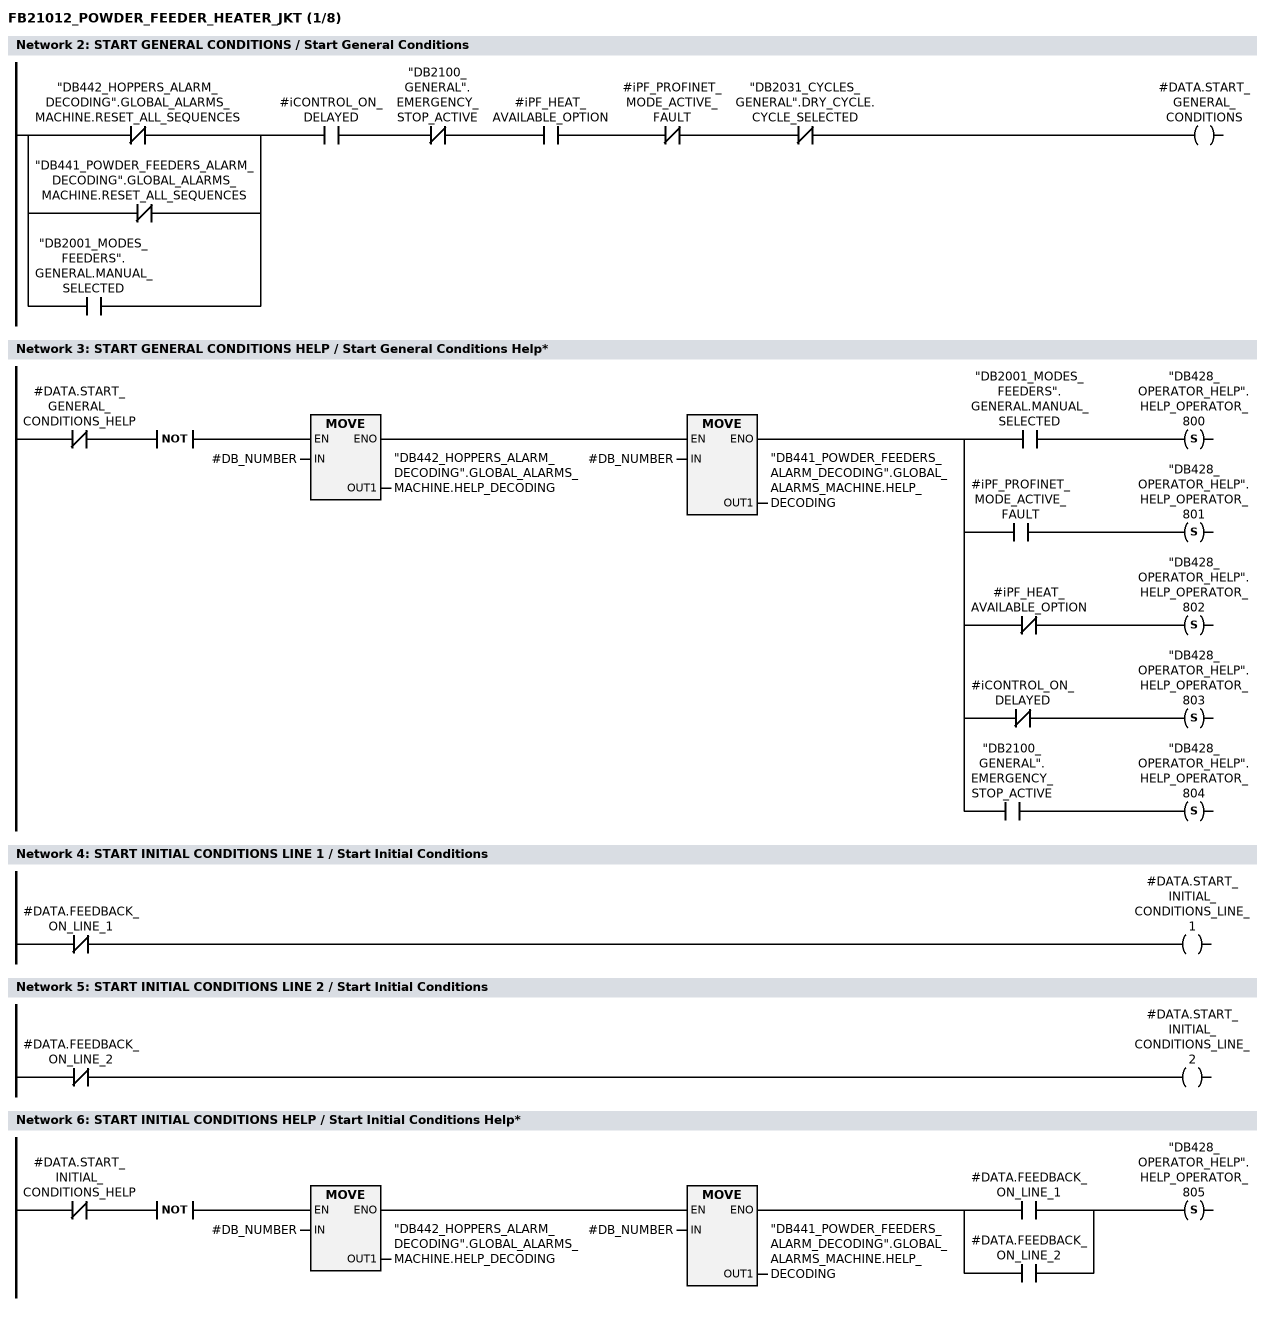
   RUNG wire#powerrail
      I_Contact( "DB442_HOPPERS_ALARM_DECODING".GLOBAL_ALARMS_MACHINE.RESET_ALL_SEQUENCES )
      wire#w1
      Contact( #iCONTROL_ON_DELAYED )
      I_Contact( "DB2100_GENERAL".EMERGENCY_STOP_ACTIVE )
      Contact( #iPF_HEAT_AVAILABLE_OPTION )
      I_Contact( #iPF_PROFINET_MODE_ACTIVE_FAULT )
      I_Contact( "DB2031_CYCLES_GENERAL".DRY_CYCLE.CYCLE_SELECTED )
      Coil( #DATA.START_GENERAL_CONDITIONS )
   END_RUNG
   RUNG wire#powerrail
      I_Contact( "DB441_POWDER_FEEDERS_ALARM_DECODING".GLOBAL_ALARMS_MACHINE.RESET_ALL_SEQUENCES )
   END_RUNG wire#w1
   RUNG wire#powerrail
      Contact( "DB2001_MODES_FEEDERS".GENERAL.MANUAL_SELECTED )
   END_RUNG wire#w1
   // the same network as SCL:
   #DATA.START_GENERAL_CONDITIONS := (NOT "DB442_HOPPERS_ALARM_DECODING".GLOBAL_ALARMS_MACHINE.RESET_ALL_SEQUENCES OR NOT "DB441_POWDER_FEEDERS_ALARM_DECODING".GLOBAL_ALARMS_MACHINE.RESET_ALL_SEQUENCES OR "DB2001_MODES_FEEDERS".GENERAL.MANUAL_SELECTED) AND #iCONTROL_ON_DELAYED AND NOT "DB2100_GENERAL".EMERGENCY_STOP_ACTIVE AND #iPF_HEAT_AVAILABLE_OPTION AND NOT #iPF_PROFINET_MODE_ACTIVE_FAULT AND NOT "DB2031_CYCLES_GENERAL".DRY_CYCLE.CYCLE_SELECTED;
END_REGION

REGION Network 3: START GENERAL CONDITIONS HELP / Start General Conditions Help*
   RUNG wire#powerrail
      I_Contact( #DATA.START_GENERAL_CONDITIONS_HELP )
      Not()
      Move(in := #DB_NUMBER, out1 => "DB442_HOPPERS_ALARM_DECODING".GLOBAL_ALARMS_MACHINE.HELP_DECODING)
      Move(in := #DB_NUMBER, out1 => "DB441_POWDER_FEEDERS_ALARM_DECODING".GLOBAL_ALARMS_MACHINE.HELP_DECODING)
      wire#w1
      Contact( "DB2001_MODES_FEEDERS".GENERAL.MANUAL_SELECTED )
      S_Coil( "DB428_OPERATOR_HELP".HELP_OPERATOR_800 )
   END_RUNG
   RUNG wire#w1
      Contact( #iPF_PROFINET_MODE_ACTIVE_FAULT )
      S_Coil( "DB428_OPERATOR_HELP".HELP_OPERATOR_801 )
   END_RUNG
   RUNG wire#w1
      I_Contact( #iPF_HEAT_AVAILABLE_OPTION )
      S_Coil( "DB428_OPERATOR_HELP".HELP_OPERATOR_802 )
   END_RUNG
   RUNG wire#w1
      I_Contact( #iCONTROL_ON_DELAYED )
      S_Coil( "DB428_OPERATOR_HELP".HELP_OPERATOR_803 )
   END_RUNG
   RUNG wire#w1
      Contact( "DB2100_GENERAL".EMERGENCY_STOP_ACTIVE )
      S_Coil( "DB428_OPERATOR_HELP".HELP_OPERATOR_804 )
   END_RUNG
   // the same network as SCL:
   #_w1 := NOT (NOT #DATA.START_GENERAL_CONDITIONS_HELP);
   IF #_w1 THEN
       "DB442_HOPPERS_ALARM_DECODING".GLOBAL_ALARMS_MACHINE.HELP_DECODING := #DB_NUMBER;
       "DB441_POWDER_FEEDERS_ALARM_DECODING".GLOBAL_ALARMS_MACHINE.HELP_DECODING := #DB_NUMBER;
   END_IF;
   IF #_w1 AND "DB2001_MODES_FEEDERS".GENERAL.MANUAL_SELECTED THEN
       "DB428_OPERATOR_HELP".HELP_OPERATOR_800 := TRUE;
   END_IF;
   IF #_w1 AND #iPF_PROFINET_MODE_ACTIVE_FAULT THEN "DB428_OPERATOR_HELP".HELP_OPERATOR_801 := TRUE; END_IF;
   IF #_w1 AND NOT #iPF_HEAT_AVAILABLE_OPTION THEN "DB428_OPERATOR_HELP".HELP_OPERATOR_802 := TRUE; END_IF;
   IF #_w1 AND NOT #iCONTROL_ON_DELAYED THEN "DB428_OPERATOR_HELP".HELP_OPERATOR_803 := TRUE; END_IF;
   IF #_w1 AND "DB2100_GENERAL".EMERGENCY_STOP_ACTIVE THEN
       "DB428_OPERATOR_HELP".HELP_OPERATOR_804 := TRUE;
   END_IF;
END_REGION

REGION Network 4: START INITIAL CONDITIONS LINE 1 / Start Initial Conditions
   RUNG wire#powerrail
      I_Contact( #DATA.FEEDBACK_ON_LINE_1 )
      Coil( #DATA.START_INITIAL_CONDITIONS_LINE_1 )
   END_RUNG
   // the same network as SCL:
   #DATA.START_INITIAL_CONDITIONS_LINE_1 := NOT #DATA.FEEDBACK_ON_LINE_1;
END_REGION

REGION Network 5: START INITIAL CONDITIONS LINE 2 / Start Initial Conditions
   RUNG wire#powerrail
      I_Contact( #DATA.FEEDBACK_ON_LINE_2 )
      Coil( #DATA.START_INITIAL_CONDITIONS_LINE_2 )
   END_RUNG
   // the same network as SCL:
   #DATA.START_INITIAL_CONDITIONS_LINE_2 := NOT #DATA.FEEDBACK_ON_LINE_2;
END_REGION

REGION Network 6: START INITIAL CONDITIONS HELP / Start Initial Conditions Help*
   RUNG wire#powerrail
      I_Contact( #DATA.START_INITIAL_CONDITIONS_HELP )
      Not()
      Move(in := #DB_NUMBER, out1 => "DB442_HOPPERS_ALARM_DECODING".GLOBAL_ALARMS_MACHINE.HELP_DECODING)
      Move(in := #DB_NUMBER, out1 => "DB441_POWDER_FEEDERS_ALARM_DECODING".GLOBAL_ALARMS_MACHINE.HELP_DECODING)
      wire#w1
      Contact( #DATA.FEEDBACK_ON_LINE_1 )
      wire#w2
      S_Coil( "DB428_OPERATOR_HELP".HELP_OPERATOR_805 )
   END_RUNG
   RUNG wire#w1
      Contact( #DATA.FEEDBACK_ON_LINE_2 )
   END_RUNG wire#w2
   // the same network as SCL:
   #_w1 := NOT (NOT #DATA.START_INITIAL_CONDITIONS_HELP);
   IF #_w1 THEN
       "DB442_HOPPERS_ALARM_DECODING".GLOBAL_ALARMS_MACHINE.HELP_DECODING := #DB_NUMBER;
       "DB441_POWDER_FEEDERS_ALARM_DECODING".GLOBAL_ALARMS_MACHINE.HELP_DECODING := #DB_NUMBER;
   END_IF;
   IF #_w1 AND (#DATA.FEEDBACK_ON_LINE_1 OR #DATA.FEEDBACK_ON_LINE_2) THEN
       "DB428_OPERATOR_HELP".HELP_OPERATOR_805 := TRUE;
   END_IF;
END_REGION

REGION Network 7: MANUAL MODE NOT SELECTED HELP / Manual Mode Not Selected Help*
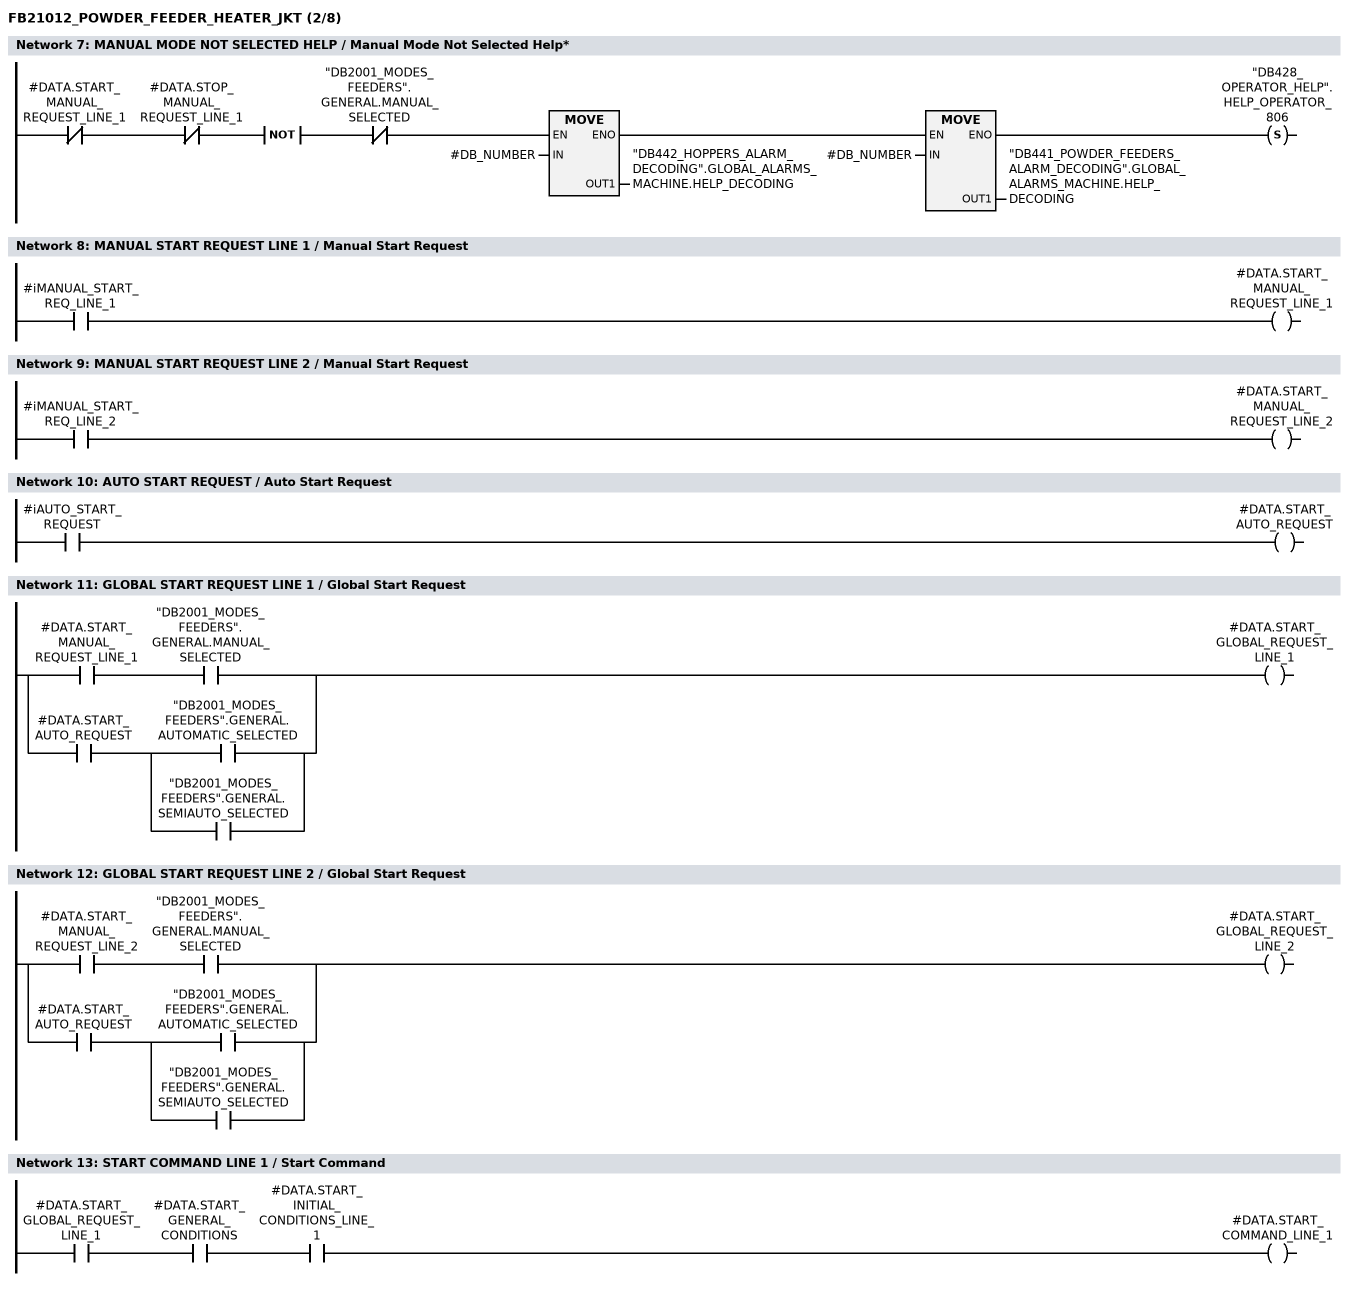
   RUNG wire#powerrail
      I_Contact( #DATA.START_MANUAL_REQUEST_LINE_1 )
      I_Contact( #DATA.STOP_MANUAL_REQUEST_LINE_1 )
      Not()
      I_Contact( "DB2001_MODES_FEEDERS".GENERAL.MANUAL_SELECTED )
      Move(in := #DB_NUMBER, out1 => "DB442_HOPPERS_ALARM_DECODING".GLOBAL_ALARMS_MACHINE.HELP_DECODING)
      Move(in := #DB_NUMBER, out1 => "DB441_POWDER_FEEDERS_ALARM_DECODING".GLOBAL_ALARMS_MACHINE.HELP_DECODING)
      S_Coil( "DB428_OPERATOR_HELP".HELP_OPERATOR_806 )
   END_RUNG
   // the same network as SCL:
   IF NOT (NOT #DATA.START_MANUAL_REQUEST_LINE_1 AND NOT #DATA.STOP_MANUAL_REQUEST_LINE_1) AND NOT "DB2001_MODES_FEEDERS".GENERAL.MANUAL_SELECTED THEN
       "DB442_HOPPERS_ALARM_DECODING".GLOBAL_ALARMS_MACHINE.HELP_DECODING := #DB_NUMBER;
       "DB441_POWDER_FEEDERS_ALARM_DECODING".GLOBAL_ALARMS_MACHINE.HELP_DECODING := #DB_NUMBER;
       "DB428_OPERATOR_HELP".HELP_OPERATOR_806 := TRUE;
   END_IF;
END_REGION

REGION Network 8: MANUAL START REQUEST LINE 1 / Manual Start Request
   RUNG wire#powerrail
      Contact( #iMANUAL_START_REQ_LINE_1 )
      Coil( #DATA.START_MANUAL_REQUEST_LINE_1 )
   END_RUNG
   // the same network as SCL:
   #DATA.START_MANUAL_REQUEST_LINE_1 := #iMANUAL_START_REQ_LINE_1;
END_REGION

REGION Network 9: MANUAL START REQUEST LINE 2 / Manual Start Request
   RUNG wire#powerrail
      Contact( #iMANUAL_START_REQ_LINE_2 )
      Coil( #DATA.START_MANUAL_REQUEST_LINE_2 )
   END_RUNG
   // the same network as SCL:
   #DATA.START_MANUAL_REQUEST_LINE_2 := #iMANUAL_START_REQ_LINE_2;
END_REGION

REGION Network 10: AUTO START REQUEST / Auto Start Request
   RUNG wire#powerrail
      Contact( #iAUTO_START_REQUEST )
      Coil( #DATA.START_AUTO_REQUEST )
   END_RUNG
   // the same network as SCL:
   #DATA.START_AUTO_REQUEST := #iAUTO_START_REQUEST;
END_REGION

REGION Network 11: GLOBAL START REQUEST LINE 1 / Global Start Request
   RUNG wire#powerrail
      Contact( #DATA.START_MANUAL_REQUEST_LINE_1 )
      Contact( "DB2001_MODES_FEEDERS".GENERAL.MANUAL_SELECTED )
      wire#w1
      Coil( #DATA.START_GLOBAL_REQUEST_LINE_1 )
   END_RUNG
   RUNG wire#powerrail
      Contact( #DATA.START_AUTO_REQUEST )
      wire#w2
      Contact( "DB2001_MODES_FEEDERS".GENERAL.AUTOMATIC_SELECTED )
   END_RUNG wire#w1
   RUNG wire#w2
      Contact( "DB2001_MODES_FEEDERS".GENERAL.SEMIAUTO_SELECTED )
   END_RUNG wire#w1
   // the same network as SCL:
   #DATA.START_GLOBAL_REQUEST_LINE_1 := (#DATA.START_MANUAL_REQUEST_LINE_1 AND "DB2001_MODES_FEEDERS".GENERAL.MANUAL_SELECTED) OR (#DATA.START_AUTO_REQUEST AND ("DB2001_MODES_FEEDERS".GENERAL.AUTOMATIC_SELECTED OR "DB2001_MODES_FEEDERS".GENERAL.SEMIAUTO_SELECTED));
END_REGION

REGION Network 12: GLOBAL START REQUEST LINE 2 / Global Start Request
   RUNG wire#powerrail
      Contact( #DATA.START_MANUAL_REQUEST_LINE_2 )
      Contact( "DB2001_MODES_FEEDERS".GENERAL.MANUAL_SELECTED )
      wire#w1
      Coil( #DATA.START_GLOBAL_REQUEST_LINE_2 )
   END_RUNG
   RUNG wire#powerrail
      Contact( #DATA.START_AUTO_REQUEST )
      wire#w2
      Contact( "DB2001_MODES_FEEDERS".GENERAL.AUTOMATIC_SELECTED )
   END_RUNG wire#w1
   RUNG wire#w2
      Contact( "DB2001_MODES_FEEDERS".GENERAL.SEMIAUTO_SELECTED )
   END_RUNG wire#w1
   // the same network as SCL:
   #DATA.START_GLOBAL_REQUEST_LINE_2 := (#DATA.START_MANUAL_REQUEST_LINE_2 AND "DB2001_MODES_FEEDERS".GENERAL.MANUAL_SELECTED) OR (#DATA.START_AUTO_REQUEST AND ("DB2001_MODES_FEEDERS".GENERAL.AUTOMATIC_SELECTED OR "DB2001_MODES_FEEDERS".GENERAL.SEMIAUTO_SELECTED));
END_REGION

REGION Network 13: START COMMAND LINE 1 / Start Command
   RUNG wire#powerrail
      Contact( #DATA.START_GLOBAL_REQUEST_LINE_1 )
      Contact( #DATA.START_GENERAL_CONDITIONS )
      Contact( #DATA.START_INITIAL_CONDITIONS_LINE_1 )
      Coil( #DATA.START_COMMAND_LINE_1 )
   END_RUNG
   // the same network as SCL:
   #DATA.START_COMMAND_LINE_1 := #DATA.START_GLOBAL_REQUEST_LINE_1 AND #DATA.START_GENERAL_CONDITIONS AND #DATA.START_INITIAL_CONDITIONS_LINE_1;
END_REGION

REGION Network 14: START COMMAND LINE 2 / Start Command
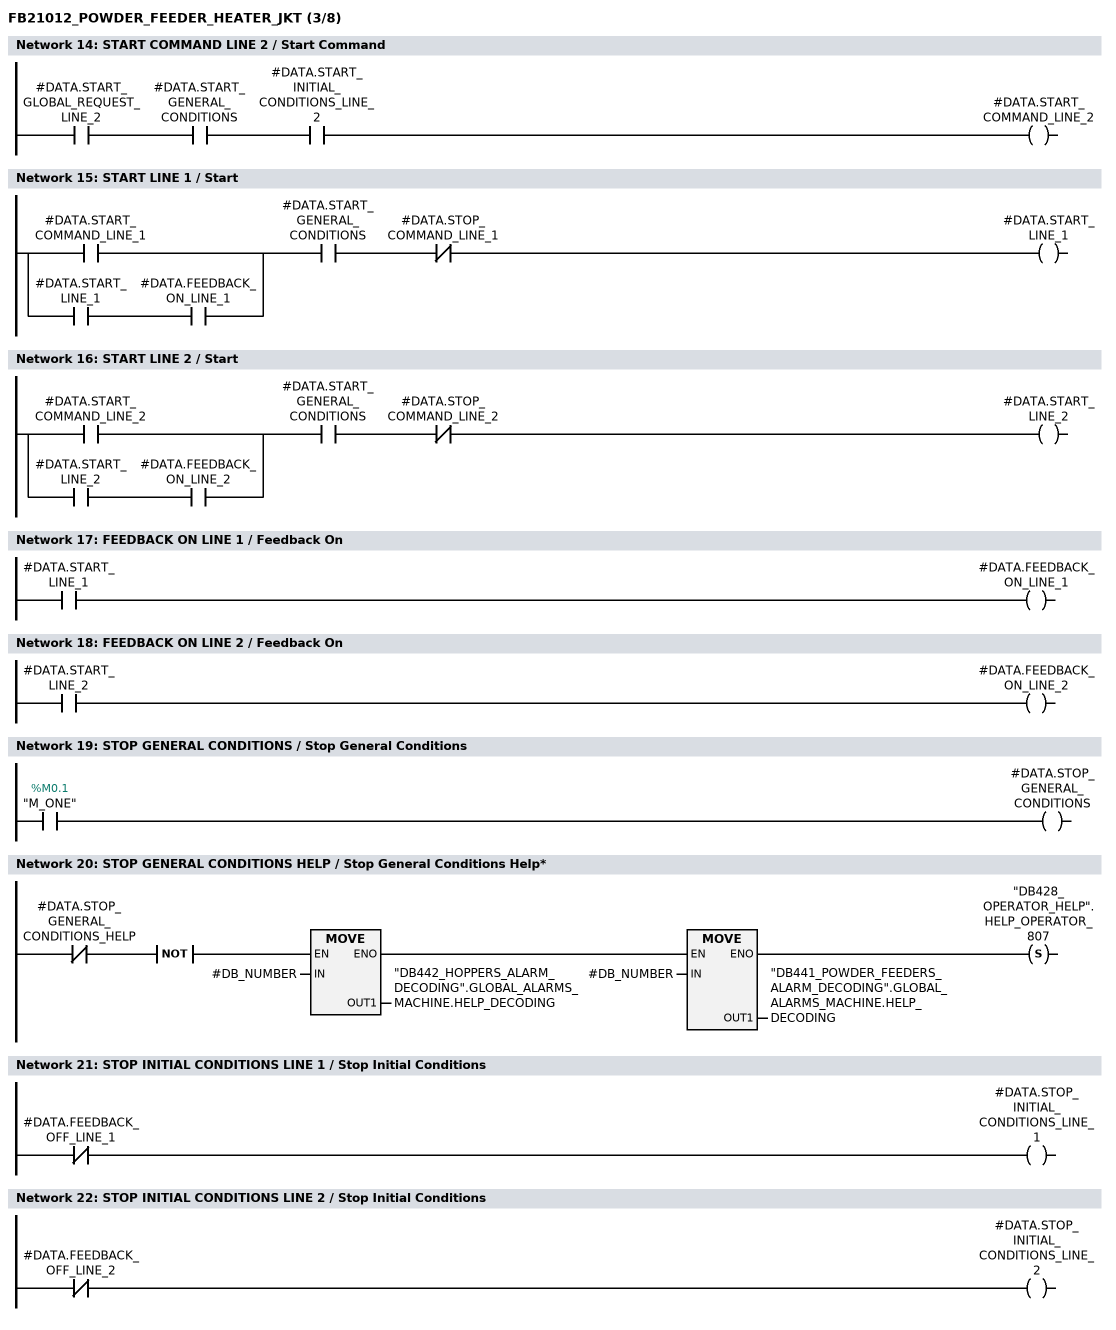
   RUNG wire#powerrail
      Contact( #DATA.START_GLOBAL_REQUEST_LINE_2 )
      Contact( #DATA.START_GENERAL_CONDITIONS )
      Contact( #DATA.START_INITIAL_CONDITIONS_LINE_2 )
      Coil( #DATA.START_COMMAND_LINE_2 )
   END_RUNG
   // the same network as SCL:
   #DATA.START_COMMAND_LINE_2 := #DATA.START_GLOBAL_REQUEST_LINE_2 AND #DATA.START_GENERAL_CONDITIONS AND #DATA.START_INITIAL_CONDITIONS_LINE_2;
END_REGION

REGION Network 15: START LINE 1 / Start
   RUNG wire#powerrail
      Contact( #DATA.START_COMMAND_LINE_1 )
      wire#w1
      Contact( #DATA.START_GENERAL_CONDITIONS )
      I_Contact( #DATA.STOP_COMMAND_LINE_1 )
      Coil( #DATA.START_LINE_1 )
   END_RUNG
   RUNG wire#powerrail
      Contact( #DATA.START_LINE_1 )
      Contact( #DATA.FEEDBACK_ON_LINE_1 )
   END_RUNG wire#w1
   // the same network as SCL:
   #DATA.START_LINE_1 := (#DATA.START_COMMAND_LINE_1 OR (#DATA.START_LINE_1 AND #DATA.FEEDBACK_ON_LINE_1)) AND #DATA.START_GENERAL_CONDITIONS AND NOT #DATA.STOP_COMMAND_LINE_1;
END_REGION

REGION Network 16: START LINE 2 / Start
   RUNG wire#powerrail
      Contact( #DATA.START_COMMAND_LINE_2 )
      wire#w1
      Contact( #DATA.START_GENERAL_CONDITIONS )
      I_Contact( #DATA.STOP_COMMAND_LINE_2 )
      Coil( #DATA.START_LINE_2 )
   END_RUNG
   RUNG wire#powerrail
      Contact( #DATA.START_LINE_2 )
      Contact( #DATA.FEEDBACK_ON_LINE_2 )
   END_RUNG wire#w1
   // the same network as SCL:
   #DATA.START_LINE_2 := (#DATA.START_COMMAND_LINE_2 OR (#DATA.START_LINE_2 AND #DATA.FEEDBACK_ON_LINE_2)) AND #DATA.START_GENERAL_CONDITIONS AND NOT #DATA.STOP_COMMAND_LINE_2;
END_REGION

REGION Network 17: FEEDBACK ON LINE 1 / Feedback On
   RUNG wire#powerrail
      Contact( #DATA.START_LINE_1 )
      Coil( #DATA.FEEDBACK_ON_LINE_1 )
   END_RUNG
   // the same network as SCL:
   #DATA.FEEDBACK_ON_LINE_1 := #DATA.START_LINE_1;
END_REGION

REGION Network 18: FEEDBACK ON LINE 2 / Feedback On
   RUNG wire#powerrail
      Contact( #DATA.START_LINE_2 )
      Coil( #DATA.FEEDBACK_ON_LINE_2 )
   END_RUNG
   // the same network as SCL:
   #DATA.FEEDBACK_ON_LINE_2 := #DATA.START_LINE_2;
END_REGION

REGION Network 19: STOP GENERAL CONDITIONS / Stop General Conditions
   RUNG wire#powerrail
      Contact( "M_ONE" )
      Coil( #DATA.STOP_GENERAL_CONDITIONS )
   END_RUNG
   // the same network as SCL:
   #DATA.STOP_GENERAL_CONDITIONS := "M_ONE";
END_REGION

REGION Network 20: STOP GENERAL CONDITIONS HELP / Stop General Conditions Help*
   RUNG wire#powerrail
      I_Contact( #DATA.STOP_GENERAL_CONDITIONS_HELP )
      Not()
      Move(in := #DB_NUMBER, out1 => "DB442_HOPPERS_ALARM_DECODING".GLOBAL_ALARMS_MACHINE.HELP_DECODING)
      Move(in := #DB_NUMBER, out1 => "DB441_POWDER_FEEDERS_ALARM_DECODING".GLOBAL_ALARMS_MACHINE.HELP_DECODING)
      S_Coil( "DB428_OPERATOR_HELP".HELP_OPERATOR_807 )
   END_RUNG
   // the same network as SCL:
   IF NOT (NOT #DATA.STOP_GENERAL_CONDITIONS_HELP) THEN
       "DB442_HOPPERS_ALARM_DECODING".GLOBAL_ALARMS_MACHINE.HELP_DECODING := #DB_NUMBER;
       "DB441_POWDER_FEEDERS_ALARM_DECODING".GLOBAL_ALARMS_MACHINE.HELP_DECODING := #DB_NUMBER;
       "DB428_OPERATOR_HELP".HELP_OPERATOR_807 := TRUE;
   END_IF;
END_REGION

REGION Network 21: STOP INITIAL CONDITIONS LINE 1 / Stop Initial Conditions
   RUNG wire#powerrail
      I_Contact( #DATA.FEEDBACK_OFF_LINE_1 )
      Coil( #DATA.STOP_INITIAL_CONDITIONS_LINE_1 )
   END_RUNG
   // the same network as SCL:
   #DATA.STOP_INITIAL_CONDITIONS_LINE_1 := NOT #DATA.FEEDBACK_OFF_LINE_1;
END_REGION

REGION Network 22: STOP INITIAL CONDITIONS LINE 2 / Stop Initial Conditions
   RUNG wire#powerrail
      I_Contact( #DATA.FEEDBACK_OFF_LINE_2 )
      Coil( #DATA.STOP_INITIAL_CONDITIONS_LINE_2 )
   END_RUNG
   // the same network as SCL:
   #DATA.STOP_INITIAL_CONDITIONS_LINE_2 := NOT #DATA.FEEDBACK_OFF_LINE_2;
END_REGION

REGION Network 23: STOP INITIAL CONDITIONS HELP / Stop Initial Conditions Help*
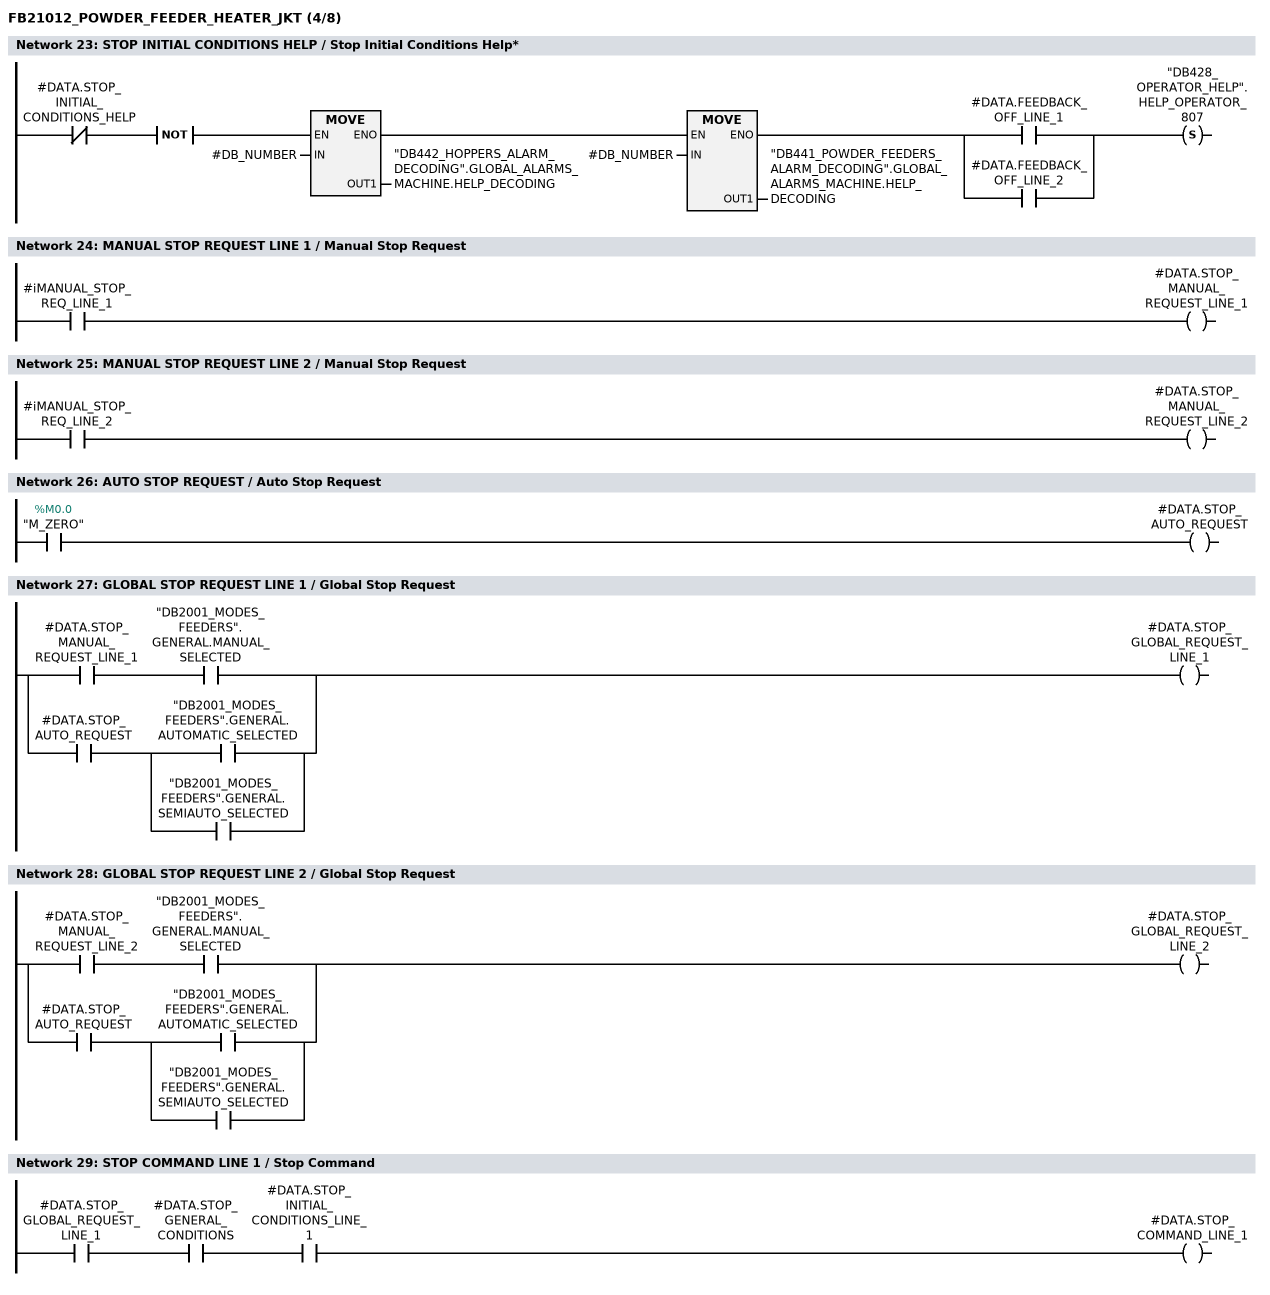
   RUNG wire#powerrail
      I_Contact( #DATA.STOP_INITIAL_CONDITIONS_HELP )
      Not()
      Move(in := #DB_NUMBER, out1 => "DB442_HOPPERS_ALARM_DECODING".GLOBAL_ALARMS_MACHINE.HELP_DECODING)
      Move(in := #DB_NUMBER, out1 => "DB441_POWDER_FEEDERS_ALARM_DECODING".GLOBAL_ALARMS_MACHINE.HELP_DECODING)
      wire#w1
      Contact( #DATA.FEEDBACK_OFF_LINE_1 )
      wire#w2
      S_Coil( "DB428_OPERATOR_HELP".HELP_OPERATOR_807 )
   END_RUNG
   RUNG wire#w1
      Contact( #DATA.FEEDBACK_OFF_LINE_2 )
   END_RUNG wire#w2
   // the same network as SCL:
   #_w1 := NOT (NOT #DATA.STOP_INITIAL_CONDITIONS_HELP);
   IF #_w1 THEN
       "DB442_HOPPERS_ALARM_DECODING".GLOBAL_ALARMS_MACHINE.HELP_DECODING := #DB_NUMBER;
       "DB441_POWDER_FEEDERS_ALARM_DECODING".GLOBAL_ALARMS_MACHINE.HELP_DECODING := #DB_NUMBER;
   END_IF;
   IF #_w1 AND (#DATA.FEEDBACK_OFF_LINE_1 OR #DATA.FEEDBACK_OFF_LINE_2) THEN
       "DB428_OPERATOR_HELP".HELP_OPERATOR_807 := TRUE;
   END_IF;
END_REGION

REGION Network 24: MANUAL STOP REQUEST LINE 1 / Manual Stop Request
   RUNG wire#powerrail
      Contact( #iMANUAL_STOP_REQ_LINE_1 )
      Coil( #DATA.STOP_MANUAL_REQUEST_LINE_1 )
   END_RUNG
   // the same network as SCL:
   #DATA.STOP_MANUAL_REQUEST_LINE_1 := #iMANUAL_STOP_REQ_LINE_1;
END_REGION

REGION Network 25: MANUAL STOP REQUEST LINE 2 / Manual Stop Request
   RUNG wire#powerrail
      Contact( #iMANUAL_STOP_REQ_LINE_2 )
      Coil( #DATA.STOP_MANUAL_REQUEST_LINE_2 )
   END_RUNG
   // the same network as SCL:
   #DATA.STOP_MANUAL_REQUEST_LINE_2 := #iMANUAL_STOP_REQ_LINE_2;
END_REGION

REGION Network 26: AUTO STOP REQUEST / Auto Stop Request
   RUNG wire#powerrail
      Contact( "M_ZERO" )
      Coil( #DATA.STOP_AUTO_REQUEST )
   END_RUNG
   // the same network as SCL:
   #DATA.STOP_AUTO_REQUEST := "M_ZERO";
END_REGION

REGION Network 27: GLOBAL STOP REQUEST LINE 1 / Global Stop Request
   RUNG wire#powerrail
      Contact( #DATA.STOP_MANUAL_REQUEST_LINE_1 )
      Contact( "DB2001_MODES_FEEDERS".GENERAL.MANUAL_SELECTED )
      wire#w1
      Coil( #DATA.STOP_GLOBAL_REQUEST_LINE_1 )
   END_RUNG
   RUNG wire#powerrail
      Contact( #DATA.STOP_AUTO_REQUEST )
      wire#w2
      Contact( "DB2001_MODES_FEEDERS".GENERAL.AUTOMATIC_SELECTED )
   END_RUNG wire#w1
   RUNG wire#w2
      Contact( "DB2001_MODES_FEEDERS".GENERAL.SEMIAUTO_SELECTED )
   END_RUNG wire#w1
   // the same network as SCL:
   #DATA.STOP_GLOBAL_REQUEST_LINE_1 := (#DATA.STOP_MANUAL_REQUEST_LINE_1 AND "DB2001_MODES_FEEDERS".GENERAL.MANUAL_SELECTED) OR (#DATA.STOP_AUTO_REQUEST AND ("DB2001_MODES_FEEDERS".GENERAL.AUTOMATIC_SELECTED OR "DB2001_MODES_FEEDERS".GENERAL.SEMIAUTO_SELECTED));
END_REGION

REGION Network 28: GLOBAL STOP REQUEST LINE 2 / Global Stop Request
   RUNG wire#powerrail
      Contact( #DATA.STOP_MANUAL_REQUEST_LINE_2 )
      Contact( "DB2001_MODES_FEEDERS".GENERAL.MANUAL_SELECTED )
      wire#w1
      Coil( #DATA.STOP_GLOBAL_REQUEST_LINE_2 )
   END_RUNG
   RUNG wire#powerrail
      Contact( #DATA.STOP_AUTO_REQUEST )
      wire#w2
      Contact( "DB2001_MODES_FEEDERS".GENERAL.AUTOMATIC_SELECTED )
   END_RUNG wire#w1
   RUNG wire#w2
      Contact( "DB2001_MODES_FEEDERS".GENERAL.SEMIAUTO_SELECTED )
   END_RUNG wire#w1
   // the same network as SCL:
   #DATA.STOP_GLOBAL_REQUEST_LINE_2 := (#DATA.STOP_MANUAL_REQUEST_LINE_2 AND "DB2001_MODES_FEEDERS".GENERAL.MANUAL_SELECTED) OR (#DATA.STOP_AUTO_REQUEST AND ("DB2001_MODES_FEEDERS".GENERAL.AUTOMATIC_SELECTED OR "DB2001_MODES_FEEDERS".GENERAL.SEMIAUTO_SELECTED));
END_REGION

